7.02 BOOL  ; #1测试NG推料气缸缩回位
7.03 BOOL  ; #1测试NG推料气缸伸出位
7.04 BOOL  ; #2测试NG推料气缸缩回位
7.05 BOOL  ; #2测试NG推料气缸伸出位
7.06 BOOL  ; 出料拉带有料感应
7.07 BOOL  ; 备用
7.08 BOOL  ; 扫码位有料感应
7.09 BOOL  ; 氦检启动OK
7.10 BOOL  ; #1氦检阀原位
7.11 BOOL  ; #2氦检原位
7.12 BOOL  ; #3氦检原位
7.13 BOOL  ; #4氦检原位
7.14 BOOL  ; 备用
7.15 BOOL  ; 可放料信号
8.00 BOOL  ; 进料伺服Serv_On
8.01 BOOL  ; 进料伺服Alarm_Clr
8.02 BOOL  ; 出料伺服Serv_On
8.03 BOOL  ; 出料伺服Alarm_Clr
8.04 BOOL  ; 前腔体进料伺服Serv_On
8.05 BOOL  ; 前腔体进料伺服Alarm_Clr
8.06 BOOL  ; 后腔体进料伺服Serv_On
8.07 BOOL  ; 后腔体进料伺服Alarm_Clr
8.08 BOOL  ; 前腔体出料伺服Serv_On
8.09 BOOL  ; 进料伺服Alarm_Clr
8.10 BOOL  ; 后腔体出料伺服Serv_On
8.11 BOOL  ; 后腔体出料伺服Alarm_Clr
8.12 BOOL  ; 启动指示灯
8.13 BOOL  ; 停止指示灯
8.14 BOOL  ; 复位指示灯
8.15 BOOL  ; 三色绿灯
9.00 BOOL  ; 三色红灯
9.01 BOOL  ; 三色黄灯
9.02 BOOL  ; 蜂鸣器
9.03 BOOL  ; #1真空泵启动
9.04 BOOL  ; 氦检电源打开
9.05 BOOL  ; 氦检仪启动
9.06 BOOL  ; 扫码阻挡
9.07 BOOL  ; 隔离夹紧气缸
9.08 BOOL  ; 上料夹爪气缸
9.09 BOOL  ; 进料升降伺服Serv_On
9.10 BOOL  ; 出料伺服Alarm_Clr
9.11 BOOL  ; 上料横移气缸缩回
9.12 BOOL  ; 上料横移气缸伸出
9.13 BOOL  ; 下料夹爪气缸
9.14 BOOL  ; 出料升降伺服Serv_On
9.15 BOOL  ; 下料#2级升降气缸
A202.00 BOOL  ; 通信端口0允许标志
A202.01 BOOL  ; 通信端口1允许标志
A202.02 BOOL  ; 通信端口2允许标志
A202.03 BOOL  ; 通信端口3允许标志
A202.04 BOOL  ; 通信端口4允许标志
A202.05 BOOL  ; 通信端口5允许标志
A202.06 BOOL  ; 通信端口6允许标志
A202.07 BOOL  ; 通信端口7允许标志
A250.04 BOOL  ; 单元4重启
A276 CHANNEL  ; 脉冲输出0 PV
A278 CHANNEL  ; 脉冲输出1 PV
A280.00 BOOL  ; 脉冲输出 0脉冲输出状态(0：恒速中,1：加减速中)
A280.01 BOOL  ; 脉冲输出 0当前值上溢/下溢
A280.02 BOOL  ; 脉冲输出0脉冲输出量设定
A280.03 BOOL  ; 脉冲输出 0脉冲输出完成
A280.04 BOOL  ; 脉冲输出 0脉冲输出中
A280.05 BOOL  ; 前上料伺服无原点标志(0：原点确定,1：原点未确定)
A280.06 BOOL  ; 脉冲输出 0原点停止标志(0：未停于原点,1：原点停止中)
A280.07 BOOL  ; 脉冲输出 0 原点搜索异常停止标志
A281.00 BOOL  ; 脉冲输出 1脉冲输出状态(0：恒速中,1：加减速中)
A281.01 BOOL  ; 脉冲输出 1当前值上溢/下溢
A281.02 BOOL  ; 脉冲输出1脉冲输出量设定
A281.03 BOOL  ; 脉冲输出 1脉冲输出完成
A281.04 BOOL  ; 脉冲输出 1脉冲输出中
A281.05 BOOL  ; 脉冲输出 1无原点标志(0：原点确定,1：原点未确定)
A281.06 BOOL  ; 脉冲输出 1原点停止标志(0：未停于原点,1：原点停止中)
A281.07 BOOL  ; 脉冲输出 1 原点搜索异常停止标志
A322 CHANNEL  ; 脉冲输出2 PV
A324 CHANNEL  ; 脉冲输出3 PV
A326.04 BOOL  ; 后上料伺服脉冲输出中
A326.05 BOOL  ; 后上料伺服无原点标志
A327.04 BOOL  ; 脉冲输出3脉冲输出中
A327.05 BOOL  ; 脉冲输出3无原点标志
A351 CHANNEL  ; 系统时间
A501.04 BOOL  ; 单元4模块重启
A623.01 BOOL  ; 3单元#1串口重启
A623.02 BOOL  ; 3单元#2串口重启
C0000 BOOL  ; 进料到后放料位次数
C0001 BOOL  ; MES离线模式下进料次数
C0010 BOOL  ; 1#腔清氦次数到达
C0020 BOOL  ; 2#腔清氦次数到达
C0030 BOOL  ; 3#腔清氦次数到达
C0040 BOOL  ; 4#腔清氦次数到达
C0060 BOOL  ; 自动重扫次数
C0090 BOOL  ; 出料到后取料位次数
D0 CHANNEL  ; PLC控制HMI切换的窗口编号
D1 CHANNEL  ; 当前窗口编号
D10 CHANNEL  ; 当前报警代码
D100 CHANNEL  ; #4腔体进入自保前时间
D1000 CHANNEL  ; 扫码自动运行步编号
D1001 CHANNEL  ; 前上料机构自动运行步编号
D1002 CHANNEL  ; 前下料机构自动运行步编号
D1003 CHANNEL  ; 后上料机构自动运行步编号
D1004 CHANNEL  ; 后下料机构自动运行步编号
D1005 CHANNEL  ; 1#腔体机构自动运行步编号
D1006 CHANNEL  ; 2#腔体机构自动运行步编号
D1007 CHANNEL  ; 3#腔体机构自动运行步编号
D1008 CHANNEL  ; 4#腔体机构自动运行步编号
D1009 CHANNEL  ; 出料机构自动运行步编号
D101 CHANNEL  ; #4腔体自保时间
D1010 CHANNEL  ; 扫码机构自动运行步编号
D10102 CHANNEL  ; 安东启动限制（0启动 1禁止）
D10103 CHANNEL  ; 启停故障原因
D10104 CHANNEL  ; PPM
D10105 CHANNEL  ; 启动限制断开（系统赋值1 PLC赋值0）
D10106 CHANNEL  ; 实时PPM
D10108 CHANNEL  ; 绿灯状态
D10109 CHANNEL  ; 红灯
D10110 CHANNEL  ; 黄灯
D10122 CHANNEL  ; 总投入
D10124 CHANNEL  ; .
D10126 CHANNEL  ; 总产出
D1015 CHANNEL  ; 1#腔体自动清氦步编号
D1016 CHANNEL  ; 2#腔体自动清氦步编号
D1017 CHANNEL  ; 3#腔体自动清氦步编号
D1018 CHANNEL  ; 4#腔体自动清氦步编号
D11 CHANNEL  ; 当前报警数量
D1142 CHANNEL  ; #1腔体测试结果
D1144 CHANNEL  ; #2腔体测试结果
D1146 CHANNEL  ; #3测试结果
D1148 CHANNEL  ; #4腔体测试结果
D1152 CHANNEL  ; 放OK品次数
D1154 CHANNEL  ; 放NG品次数
D116 CHANNEL  ; 前上料往腔体1放料安全位置
D1160 CHANNEL  ; 生产总数
D1162 CHANNEL  ; 生产OK品总数
D1164 CHANNEL  ; 生产NG品总数
D1166 CHANNEL  ; 良品率(%)
D118 CHANNEL  ; 前下料腔体1取料安全位
D1200 CHANNEL  ; 腔体真空阀值
D1202 CHANNEL  ; 腔体抽真空时间
D1204 CHANNEL  ; 检漏口压力设定值
D1206 CHANNEL  ; 漏率设定值
D1208 CHANNEL  ; 电池破真空阀值
D1210 CHANNEL  ; 氦检仪稳定设定时间
D1212 CHANNEL  ; 腔体破真空阀值
D1214 CHANNEL  ; 腔体抽氦后压力
D1216 CHANNEL  ; 自检真空阀值
D1218 CHANNEL  ; 自检抽真空时间
D1220 CHANNEL  ; 自检泄漏量
D1222 CHANNEL  ; 自检保压前延时-HMI
D1224 CHANNEL  ; 自检保压时间-HMI
D1226 CHANNEL  ; 氦检时间
D1228 CHANNEL  ; 抽残气时间
D1229 CHANNEL  ; 抽残气压力达到延时
D1230 CHANNEL  ; 电池抽真空阀值
D1232 CHANNEL  ; 电池抽真空时间
D1234 CHANNEL  ; 注氦后压力
D1236 CHANNEL  ; 电池抽氦后压力
D1238 CHANNEL  ; 注氦气时间
D1240 CHANNEL  ; 氦检时的真空阀值
D1242 CHANNEL  ; 充氦压力下限值Pa(F)
D1246 CHANNEL  ; 充氦压力上限值Pa(F)
D1250 CHANNEL  ; 检漏口压力设定值小数部分
D1252 CHANNEL  ; 检漏口压力设定值指数
D1254 CHANNEL  ; 漏率设定值小数部分
D1256 CHANNEL  ; 漏率设定值指数
D1260 CHANNEL  ; 检漏口压力设定值指数部分
D1264 CHANNEL  ; 漏率设定值指数部分
D1266 CHANNEL  ; 漏率设定值(浮点数Pa.m3)
D1270 CHANNEL  ; 注氦嘴气密性设定值小数部分
D1272 CHANNEL  ; 注氦嘴气密性设定值指数
D1274 CHANNEL  ; 注氦嘴气密性设定值指数部分
D1276 CHANNEL  ; 注氦嘴气密性设定值(Float)
D1278 CHANNEL  ; 清氦次数设定值
D1280 CHANNEL  ; 1#腔体抽气阀关闭延时
D1282 CHANNEL  ; 2#腔体抽气阀关闭延时
D1284 CHANNEL  ; 3#腔体抽气阀关闭延时
D1286 CHANNEL  ; 4#腔体抽气阀关闭延时
D1290 CHANNEL  ; 1#腔体抽残气时间
D1292 CHANNEL  ; 2#腔体抽残气时间
D1294 CHANNEL  ; 3#腔体抽残气时间
D1296 CHANNEL  ; 4#腔体抽残气时间
D130 CHANNEL  ; 前腔体电池NG状态
D130.00 BOOL  ; 1#腔电池NG
D130.01 BOOL  ; 2#腔电池NG
D131 CHANNEL  ; 后腔体电池NG状态
D1310 CHANNEL  ; 氦检仪稳定漏率设定值小数
D1312 CHANNEL  ; 氦检仪稳定漏率设定值指数
D1316 CHANNEL  ; 氦检仪稳定漏率设定值(Float)
D131.00 BOOL  ; 3#腔电池NG
D131.01 BOOL  ; 4#腔电池NG
D1330 CHANNEL  ; #1腔体注氦压力阀值
D1332 CHANNEL  ; #2腔体注氦压力阀值
D1334 CHANNEL  ; #3腔体注氦压力阀值
D1336 CHANNEL  ; #4腔体注氦压力阀值
D1342 CHANNEL  ; 充氦压力下限值kPa(F)
D1346 CHANNEL  ; 充氦压力上限值kPa(F)
D135 CHANNEL  ; 清氦失败腔体号
D1350 CHANNEL  ; 1#腔体充氦时电池实际压力（浮点）
D1352 CHANNEL  ; 1#腔体氦检时腔体实际压力（浮点）
D1354 CHANNEL  ; 2#腔体充氦时电池实际压力（浮点）
D1356 CHANNEL  ; 2#腔体氦检时腔体实际压力（浮点）
D1358 CHANNEL  ; 3#腔体充氦时电池实际压力（浮点）
D1360 CHANNEL  ; 3#腔体氦检时腔体实际压力（浮点）
D1362 CHANNEL  ; 4#腔体充氦时电池实际压力（浮点）
D1364 CHANNEL  ; 4#腔体氦检时腔体实际压力（浮点）
D1366 CHANNEL  ; 前下料爪 充氦时电池实际压力（浮点）
D1368 CHANNEL  ; 前下料爪 氦检时腔体实际压力（浮点）
D1370 CHANNEL  ; 后下料爪 充氦时电池实际压力（浮点）
D1372 CHANNEL  ; 后下料爪 氦检时腔体实际压力（浮点）
D14 CHANNEL  ; 感应器ON延时时间
D1400 CHANNEL  ; #1连续NG次数
D1401 CHANNEL  ; #2腔体连续NG次数
D1402 CHANNEL  ; #3腔体连续NG次数
D1403 CHANNEL  ; #4腔体连续NG次数
D1410 CHANNEL  ; 连续NG报警设定
D1411 CHANNEL  ; 自动离线次数
D1412 CHANNEL  ; NG报警状态
D1415 CHANNEL  ; 写数据超时时间
D1416 CHANNEL  ; 氦检仪压力异常延时
D1500 CHANNEL  ; 来料隔离气缸缩回位
D1501 CHANNEL  ; 来料隔离气缸伸出位屏蔽延时时间
D1502 CHANNEL  ; 扫码阻挡气缸缩回位屏蔽延时时间
D1503 CHANNEL  ; 扫码阻挡气缸伸出屏蔽延时时间
D1504 CHANNEL  ; 上料夹爪张开位屏蔽延时时间
D1505 CHANNEL  ; 上料夹爪夹紧位屏蔽延时时间
D1506 CHANNEL  ; 上料#1气缸缩回位蔽延时时间
D1507 CHANNEL  ; 上料#1气缸伸出位屏蔽延时时间
D1508 CHANNEL  ; 上料#2气缸缩回位屏蔽延时
D1509 CHANNEL  ; 上料#2气缸伸出位屏蔽延时
D1510 CHANNEL  ; 上料横移气缸缩回位屏蔽延时
D1511 CHANNEL  ; 上料横移气缸伸出位屏蔽延时
D1512 CHANNEL  ; 下料夹爪张开位蔽延时时间
D1513 CHANNEL  ; 下料夹爪夹紧位屏蔽延时时间
D1514 CHANNEL  ; 下料#1升降气缸缩回位屏蔽延时
D1515 CHANNEL  ; 下料#1级升降气缸伸出位屏蔽延时
D1516 CHANNEL  ; 下料#2级升降气缸缩回位蔽延时时间
D1517 CHANNEL  ; 下料#2级升降气缸伸出位屏蔽延时时间
D1518 CHANNEL  ; 下料横移气缸缩回位蔽延时时间
D1519 CHANNEL  ; 下料横移气缸伸出位屏蔽延时
D1520 CHANNEL  ; 拉带进料夹爪有料感应延时时间
D1521 CHANNEL  ; 拉带出料夹爪有料感应延时时间
D1522 CHANNEL  ; 前腔体进料夹爪有料感应屏蔽延时
D1523 CHANNEL  ; 前腔体出料夹爪有料感应屏蔽延时
D1524 CHANNEL  ; 后腔体进料夹爪有料感应
D1525 CHANNEL  ; 后腔体出料夹爪有料感应
D1526 CHANNEL  ; 精密调压阀过低报警
D1527 CHANNEL  ; 后腔体出料位顶升气缸伸出位屏蔽延时
D1528 CHANNEL  ; 前腔体进料机械手夹爪张开位屏蔽延时时间
D1529 CHANNEL  ; 前腔体进料机械手夹爪夹紧位屏蔽延时
D1530 CHANNEL  ; 前腔体进料机械手升降气缸缩回位屏蔽延时
D1531 CHANNEL  ; 前腔体进料机械手升降气缸伸出位屏蔽延时
D1532 CHANNEL  ; 后腔体进料机械手张开位屏蔽延时
D1533 CHANNEL  ; 后腔体进料机械手夹爪夹紧位屏蔽延时
D1534 CHANNEL  ; 后腔体进料机械手升降气缸缩回位屏蔽延时
D1535 CHANNEL  ; 后腔体进料机械手升降气缸伸出位屏蔽延时
D1536 CHANNEL  ; 前腔体上料机械手夹爪张开位屏蔽延时
D1537 CHANNEL  ; 前腔体出料机械手夹爪夹紧位屏蔽延时
D1538 CHANNEL  ; 前腔体出料机械手升降气缸缩回位屏蔽延时
D1539 CHANNEL  ; 前腔体出料机械手升降气缸伸出位屏蔽延时
D1540 CHANNEL  ; 后腔体出料机械手夹爪张开位屏蔽延时
D1541 CHANNEL  ; 后腔体出料机械手夹爪夹紧位屏蔽延时
D1542 CHANNEL  ; 后腔体出料机械手升降气缸缩回位屏蔽延时
D1543 CHANNEL  ; 后腔体出料机械手升降气缸伸出位屏蔽延时
D1544 CHANNEL  ; #1腔体移栽气缸缩回位屏蔽延时
D1545 CHANNEL  ; #1腔体移栽气缸伸出位屏蔽延时
D1546 CHANNEL  ; #1腔体顶升气缸缩回位屏蔽延时
D1547 CHANNEL  ; #1腔体顶升气缸伸出位屏蔽延时
D1548 CHANNEL  ; #2腔体移栽气缸缩回位屏蔽延时
D1549 CHANNEL  ; #2腔体移栽气缸伸出位屏蔽延时
D1550 CHANNEL  ; #2腔体顶升气缸缩回位屏蔽延时
D1551 CHANNEL  ; #2腔体顶升气缸伸出位屏蔽延时
D1552 CHANNEL  ; #3腔体移栽气缸缩回位屏蔽延时
D1553 CHANNEL  ; #3腔体移栽气缸伸出位屏蔽延时
D1554 CHANNEL  ; #3腔体顶升气缸缩回位屏蔽延时
D1555 CHANNEL  ; #3腔体顶升气缸伸出位屏蔽延时
D1556 CHANNEL  ; #4腔体移栽气缸缩回位屏蔽延时
D1557 CHANNEL  ; #4腔体移栽气缸伸出位屏蔽延时
D1558 CHANNEL  ; #4腔体顶升气缸缩回位屏蔽延时
D1559 CHANNEL  ; #4腔体顶升气缸伸出位屏蔽延时
D1560 CHANNEL  ; #1扫码NG推料气缸缩回位屏蔽延时
D1561 CHANNEL  ; #1扫码NG推料气缸伸出位屏蔽延时
D1562 CHANNEL  ; #2扫码NG推料气缸缩回位屏蔽延时
D1563 CHANNEL  ; #2扫码NG推料气缸伸出位屏蔽延时
D1564 CHANNEL  ; #1测试NG推料气缸缩回位屏蔽延时
D1565 CHANNEL  ; #1测试NG推料气缸伸出屏蔽延时
D1566 CHANNEL  ; #2测试NG推料气缸缩回位屏蔽延时
D1567 CHANNEL  ; #2测试NG推料气缸伸出位屏蔽延时
D1568 CHANNEL  ; 前进料旋转气缸初始位屏蔽延时时间
D1569 CHANNEL  ; 前进料旋转气缸旋转位屏蔽延时时间
D1570 CHANNEL  ; 前出料旋转气缸初始位屏蔽延时时间
D1571 CHANNEL  ; 前出料旋转气缸旋转位屏蔽延时时间
D1572 CHANNEL  ; 后进料旋转气缸初始位屏蔽延时时间
D1573 CHANNEL  ; 后进料旋转气缸旋转位屏蔽延时时间
D1574 CHANNEL  ; 后出料旋转气缸初始位屏蔽延时时间
D1575 CHANNEL  ; 后出料旋转气缸旋转位屏蔽延时时间
D1580 CHANNEL  ; 腔体1左电池密封气缸上位屏蔽延时时间
D1581 CHANNEL  ; 腔体1左电池密封气缸下位屏蔽延时时间
D1582 CHANNEL  ; 腔体1右电池密封气缸上位屏蔽延时时间
D1583 CHANNEL  ; 腔体1右电池密封气缸下位屏蔽延时时间
D1584 CHANNEL  ; 腔体2左电池密封气缸上位屏蔽延时时间
D1585 CHANNEL  ; 腔体2左电池密封气缸下位屏蔽延时时间
D1586 CHANNEL  ; 腔体2右电池密封气缸上位屏蔽延时时间
D1587 CHANNEL  ; 腔体2右电池密封气缸下位屏蔽延时时间
D1588 CHANNEL  ; 腔体3左电池密封气缸上位屏蔽延时时间
D1589 CHANNEL  ; 腔体3左电池密封气缸下位屏蔽延时时间
D1590 CHANNEL  ; 腔体3右电池密封气缸上位屏蔽延时时间
D1591 CHANNEL  ; 腔体3右电池密封气缸下位屏蔽延时时间
D1592 CHANNEL  ; 腔体4左电池密封气缸上位屏蔽延时时间
D1593 CHANNEL  ; 腔体4左电池密封气缸下位屏蔽延时时间
D1594 CHANNEL  ; 腔体4右电池密封气缸上位屏蔽延时时间
D1595 CHANNEL  ; 腔体4右电池密封气缸下位屏蔽延时时间
D1596 CHANNEL  ; 腔体1平移气缸后退位屏蔽延时时间
D1597 CHANNEL  ; 腔体1平移气缸前进位屏蔽延时时间
D1598 CHANNEL  ; 腔体1顶升气缸下位屏蔽延时时间
D1599 CHANNEL  ; 腔体1顶升气缸上位屏蔽延时时间
D16 CHANNEL  ; 感应器Off延时时间
D1600 CHANNEL  ; 腔体2平移气缸后退位屏蔽延时时间
D1601 CHANNEL  ; 腔体2平移气缸前进位屏蔽延时时间
D1602 CHANNEL  ; 腔体2顶升气缸下位屏蔽延时时间
D1603 CHANNEL  ; 腔体2顶升气缸上位屏蔽延时时间
D1604 CHANNEL  ; 腔体3平移气缸后退位屏蔽延时时间
D1605 CHANNEL  ; 腔体3平移气缸前进位屏蔽延时时间
D1606 CHANNEL  ; 腔体3顶升气缸下位屏蔽延时时间
D1607 CHANNEL  ; 腔体3顶升气缸上位屏蔽延时时间
D1608 CHANNEL  ; 腔体4平移气缸后退位屏蔽延时时间
D1609 CHANNEL  ; 腔体4平移气缸前进位屏蔽延时时间
D1610 CHANNEL  ; 腔体4顶升气缸下位屏蔽延时时间
D1611 CHANNEL  ; 腔体4顶升气缸上位屏蔽延时时间
D1700 CHANNEL  ; 左进料阻挡气缸放行位屏蔽设定时间
D1701 CHANNEL  ; 左进料阻挡气缸阻挡位屏蔽设定时间
D1702 CHANNEL  ; 右进料阻挡气缸放行位屏蔽设定时间
D1703 CHANNEL  ; 右进料阻挡气缸阻挡位屏蔽设定时间
D1704 CHANNEL  ; 左扫码阻挡气缸放行位屏蔽设定时间
D1705 CHANNEL  ; 左扫码阻挡气缸阻挡位屏蔽设定时间
D1706 CHANNEL  ; 右扫码阻挡气缸放行位屏蔽设定时间
D1707 CHANNEL  ; 右扫码阻挡气缸阻挡位屏蔽设定时间
D1708 CHANNEL  ; 扫码NG缓存避位气缸接料位屏蔽设定时间
D1709 CHANNEL  ; 扫码NG缓存避位气缸避位位屏蔽设定时间
D1710 CHANNEL  ; 扫码NG缓存接料气缸后退位屏蔽设定时间
D1711 CHANNEL  ; 扫码NG缓存接料气缸前进位屏蔽设定时间
D1712 CHANNEL  ; 扫码NG缓存间隔气缸上位屏蔽设定时间
D1713 CHANNEL  ; 扫码NG缓存间隔气缸下位屏蔽设定时间
D1716 CHANNEL  ; 进料机械手升降气缸上位屏蔽设定时间
D1717 CHANNEL  ; 进料机械手升降气缸下位屏蔽设定时间
D1718 CHANNEL  ; 进料机械手平移气缸开位屏蔽设定时间
D1719 CHANNEL  ; 进料机械手平移气缸合位屏蔽设定时间
D1720 CHANNEL  ; 进料机械手左夹爪气缸张开位屏蔽设定时间
D1721 CHANNEL  ; 进料机械手左夹爪气缸夹紧位屏蔽设定时间
D1722 CHANNEL  ; 进料机械手右夹爪气缸张开位屏蔽设定时间
D1723 CHANNEL  ; 进料机械手右夹爪气缸夹紧位屏蔽设定时间
D1724 CHANNEL  ; 出料机械手升降气缸上位屏蔽设定时间
D1725 CHANNEL  ; 出料机械手升降气缸下位屏蔽设定时间
D1726 CHANNEL  ; 出料机械手平移气缸开位屏蔽设定时间
D1727 CHANNEL  ; 出料机械手平移气缸合位屏蔽设定时间
D1728 CHANNEL  ; 出料机械手左夹爪气缸张开位屏蔽设定时间
D1729 CHANNEL  ; 出料机械手左夹爪气缸夹紧位屏蔽设定时间
D1730 CHANNEL  ; 出料机械手右夹爪气缸张开位屏蔽设定时间
D1731 CHANNEL  ; 出料机械手右夹爪气缸夹紧位屏蔽设定时间
D1732 CHANNEL  ; 前上料机械手1级升降气缸上位屏蔽设定时间
D1733 CHANNEL  ; 前上料机械手1级升降气缸下位屏蔽设定时间
D1734 CHANNEL  ; 前上料机械手2级升降气缸上位屏蔽设定时间
D1735 CHANNEL  ; 前上料机械手2级升降气缸下位屏蔽设定时间
D1736 CHANNEL  ; 前上料机械手左夹爪气缸张开位屏蔽设定时间
D1737 CHANNEL  ; 前上料机械手左夹爪气缸夹紧位屏蔽设定时间
D1738 CHANNEL  ; 前上料机械手右夹爪气缸张开位屏蔽设定时间
D1739 CHANNEL  ; 前上料机械手右夹爪气缸夹紧位屏蔽设定时间
D1740 CHANNEL  ; 前取料机械手1级升降气缸上位屏蔽设定时间
D1741 CHANNEL  ; 前取料机械手1级升降气缸下位屏蔽设定时间
D1742 CHANNEL  ; 前取料机械手2级升降气缸上位屏蔽设定时间
D1743 CHANNEL  ; 前取料机械手2级升降气缸下位屏蔽设定时间
D1744 CHANNEL  ; 前取料机械手左夹爪气缸张开位屏蔽设定时间
D1745 CHANNEL  ; 前取料机械手左夹爪气缸夹紧位屏蔽设定时间
D1746 CHANNEL  ; 前取料机械手右夹爪气缸张开位屏蔽设定时间
D1747 CHANNEL  ; 前取料机械手右夹爪气缸夹紧位屏蔽设定时间
D1748 CHANNEL  ; 后上料机械手1级升降气缸上位屏蔽设定时间
D1749 CHANNEL  ; 后上料机械手1级升降气缸下位屏蔽设定时间
D1750 CHANNEL  ; 后上料机械手2级升降气缸上位屏蔽设定时间
D1751 CHANNEL  ; 后上料机械手2级升降气缸下位屏蔽设定时间
D1752 CHANNEL  ; 后上料机械手左夹爪气缸张开位屏蔽设定时间
D1753 CHANNEL  ; 后上料机械手左夹爪气缸夹紧位屏蔽设定时间
D1754 CHANNEL  ; 后上料机械手右夹爪气缸张开位屏蔽设定时间
D1755 CHANNEL  ; 后上料机械手右夹爪气缸夹紧位屏蔽设定时间
D1756 CHANNEL  ; 后取料机械手1级升降气缸上位屏蔽设定时间
D1757 CHANNEL  ; 后取料机械手1级升降气缸下位屏蔽设定时间
D1758 CHANNEL  ; 后取料机械手2级升降气缸上位屏蔽设定时间
D1759 CHANNEL  ; 后取料机械手2级升降气缸下位屏蔽设定时间
D1760 CHANNEL  ; 后取料机械手左夹爪气缸张开位屏蔽设定时间
D1761 CHANNEL  ; 后取料机械手左夹爪气缸夹紧位屏蔽设定时间
D1762 CHANNEL  ; 后取料机械手右夹爪气缸张开位屏蔽设定时间
D1763 CHANNEL  ; 后取料机械手右夹爪气缸夹紧位屏蔽设定时间
D1764 CHANNEL  ; 前NG拨料气缸后位屏蔽设定时间
D1765 CHANNEL  ; 前NG拨料气缸前位屏蔽设定时间
D1766 CHANNEL  ; 后NG拨料气缸后位屏蔽设定时间
D1767 CHANNEL  ; 后NG拨料气缸前位屏蔽设定时间
D1768 CHANNEL  ; 前进料旋转气缸初始位屏蔽设定时间
D1769 CHANNEL  ; 前进料旋转气缸旋转位屏蔽设定时间
D1770 CHANNEL  ; 前出料旋转气缸初始位屏蔽设定时间
D1771 CHANNEL  ; 前出料旋转气缸旋转位屏蔽设定时间
D1772 CHANNEL  ; 后进料旋转气缸初始位屏蔽设定时间
D1773 CHANNEL  ; 后进料旋转气缸旋转位屏蔽设定时间
D1774 CHANNEL  ; 后出料旋转气缸初始位屏蔽设定时间
D1775 CHANNEL  ; 后出料旋转气缸旋转位屏蔽设定时间
D1780 CHANNEL  ; 腔体1左电池密封气缸上位屏蔽设定时间
D1781 CHANNEL  ; 腔体1左电池密封气缸下位屏蔽设定时间
D1782 CHANNEL  ; 腔体1右电池密封气缸上位屏蔽设定时间
D1783 CHANNEL  ; 腔体1右电池密封气缸下位屏蔽设定时间
D1784 CHANNEL  ; 腔体2左电池密封气缸上位屏蔽设定时间
D1785 CHANNEL  ; 腔体2左电池密封气缸下位屏蔽设定时间
D1786 CHANNEL  ; 腔体2右电池密封气缸上位屏蔽设定时间
D1787 CHANNEL  ; 腔体2右电池密封气缸下位屏蔽设定时间
D1788 CHANNEL  ; 腔体3左电池密封气缸上位屏蔽设定时间
D1789 CHANNEL  ; 腔体3左电池密封气缸下位屏蔽设定时间
D1790 CHANNEL  ; 腔体3右电池密封气缸上位屏蔽设定时间
D1791 CHANNEL  ; 腔体3右电池密封气缸下位屏蔽设定时间
D1792 CHANNEL  ; 腔体4左电池密封气缸上位屏蔽设定时间
D1793 CHANNEL  ; 腔体4左电池密封气缸下位屏蔽设定时间
D1794 CHANNEL  ; 腔体4右电池密封气缸上位屏蔽设定时间
D1795 CHANNEL  ; 腔体4右电池密封气缸下位屏蔽设定时间
D1796 CHANNEL  ; 腔体1平移气缸后退位屏蔽设定时间
D1797 CHANNEL  ; 腔体1平移气缸前进位屏蔽设定时间
D1798 CHANNEL  ; 腔体1顶升气缸下位屏蔽设定时间
D1799 CHANNEL  ; 腔体1顶升气缸上位屏蔽设定时间
D18 CHANNEL  ; 自动运行条件延时时间
D1800 CHANNEL  ; 腔体2平移气缸后退位屏蔽设定时间
D1801 CHANNEL  ; 腔体2平移气缸前进位屏蔽设定时间
D1802 CHANNEL  ; 腔体2顶升气缸下位屏蔽设定时间
D1803 CHANNEL  ; 腔体2顶升气缸上位屏蔽设定时间
D1804 CHANNEL  ; 腔体3平移气缸后退位屏蔽设定时间
D1805 CHANNEL  ; 腔体3平移气缸前进位屏蔽设定时间
D1806 CHANNEL  ; 腔体3顶升气缸下位屏蔽设定时间
D1807 CHANNEL  ; 腔体3顶升气缸上位屏蔽设定时间
D1808 CHANNEL  ; 腔体4平移气缸后退位屏蔽设定时间
D1809 CHANNEL  ; 腔体4平移气缸前进位屏蔽设定时间
D1810 CHANNEL  ; 腔体4顶升气缸下位屏蔽设定时间
D1811 CHANNEL  ; 腔体4顶升气缸上位屏蔽设定时间
D19 CHANNEL  ; 自动运行步间间隔时间
D2 CHANNEL  ; 机台有柔性报警
D20 CHANNEL  ; 轴控位置预置
D2000 CHANNEL  ; 进料水平伺服手动低速加速时间
D2001 CHANNEL  ; 进料伺服手动低速加速时间
D2002 CHANNEL  ; 进料水平移载伺服手动低速减速时间
D2003 CHANNEL  ; 进料伺服手动低速减速时间
D2004 CHANNEL  ; 进料水平移载伺服手动低速速度
D2005 CHANNEL  ; 进料伺服手动低速速度
D2006 CHANNEL  ; 进料伺服手动低速输出脉冲
D20068 CHANNEL  ; 进料伺服定位位置
D20069 CHANNEL  ; 进料伺服定位位置
D2007 CHANNEL  ; 进料伺服手动低速输出脉冲
D20070 CHANNEL  ; 进料伺服定位速度
D20071 CHANNEL  ; 进料伺服定位速度
D20072 CHANNEL  ; 进料伺服加速时间
D20073 CHANNEL  ; 进料伺服加速时间
D20074 CHANNEL  ; 进料伺服减速时间
D20075 CHANNEL  ; 进料伺服减速时间
D2008 CHANNEL  ; 进料水平移载伺服手动当前速度
D20080 CHANNEL  ; 出料伺服定位位置
D20081 CHANNEL  ; 出料伺服定位位置
D20082 CHANNEL  ; 出料伺服定位速度
D20083 CHANNEL  ; 出料伺服定位速度
D20084 CHANNEL  ; 出料伺服加速时间
D20085 CHANNEL  ; 出料伺服加速时间
D20086 CHANNEL  ; 出料伺服减速时间
D20087 CHANNEL  ; 出料伺服减速时间
D2009 CHANNEL  ; 进料伺服手动当前速度
D20092 CHANNEL  ; 进料伺服当前位置
D20093 CHANNEL  ; 进料伺服当前位置
D20096 CHANNEL  ; 出料伺服当前位置
D20097 CHANNEL  ; 出料伺服当前位置
D2010 CHANNEL  ; 进料移载伺服手动高速加速时间
D2011 CHANNEL  ; 进料伺服手动高速加速时间
D2012 CHANNEL  ; 进料移载伺服手动高速减速时间
D20124 CHANNEL  ; 进料伺服定位位置
D20126 CHANNEL  ; 进料水平移载伺服定位速度
D20128 CHANNEL  ; 进料水平伺服加速时间
D2013 CHANNEL  ; 进料伺服手动高速减速时间
D20130 CHANNEL  ; 进料水平伺服减速度
D20136 CHANNEL  ; 出料伺服定位位置
D20138 CHANNEL  ; 出料移载伺服定位速度
D2014 CHANNEL  ; 进料伺服手动高速速度
D20140 CHANNEL  ; 出料移载伺服加速时间
D20142 CHANNEL  ; 出料移载伺服减速时间
D20148 CHANNEL  ; 进料升降伺服定位位置
D2015 CHANNEL  ; 进料伺服手动高速速度
D20150 CHANNEL  ; 进料升降伺服定位速度
D20152 CHANNEL  ; 进料升降伺服加速时间
D20154 CHANNEL  ; 进料升降伺服减速度
D2016 CHANNEL  ; 进料伺服手动高速输出脉冲
D20160 CHANNEL  ; 出料升降伺服定位位置
D20162 CHANNEL  ; 出料升降伺服定位速度
D20164 CHANNEL  ; 出料升降伺服加速时间
D20166 CHANNEL  ; 出料升降伺服减速时间
D2017 CHANNEL  ; 进料伺服手动高速输出脉冲
D20172 CHANNEL  ; 进料移载伺服当前位置
D20176 CHANNEL  ; 出料移载伺服当前位置
D2018 CHANNEL  ; 进料伺服寸动距离
D20180 CHANNEL  ; 进料升降伺服当前位置
D20184 CHANNEL  ; 出料升降伺服当前位置
D2019 CHANNEL  ; 进料伺服寸动距离
D2020 CHANNEL  ; 进料水平移载伺服自动加速时间
D2021 CHANNEL  ; 进料伺服自动加速时间
D2022 CHANNEL  ; 进料水平移载伺服自动减速时间
D2023 CHANNEL  ; 进料伺服自动减速时间
D2024 CHANNEL  ; 进料移载伺服自动速度
D2025 CHANNEL  ; 进料伺服自动速度
D2026 CHANNEL  ; 进料伺服自动输出脉冲
D2027 CHANNEL  ; 进料伺服自动输出脉冲
D2028 CHANNEL  ; 进料伺服自动速度2(低速)
D2030 CHANNEL  ; #4扫码NG位
D2031 CHANNEL  ; 进料伺服待机位置
D2032 CHANNEL  ; 进料水平伺服上料位置
D2033 CHANNEL  ; 进料伺服上料位置
D2034 CHANNEL  ; 进料水平伺服前放料位
D2035 CHANNEL  ; 进料伺服前放料位
D2036 CHANNEL  ; 进料水平伺服后放料位
D2037 CHANNEL  ; 进料伺服后放料位
D2040 CHANNEL  ; #1扫码NG位
D2041 CHANNEL  ; 外部拉带安全运行进料伺服位置
D2042 CHANNEL  ; #2扫码NG位
D2044 CHANNEL  ; #3扫码NG位
D2046 CHANNEL  ; #4扫码NG位
D2050 CHANNEL  ; 进出料转盘直径
D2080 CHANNEL  ; #2扫码NG位
D2082 CHANNEL  ; 前进料转盘后直径边缘位置
D2084 CHANNEL  ; 后进料转盘前直径边缘位置
D2086 CHANNEL  ; 后进料转盘后直径边缘位置
D2100 CHANNEL  ; 前上料伺服手动低速加速比率
D2101 CHANNEL  ; 前上料伺服手动低速减速比率
D2102 CHANNEL  ; 前上料伺服手动低速速度
D2103 CHANNEL  ; 前上料伺服手动低速速度
D2104 CHANNEL  ; 前上料伺服手动低速输出脉冲
D2105 CHANNEL  ; 前上料伺服手动输出脉冲
D2106 CHANNEL  ; 前上料伺服手动启动速度
D2107 CHANNEL  ; 前上料伺服手动启动速度
D2108 CHANNEL  ; 前上料伺服手动当前速度
D2109 CHANNEL  ; 前上料伺服手动当前速度
D2110 CHANNEL  ; 前上料伺服手动高速加速比率
D2111 CHANNEL  ; 前上料伺服手动高速减速比率
D2112 CHANNEL  ; 前上料伺服手动高速速度
D2113 CHANNEL  ; 前上料伺服手动高速速度
D2114 CHANNEL  ; 前上料伺服手动高速输出脉冲
D2115 CHANNEL  ; 前上料伺服手动高速输出脉冲
D2116 CHANNEL  ; 前上料伺服手动高速启动速度
D2117 CHANNEL  ; 前上料伺服手动高速启动速度
D2118 CHANNEL  ; 前上料伺服寸动距离
D2119 CHANNEL  ; 前上料伺服寸动距离
D2120 CHANNEL  ; 前上料伺服自动加速比率
D2121 CHANNEL  ; 前上料伺服自动减速比率
D2122 CHANNEL  ; 前上料伺服自动速度
D2123 CHANNEL  ; 前上料伺服自动速度
D2124 CHANNEL  ; 前上料伺服自动输出脉冲
D2125 CHANNEL  ; 前上料伺服自动输出脉冲
D2126 CHANNEL  ; 前上料伺服自动启动速度
D2127 CHANNEL  ; 前上料伺服自动启动速度
D2130 CHANNEL  ; 前上料伺服待机位置
D2131 CHANNEL  ; 前上料伺服待机位置
D2132 CHANNEL  ; 前上料伺服上料位置
D2133 CHANNEL  ; 前上料伺服上料位置
D2134 CHANNEL  ; 前上料伺服仓1放料位
D2135 CHANNEL  ; 前上料伺服仓1放料位
D2136 CHANNEL  ; 前上料伺服仓2放料位
D2137 CHANNEL  ; 前上料伺服仓2放料位
D2140 CHANNEL  ; 安全位置
D2141 CHANNEL  ; 安全位置
D2150 CHANNEL  ; 前上料伺服上料位置
D2154 CHANNEL  ; 前上料伺服仓1放料位
D2160 CHANNEL  ; 前上料伺服仓2放料位
D220 CHANNEL  ; 接收检漏仪状态的起始字
D2200 CHANNEL  ; 前下料伺服手动低速加速比率
D2201 CHANNEL  ; 前下料伺服手动低速减速比率
D2202 CHANNEL  ; 前下料伺服手动低速速度
D2203 CHANNEL  ; 前下料伺服手动低速速度
D2204 CHANNEL  ; 前下料伺服手动输出脉冲
D2205 CHANNEL  ; 前下料伺服手动输出脉冲
D2206 CHANNEL  ; 前下料伺服手动启动速度
D2207 CHANNEL  ; 前下料伺服手动启动速度
D2208 CHANNEL  ; 前下料伺服手动当前速度
D2209 CHANNEL  ; 前下料伺服手动当前速度
D221 CHANNEL  ; 接收的检漏仪状态
D2210 CHANNEL  ; 前下料伺服手动高速加速比率
D2211 CHANNEL  ; 前下料伺服手动高速减速比率
D2212 CHANNEL  ; 前下料伺服手动高速速度
D2213 CHANNEL  ; 前下料伺服手动高速速度
D2214 CHANNEL  ; 前下料伺服手动高速输出脉冲
D2215 CHANNEL  ; 前下料伺服手动高速输出脉冲
D2216 CHANNEL  ; 前下料伺服手动高速启动速度
D2217 CHANNEL  ; 前下料伺服手动高速启动速度
D2218 CHANNEL  ; 前下料伺服寸动距离
D2219 CHANNEL  ; 前下料伺服寸动距离
D2220 CHANNEL  ; 前下料伺服自动加速比率
D2221 CHANNEL  ; 前下料伺服自动减速比率
D2222 CHANNEL  ; 前下料伺服自动速度与上料相同
D2223 CHANNEL  ; 前下料伺服自动速度
D2224 CHANNEL  ; 前下料伺服自动输出脉冲
D2225 CHANNEL  ; 前下料伺服自动输出脉冲
D2226 CHANNEL  ; 前下料伺服自动启动速度
D2227 CHANNEL  ; 前下料伺服自动启动速度
D2230 CHANNEL  ; 前下料伺服待机位置
D2231 CHANNEL  ; 前下料伺服待机位置
D2232 CHANNEL  ; 前下料伺服仓1取料位
D2233 CHANNEL  ; 前下料伺服仓1取料位
D2234 CHANNEL  ; 前下料伺服仓2取料位
D2235 CHANNEL  ; 前下料伺服仓2取料位
D2236 CHANNEL  ; 前下料伺服放料位
D2237 CHANNEL  ; 前下料伺服OK放料位
D2238 CHANNEL  ; 前下料伺服NG放料位
D2239 CHANNEL  ; 前下料伺服NG放料位
D2300 CHANNEL  ; 后上料伺服手动低速加速比率
D2301 CHANNEL  ; 后上料伺服手动低速减速比率
D2302 CHANNEL  ; 后上料伺服手动低速速度
D2303 CHANNEL  ; 后上料伺服手动低速速度
D2304 CHANNEL  ; 后上料伺服手动输出脉冲
D2305 CHANNEL  ; 后上料伺服手动输出脉冲
D2306 CHANNEL  ; 后上料伺服手动启动速度
D2307 CHANNEL  ; 后上料伺服手动启动速度
D2308 CHANNEL  ; 后上料伺服手动当前速度
D2309 CHANNEL  ; 后上料伺服手动当前速度
D2310 CHANNEL  ; 后上料伺服手动高速加速比率
D2311 CHANNEL  ; 后上料伺服手动高速减速比率
D2312 CHANNEL  ; 后上料伺服手动高速速度
D2313 CHANNEL  ; 后上料伺服手动高速速度
D2314 CHANNEL  ; 后上料伺服手动高速输出脉冲
D2315 CHANNEL  ; 后上料伺服手动高速输出脉冲
D2316 CHANNEL  ; 后上料伺服手动高速启动速度
D2317 CHANNEL  ; 后上料伺服手动高速启动速度
D2318 CHANNEL  ; 后上料伺服寸动距离
D2319 CHANNEL  ; 后上料伺服寸动距离
D2320 CHANNEL  ; 后上料伺服自动加速比率
D2321 CHANNEL  ; 后上料伺服自动减速比率
D2322 CHANNEL  ; 后上料伺服自动速度
D2323 CHANNEL  ; 后上料伺服自动速度
D2324 CHANNEL  ; 后上料伺服自动输出脉冲
D2325 CHANNEL  ; 后上料伺服自动输出脉冲
D2326 CHANNEL  ; 后上料伺服自动启动速度
D2327 CHANNEL  ; 后上料伺服自动启动速度
D2330 CHANNEL  ; 后上料伺服待机位置
D2331 CHANNEL  ; 后上料伺服待机位置
D2332 CHANNEL  ; 后上料伺服上料位置
D2333 CHANNEL  ; 后上料伺服上料位置
D2334 CHANNEL  ; 后上料伺服仓3放料位
D2335 CHANNEL  ; 后上料伺服仓3放料位
D2336 CHANNEL  ; 后上料伺服仓4放料位
D2337 CHANNEL  ; 后上料伺服仓4放料位
D240 CHANNEL  ; 接收检漏仪状态起始字
D2400 CHANNEL  ; 后下料伺服手动低速加速比率
D2401 CHANNEL  ; 后下料伺服手动低速减速比率
D2402 CHANNEL  ; 后下料伺服手动低速速度
D2403 CHANNEL  ; 后下料伺服手动低速速度
D2404 CHANNEL  ; 后下料伺服手动输出脉冲
D2405 CHANNEL  ; 后下料伺服手动输出脉冲
D2406 CHANNEL  ; 后下料伺服手动启动速度
D2407 CHANNEL  ; 后下料伺服手动启动速度
D2408 CHANNEL  ; 后下料伺服手动当前速度
D2409 CHANNEL  ; 后下料伺服手动当前速度
D241 CHANNEL  ; 接收检漏仪状态起始字(ASCII)
D2410 CHANNEL  ; 后下料伺服手动高速加速比率
D2411 CHANNEL  ; 后下料伺服手动高速减速比率
D2412 CHANNEL  ; 后下料伺服手动高速速度
D2413 CHANNEL  ; 后下料伺服手动高速速度
D2414 CHANNEL  ; 后下料伺服手动高速输出脉冲
D2415 CHANNEL  ; 后下料伺服手动高速输出脉冲
D2416 CHANNEL  ; 后下料伺服手动高速启动速度
D2417 CHANNEL  ; 后下料伺服手动高速启动速度
D2418 CHANNEL  ; 后下料伺服寸动距离
D2419 CHANNEL  ; 后下料伺服寸动距离
D2420 CHANNEL  ; 后下料伺服自动加速比率
D2421 CHANNEL  ; 后下料伺服自动减速比率
D2422 CHANNEL  ; 后下料伺服自动速度
D2423 CHANNEL  ; 后下料伺服自动速度
D2424 CHANNEL  ; 后下料伺服自动输出脉冲
D2425 CHANNEL  ; 后下料伺服自动输出脉冲
D2426 CHANNEL  ; 后下料伺服自动启动速度
D2427 CHANNEL  ; 后下料伺服自动启动速度
D2430 CHANNEL  ; 后下料伺服待机位置
D2431 CHANNEL  ; 后下料伺服待机位置
D2432 CHANNEL  ; 后下料伺服仓3取料位
D2433 CHANNEL  ; 后下料伺服仓3取料位
D2434 CHANNEL  ; 后下料伺服仓4取料位
D2435 CHANNEL  ; 后下料伺服仓4取料位
D2436 CHANNEL  ; 后下料伺服OK放料位
D2437 CHANNEL  ; 后下料伺服OK放料位
D2438 CHANNEL  ; 后下料伺服NG放料位
D2439 CHANNEL  ; 后下料伺服NG放料位
D2440 CHANNEL  ; 下料2#NG放料位
D2442 CHANNEL  ; 下料3#NG放料位
D2444 CHANNEL  ; 下料4#NG放料位
D250 CHANNEL  ; 接收检漏口压力的起始字
D2500 CHANNEL  ; 进料升降伺服当前位置
D2504 CHANNEL  ; 进料升降伺服手动低速速度
D2506 CHANNEL  ; 进料升降伺服自动加速时间
D251 CHANNEL  ; 接收检漏口压力(ASCII)
D2510 CHANNEL  ; 进料升降伺服到取料位
D2512 CHANNEL  ; 进料伺服取放料高中
D2514 CHANNEL  ; 进料升降伺服放料位
D2520 CHANNEL  ; 升降伺到取料位
D260 CHANNEL  ; 接收漏率起始字
D2600 CHANNEL  ; 进料升降手动低速加速时间
D2602 CHANNEL  ; 进料升降手动低速减速时间
D261 CHANNEL  ; 接收的漏率(ASCII)
D2620 CHANNEL  ; 进料升降伺服自动加速时间
D2622 CHANNEL  ; 进料升降伺服自动减速时间
D2700 CHANNEL  ; 出料升降伺服当前位置
D2704 CHANNEL  ; 出料升降伺服手动低速速度
D2706 CHANNEL  ; 出料升降自动速度
D2710 CHANNEL  ; 出料升降伺服取料高度
D2712 CHANNEL  ; 出为料升降伺服放料高度
D2720 CHANNEL  ; 出料升降伺服定位位置
D2800 CHANNEL  ; 出料升降伺服手动低速加速时间
D2802 CHANNEL  ; 出料升降伺服手动低速减速时间
D2820 CHANNEL  ; 出料升降伺服自动加速时间
D2822 CHANNEL  ; 出料升降伺服自动减速时间
D2900 CHANNEL  ; 出料伺服手动低速加速时间
D2901 CHANNEL  ; 出料伺服手动低速加速时间
D2902 CHANNEL  ; 出料伺服手动低速减速时间
D2903 CHANNEL  ; 出料伺服手动低速减速时间
D2904 CHANNEL  ; 出料伺服手动低速速度
D2905 CHANNEL  ; 出料伺服手动低速速度
D2906 CHANNEL  ; 出料伺服手动低速输出脉冲
D2907 CHANNEL  ; 出料伺服手动低速输出脉冲
D2908 CHANNEL  ; 出料伺服手动当前速度
D2909 CHANNEL  ; 出料伺服手动当前速度
D2910 CHANNEL  ; 出料伺服手动高速加速时间
D2911 CHANNEL  ; 出料伺服手动高速加速时间
D2912 CHANNEL  ; 出料伺服手动高速减速时间
D2913 CHANNEL  ; 出料伺服手动高速减速时间
D2914 CHANNEL  ; 出料伺服手动高速速度
D2915 CHANNEL  ; 出料伺服手动高速速度
D2916 CHANNEL  ; 出料伺服手动高速输出脉冲
D2917 CHANNEL  ; 出料伺服手动高速输出脉冲
D2918 CHANNEL  ; 出料伺服寸动距离
D2919 CHANNEL  ; 出料伺服寸动距离
D2920 CHANNEL  ; 出料伺服自动加速时间
D2921 CHANNEL  ; 出料伺服自动加速时间
D2922 CHANNEL  ; 出料伺服自动减速时间
D2923 CHANNEL  ; 出料伺服自动减速时间
D2924 CHANNEL  ; 出料伺服自动速度
D2925 CHANNEL  ; 出料伺服自动速度
D2926 CHANNEL  ; 出料伺服自动输出脉冲
D2927 CHANNEL  ; 出料伺服自动输出脉冲
D2928 CHANNEL  ; 出料伺服自动速度2(低速)
D2930 CHANNEL  ; 出料伺服待机位置
D2931 CHANNEL  ; 出料伺服待机位置
D2932 CHANNEL  ; 出料伺服前取料位置
D2933 CHANNEL  ; 出料伺服前取料位置
D2934 CHANNEL  ; 出料伺服后取料位置
D2935 CHANNEL  ; 出料伺服后取料位置
D2936 CHANNEL  ; 出料轴出料位
D2937 CHANNEL  ; 出料伺服放料位
D2938 CHANNEL  ; 出料伺服#1NG测试位置
D2940 CHANNEL  ; 出料伺服#2NG测试位
D2942 CHANNEL  ; 出料伺服#3NG位
D2944 CHANNEL  ; 出料伺服#4NG位
D2980 CHANNEL  ; 前出料转盘前直径边缘位置
D2982 CHANNEL  ; 前出料转盘后直径边缘位置
D2984 CHANNEL  ; 后出料转盘前直径边缘位置
D2986 CHANNEL  ; 后出料转盘后直径边缘位置
D30 CHANNEL  ; #1腔体状态(停用，待料中，测试中，测试完成
D300 CHANNEL  ; #1腔体检漏口压力(浮点)
D3000 CHANNEL  ; 进料水平伺服当前位置
D3010 CHANNEL  ; 间隔气缸下降条件
D302 CHANNEL  ; #1腔体清氦氦检完成时检漏口压力(浮点)
D3030 CHANNEL  ; 进料伺服自动定位位置
D310 CHANNEL  ; #2腔体检漏口压力(浮点)
D3100 CHANNEL  ; 前腔体上料伺服当前位置
D312 CHANNEL  ; #2腔体清氦氦检完成时检漏口压力(浮点)
D3120 CHANNEL  ; 前上料伺服当前定位位置(M)
D3130 CHANNEL  ; 前上料伺服自动定位位置
D3140 CHANNEL  ; 腔体1检测有料开始位置
D3142 CHANNEL  ; 腔体1检测最后位置
D3144 CHANNEL  ; 腔体2检测有料开始位置
D3146 CHANNEL  ; 腔体2检测结束位
D32 CHANNEL  ; #2腔体状态(停用，待料中，测试中，测试完成
D320 CHANNEL  ; #3腔体检漏口压力(浮点)
D3200 CHANNEL  ; 前下料伺服当前位置
D322 CHANNEL  ; #3腔体清氦氦检完成时检漏口压力(浮点)
D3220 CHANNEL  ; 前下料伺服当前定位位置(M)
D3230 CHANNEL  ; 前下料伺服自动定位位置
D330 CHANNEL  ; #4腔体检漏口压力(浮点)
D3300 CHANNEL  ; 后腔体上料伺服当前位置
D332 CHANNEL  ; #4腔体清氦氦检完成时检漏口压力(浮点)
D3320 CHANNEL  ; 后上料伺服当前定位位置(M)
D3330 CHANNEL  ; 后上料伺服自动定位位置
D3340 CHANNEL  ; 腔体3检测有料开始位置
D3342 CHANNEL  ; 腔体3检测最后位置
D3344 CHANNEL  ; 腔体4检测有料开始位置
D3346 CHANNEL  ; 腔体4检测最后位置
D34 CHANNEL  ; #3腔体状态(停用，待料中，测试中，测试完成
D3400 CHANNEL  ; 后下料伺服当前位置
D3420 CHANNEL  ; 后下料伺服当前定位位置(M)
D3430 CHANNEL  ; 后下料伺服自动定位位置
D36 CHANNEL  ; #4腔体状态(停用，待料中，测试中，测试完成
D370 CHANNEL  ; 氦检仪就绪状态
D3900 CHANNEL  ; 出料移载伺服当前位置
D3920 CHANNEL  ; 出料伺服当前定位位置(M)
D3930 CHANNEL  ; 出料伺服自动定位位置
D40 CHANNEL  ; 腔体真空达到阀值
D400 CHANNEL  ; #1腔体漏率(浮点)
D4000 CHANNEL  ; 真空值1转存
D4002 CHANNEL  ; #1真空值运算1
D4004 CHANNEL  ; #1真空值运算2
D4006 CHANNEL  ; #1真空值运算3
D4008 CHANNEL  ; #1真空值运算4
D4010 CHANNEL  ; 腔体1实际真空值(浮点)
D402 CHANNEL  ; #1腔体清氦氦检完成时漏率(浮点)
D4020 CHANNEL  ; 真空值2转存
D4022 CHANNEL  ; #2真空值运算1
D4024 CHANNEL  ; #2真空值运算2
D4026 CHANNEL  ; #2真空值运算3
D4028 CHANNEL  ; #2真空值运算4
D4030 CHANNEL  ; 腔体2实际真空值(浮点)
D4040 CHANNEL  ; 真空值3转存
D4042 CHANNEL  ; #3真空值运算1
D4044 CHANNEL  ; #3真空值运算2
D4046 CHANNEL  ; #3真空值运算3
D4048 CHANNEL  ; #3真空值运算4
D4050 CHANNEL  ; 腔体3实际真空值(浮点)
D4060 CHANNEL  ; 真空3转存
D4062 CHANNEL  ; #4真空值运算1
D4064 CHANNEL  ; #4真空值运算2
D4066 CHANNEL  ; #4真空值运算3
D4068 CHANNEL  ; #4真空值运算4
D4070 CHANNEL  ; 腔体4实际真空值(浮点)
D410 CHANNEL  ; #2腔体漏率(浮点)
D4100 CHANNEL  ; #1电池真空压力表模拟量读数
D4104 CHANNEL  ; #1电池真空压力表读数(浮点)
D4108 CHANNEL  ; #1电池真空压力表计算一
D4110 CHANNEL  ; 氦检开启时腔体实际压力
D4112 CHANNEL  ; #1电池真空压力表计算二
D4116 CHANNEL  ; #1电池真空压力表读数(#1电池真空)
D412 CHANNEL  ; #2腔体清氦氦检完成时漏率(浮点)
D4120 CHANNEL  ; #2电池真空压力表模拟量读数
D4124 CHANNEL  ; #2电池真空压力表读数(浮点)
D4128 CHANNEL  ; #2电池真空压力表计算一
D4132 CHANNEL  ; #2电池真空压力表计算二
D4136 CHANNEL  ; #2电池真空压力表读数
D4140 CHANNEL  ; #3电池真空压力表模拟量读数
D4144 CHANNEL  ; #3电池真空压力表模拟量读数(浮点)
D4148 CHANNEL  ; #3电池真空压力表计算一
D4152 CHANNEL  ; #3电池真空压力表计算二
D4156 CHANNEL  ; #3电池真空压力表读数
D4160 CHANNEL  ; #4电池真空压力表模拟量读数
D4164 CHANNEL  ; #4电池真空压力表模拟量读数(浮点)
D4168 CHANNEL  ; #4电池真空压力表计算一
D4172 CHANNEL  ; #4电池真空压力表计算二
D4176 CHANNEL  ; #4电池真空压力表读数(实际真空值)
D4180 CHANNEL  ; 1#电池真空压力修正系数
D4182 CHANNEL  ; 2#电池真空压力修正系数
D4184 CHANNEL  ; 3#电池真空压力修正系数
D4186 CHANNEL  ; 4#电池真空压力修正系数
D4188 CHANNEL  ; 压力系数5
D42 CHANNEL  ; 腔体抽气时间
D420 CHANNEL  ; #3腔体漏率(浮点)
D4200 CHANNEL  ; #1密封气缸压力表读数(模拟量)
D4204 CHANNEL  ; 1#密封气缸压力表模拟量读数(浮点)
D4216 CHANNEL  ; 1#密封气缸压力表读数(实际压力值)
D422 CHANNEL  ; #3腔体清氦氦检完成时漏率(浮点)
D4220 CHANNEL  ; 2#密封气缸压力表读数(模拟量)
D4224 CHANNEL  ; 2#密封气缸压力表模拟量读数(浮点)
D4236 CHANNEL  ; 2#密封气缸压力表读数(实际压力值)
D4240 CHANNEL  ; 3#密封气缸压力表读数(模拟量)
D4244 CHANNEL  ; 3#密封气缸压力表模拟量读数(浮点)
D4256 CHANNEL  ; 3#密封气缸压力表读数(实际压力值)
D4260 CHANNEL  ; 4#密封气缸压力表读数(模拟量)
D4264 CHANNEL  ; 4#密封气缸压力表模拟量读数(浮点)
D4276 CHANNEL  ; 4#密封气缸压力表读数(实际压力值)
D430 CHANNEL  ; #4腔体漏率(浮点)
D4300 CHANNEL  ; #1腔体保压前真空值
D4304 CHANNEL  ; #1腔体保压后真空值
D4308 CHANNEL  ; #1腔体泄漏量
D432 CHANNEL  ; #4腔体清氦氦检完成时漏率(浮点)
D4320 CHANNEL  ; #2腔体保压前真空
D4324 CHANNEL  ; #2腔体保压后真空
D4328 CHANNEL  ; #2腔体泄漏量
D4340 CHANNEL  ; #3腔体保压前真空
D4344 CHANNEL  ; #3腔体保压后真空
D4348 CHANNEL  ; #3腔体泄漏量
D4360 CHANNEL  ; #4腔体保压前真空
D4364 CHANNEL  ; #4腔体保压后真空
D4368 CHANNEL  ; #4腔体泄漏量
D450 CHANNEL  ; 氦检仪当前实时漏率
D46 CHANNEL  ; 氦检设定时间
D4900 CHANNEL  ; 扫码位暂存码1
D4910 CHANNEL  ; 取料位条码
D50 CHANNEL  ; #1腔体正常抽气时间
D500 CHANNEL  ; 检漏压力
D5000 CHANNEL  ; 扫码1长度
D5001 CHANNEL  ; #1条码
D5020 CHANNEL  ; 条码1在进料爪子
D5060 CHANNEL  ; 条码2在进料爪子
D51 CHANNEL  ; #1电池正常抽气时间
D510 CHANNEL  ; 检漏口压力 浮点
D5100 CHANNEL  ; 在前进料托盘
D5120 CHANNEL  ; 在前上料爪子
D5140 CHANNEL  ; 条码在仓1
D5160 CHANNEL  ; 条码1在仓2
D5180 CHANNEL  ; 条码1在前下料爪子
D52 CHANNEL  ; #2腔体正常抽气时间
D520 CHANNEL  ; 检漏口压力最小值
D5200 CHANNEL  ; 在前进料托盘
D5220 CHANNEL  ; 在前上料爪子
D5240 CHANNEL  ; 条码在仓1
D5260 CHANNEL  ; 条码2在仓2
D5280 CHANNEL  ; 条码2在前下料爪子
D53 CHANNEL  ; #2电池正常抽气时间
D5300 CHANNEL  ; NG位1#条码
D5320 CHANNEL  ; 条码在前出料托盘
D5360 CHANNEL  ; 出料爪上1#条码
D54 CHANNEL  ; #3腔体正常抽气时间
D5400 CHANNEL  ; NG位2#条码
D5420 CHANNEL  ; 条码在前出料托盘
D5460 CHANNEL  ; 出料爪上2#条码
D55 CHANNEL  ; #3电池正常抽气时间
D5510 CHANNEL  ; #1腔检漏口压力
D5512 CHANNEL  ; #1、2腔检漏口压力在前出料托盘
D5516 CHANNEL  ; #1、2腔压力在出料爪子
D5520 CHANNEL  ; #2腔检漏口压力在前下料夹爪
D5530 CHANNEL  ; 腔检漏口压力在NG
D5540 CHANNEL  ; #1/2腔注氦后压力(kPa)(前NG位)
D5550 CHANNEL  ; 前NG位测试结果
D56 CHANNEL  ; #4腔体正常抽气时间
D5610 CHANNEL  ; #1腔体漏率
D5612 CHANNEL  ; 1、2腔体漏率在前出料托盘
D5616 CHANNEL  ; 1、2腔体漏率在出料爪子
D5620 CHANNEL  ; #2腔漏率在前下料夹爪
D5630 CHANNEL  ; 1#腔充氦压力(kPa)在前下料夹爪
D5632 CHANNEL  ; #1、2腔充氦压力在前出料托盘
D5636 CHANNEL  ; #1、2腔充氦压力在出料夹爪
D5640 CHANNEL  ; 腔体漏率
D5650 CHANNEL  ; 1#腔测试结果在前下料夹爪
D5652 CHANNEL  ; #1、2腔测试结果在前出料托盘
D5656 CHANNEL  ; #1、2腔测试结果在出料夹爪
D5660 CHANNEL  ; 2#腔充氦压力(kPa)在前下料夹爪
D5670 CHANNEL  ; 2#腔测试结果在前下料夹爪
D57 CHANNEL  ; #4电池正常抽气时间
D5800 CHANNEL  ; 数据上传位电池的检漏口压力
D5802 CHANNEL  ; 后下料机械手检漏口压力
D5804 CHANNEL  ; 检漏口压在出料托盘
D5900 CHANNEL  ; 数据上传位电池的漏率
D5902 CHANNEL  ; 后下料机械手漏率
D5904 CHANNEL  ; 漏率在出料托盘
D5910 CHANNEL  ; 数据上传位电池充氦压力
D5912 CHANNEL  ; 后下料机械手充氦压力
D5914 CHANNEL  ; 充氦压力在出料托盘
D5920 CHANNEL  ; 数据上传位电池测试结果
D5922 CHANNEL  ; 后下料机械手电池测试结果
D5924 CHANNEL  ; 测试结果在出料托盘
D5930 CHANNEL  ; 前下料机械手电池腔体位置
D5932 CHANNEL  ; 后下料机械手电池腔体位置
D5934 CHANNEL  ; 腔体位置到出料托盘
D60 CHANNEL  ; 接收条码数据字长度
D600 CHANNEL  ; 氦检下限位值
D6000 CHANNEL  ; 设备OEE状态(0-待机,10-正常,70-故障)
D6003.05 BOOL  ; 300A_0_2St TR_Down
D602 CHANNEL  ; 氦检上限位值
D6110 CHANNEL  ; 流入个数
D6204 CHANNEL  ; #1腔体测试完成时的检漏口压力
D6206 CHANNEL  ; #1腔体测试完成时漏率
D6214 CHANNEL  ; #2腔体测试完成时的检漏口压力
D6216 CHANNEL  ; #2腔体测试完成时漏率
D6224 CHANNEL  ; #3腔体测试完成时检漏口压力
D6226 CHANNEL  ; #3腔体测试完成时漏率
D6234 CHANNEL  ; #4腔体测试完成时检漏口压力
D6236 CHANNEL  ; #4腔体测试完成时漏率
D651 CHANNEL  ; 报警时检漏口压力
D66 CHANNEL  ; 设定条码长度
D670 CHANNEL  ; 报警时检漏口压力
D68 CHANNEL  ; 设定条码字长度
D700 CHANNEL  ; 氦检设定时间(储存)
D7000 CHANNEL  ; 扫码2长度
D7001 CHANNEL  ; #2条码
D702 CHANNEL  ; 检漏口压力设定值小数部分(储存)
D704 CHANNEL  ; 检漏口压力设定值指数(储存)
D706 CHANNEL  ; 漏率设定值小数部分(储存)
D708 CHANNEL  ; 漏率设定值指数(储存)
D7100 CHANNEL  ; 在后进料托盘
D7120 CHANNEL  ; 在后上料爪子
D7140 CHANNEL  ; 条码在仓3
D7160 CHANNEL  ; 条码在仓4
D7180 CHANNEL  ; 条码在后下料爪子
D720 CHANNEL  ; 设备状态
D7200 CHANNEL  ; 在后进料托盘
D721 CHANNEL  ; 设备状态(储存)
D722 CHANNEL  ; 设备状态变更
D7220 CHANNEL  ; 在后上料爪子
D7240 CHANNEL  ; 条码在仓3
D7260 CHANNEL  ; 条码在仓4
D7280 CHANNEL  ; 条码在后下料爪子
D730 CHANNEL  ; 早班分、秒
D7300 CHANNEL  ; 条码在NG
D731 CHANNEL  ; 早班日、时
D7320 CHANNEL  ; 条码在后出料托盘
D733 CHANNEL  ; 晚班分、秒
D734 CHANNEL  ; 晚班日、时
D736 CHANNEL  ; 只比较时、分、秒
D7360 CHANNEL  ; 条码在出料爪
D740 CHANNEL  ; 单班生产时间
D7400 CHANNEL  ; 条码在NG
D742 CHANNEL  ; 单班故障时间
D7420 CHANNEL  ; 条码在后出料托盘
D7460 CHANNEL  ; 条码在出料爪
D7510 CHANNEL  ; #3腔检漏口压力在后下料夹爪
D7512 CHANNEL  ; #3、4腔检漏口压力在后托盘
D7516 CHANNEL  ; 出料夹爪上电池的检漏口压力
D7520 CHANNEL  ; #4检漏口压力
D7530 CHANNEL  ; #3、4腔检漏口压力在后NG位
D7540 CHANNEL  ; 后NG位注氦后压力(kPa）
D7550 CHANNEL  ; 后NG位结果类型
D7610 CHANNEL  ; #3腔体漏率在后下料夹爪
D7612 CHANNEL  ; #3、4腔体漏率在后托盘
D7616 CHANNEL  ; 出料夹爪上电池的漏率
D7620 CHANNEL  ; #4腔体漏率
D7630 CHANNEL  ; #3腔体充氦压力在后下料夹爪
D7632 CHANNEL  ; #3/4腔体充氦压力在后出料托盘
D7636 CHANNEL  ; #3/4腔体充氦压力在出料夹爪
D7640 CHANNEL  ; #3、4腔漏率在后NG位
D7650 CHANNEL  ; #3腔体测试结果在后下料夹爪
D7652 CHANNEL  ; #3/4腔体测试结果在后出料托盘
D7656 CHANNEL  ; #3/4腔体测试结果在出料夹爪
D7660 CHANNEL  ; #4腔体充氦压力在后下料夹爪
D7670 CHANNEL  ; #4腔体测试结果在后下料夹爪
D7800 CHANNEL  ; 数据上传位1#条码
D7820 CHANNEL  ; 条码在后下料爪子
D7840 CHANNEL  ; 条码在出料托盘
D7900 CHANNEL  ; 数据上传位2#条码
D800 CHANNEL  ; 扫码步
D8000 CHANNEL  ; 检漏状态第一字节
D8001 CHANNEL  ; 检漏状态第二字节
D8002 CHANNEL  ; 检漏状态结束字节
D8010 CHANNEL  ; 待机状态第一字节
D8011 CHANNEL  ; 待机状态第二字节
D8012 CHANNEL  ; 待机状态结束字节
D802 CHANNEL  ; 进料顺控编号
D8020 CHANNEL  ; 定标状态第一字节
D8021 CHANNEL  ; 定标状态第二字节
D8022 CHANNEL  ; 定标状态结束字节
D8030 CHANNEL  ; 启动状态第一字节
D8031 CHANNEL  ; 启动状态第二字节
D8032 CHANNEL  ; 启动状态结束字节
D804 CHANNEL  ; 检漏口压力底数(储存)
D8040 CHANNEL  ; 错误状态第一字节
D8041 CHANNEL  ; 错误状态第二字节
D8042 CHANNEL  ; 错误状态结束字节
D8050 CHANNEL  ; 暂停状态第一字节
D8051 CHANNEL  ; 暂停状态第二字节
D8052 CHANNEL  ; 暂停状态结束字节
D806 CHANNEL  ; 漏率指数
D808 CHANNEL  ; 漏率底数
D8100 CHANNEL  ; 氦检仪状态(1-检漏,2-待机,3-启动,4-定标,5-错误,6-暂停)
D82 CHANNEL  ; #1冲氦压力
D820 CHANNEL  ; 设备状态
D821 CHANNEL  ; 设备状态(储存)
D822 CHANNEL  ; 设备状态变更
D830 CHANNEL  ; 早班分、秒
D8300 CHANNEL  ; #1条码状态 0-EMS已读取 <>0 触发扫码
D8302 CHANNEL  ; 校验结果（1-OK，2-NG）
D831 CHANNEL  ; 早班日、时
D833 CHANNEL  ; 晚班分、秒
D834 CHANNEL  ; 晚班日、时
D836 CHANNEL  ; 只比较时、分、秒
D838 CHANNEL  ; 晚班传输信号
D84 CHANNEL  ; #2冲氦压力
D840 CHANNEL  ; 单班生产时间
D8400 CHANNEL  ; 读氦检仪报警
D842 CHANNEL  ; 单班故障时间
D8500 CHANNEL  ; 读氦检仪内部校准状态
D86 CHANNEL  ; #3冲氦压力
D8600 CHANNEL  ; 氦检校准暂存状态1-完成
D8601 CHANNEL  ; 氦检校准暂存状态1-完成
D8610 CHANNEL  ; 氦检校准暂存状态2-通过
D8611 CHANNEL  ; 氦检校准暂存状态2-通过
D8612 CHANNEL  ; 氦检校准暂存状态3
D8620 CHANNEL  ; 氦检校准暂存状态3-进行
D8621 CHANNEL  ; 氦检校准暂存状态3-进行
D8622 CHANNEL  ; 氦检校准暂存状态3-进行
D870 CHANNEL  ; 早班分、秒
D88 CHANNEL  ; #4冲氦压力
D90 CHANNEL  ; #1腔体手动抽气时间
D9000 CHANNEL  ; PC通信标志
D9003 CHANNEL  ; PC交互
D91 CHANNEL  ; #1腔体保压前时间
D910 CHANNEL  ; 连续NG次数
D9100 CHANNEL  ; PC返回MES校验结果 1-0K 2-NG
D9101 CHANNEL  ; #1腔体数据处理完成
D9102 CHANNEL  ; #2腔体数据处理完成
D9103 CHANNEL  ; #3腔体数据处理完成
D9104 CHANNEL  ; #4腔体数据处理完成
D9105 CHANNEL  ; #1腔体NG数据处理完成
D9106 CHANNEL  ; #2腔体NG数据处理完成
D9107 CHANNEL  ; #3腔体NG数据处理完成
D9108 CHANNEL  ; #4腔体NG数据处理完成
D9110 CHANNEL  ; PC已接收到更新后参数标志
D912 CHANNEL  ; 测试连续NG三个
D92 CHANNEL  ; #1腔体保压时间
D9200 CHANNEL  ; 错误码
D93 CHANNEL  ; #2腔体自检抽气时间
D9300 CHANNEL  ; 前下料机械手放料
D9302 CHANNEL  ; 后下料机械手放料
D94 CHANNEL  ; #2腔体进入保压前时间
D95 CHANNEL  ; #2腔体保压时间
D9590 CHANNEL  ; 前下料机械手条码
D96 CHANNEL  ; #3腔体自检抽气时间
D9600 CHANNEL  ; 条码在前下料爪子
D9612 CHANNEL  ; 前下料机械手漏率
D9614 CHANNEL  ; 检漏口压力在前下料爪
D9616 CHANNEL  ; 前下料爪电池腔体位置
D9618 CHANNEL  ; 前下料爪电池充氦压力
D9620 CHANNEL  ; 前下料爪电池测试结果
D9622 CHANNEL  ; 前下料爪氦检打开时腔体真空实际值（浮点PC）
D9624 CHANNEL  ; 前下料爪充氦时电池真空实际值（浮点PC）
D9630 CHANNEL  ; 漏率设定值(浮点数Pa.m3)
D9632 CHANNEL  ; 检漏口压力设定值
D9634 CHANNEL  ; 氦检时间（浮点）
D9636 CHANNEL  ; 注氦后压力
D9638 CHANNEL  ; 腔体真空阀值(浮点pc)
D9640 CHANNEL  ; 电池抽真空阀值(浮点pc)
D9690 CHANNEL  ; 条码在后下料爪子
D97 CHANNEL  ; #3腔体自保前时间
D9712 CHANNEL  ; 后下料机械手漏率
D9714 CHANNEL  ; 检漏口压力在后下料爪
D9716 CHANNEL  ; 后下料爪电池腔体位置
D9718 CHANNEL  ; 后下料爪电池充氦压力
D9720 CHANNEL  ; 后下料爪电池测试结果
D9722 CHANNEL  ; 后下料爪氦检打开时腔体真空实际值（浮点PC）
D9724 CHANNEL  ; 后下料爪充氦时电池真空实际值（浮点PC）
D98 CHANNEL  ; #3腔体自保时间
D99 CHANNEL  ; #4腔体自检抽气时间
H0.00 BOOL  ; 手动模式
H0.01 BOOL  ; 自动模式
H100.02 BOOL  ; 错误模拟
H10.06 BOOL  ; 上料托盘有料
H11.00 BOOL  ; 进料夹爪夹紧
H11.01 BOOL  ; 前上料夹爪夹紧
H11.02 BOOL  ; 前下料夹爪夹紧
H11.03 BOOL  ; 后上料夹爪夹紧
H11.04 BOOL  ; 后下料夹爪夹紧
H11.05 BOOL  ; 出料爪子夹紧
H11.09 BOOL  ; 出料夹爪夹紧
H12.00 BOOL  ; 进料伺服归零完成
H12.01 BOOL  ; 前上料伺服归零完成
H12.02 BOOL  ; 前下料伺服归零完成
H12.03 BOOL  ; 后上料伺服归零完成
H12.04 BOOL  ; 后下料伺服归零完成
H12.09 BOOL  ; 出料移栽伺服归零完成
H13.01 BOOL  ; 1腔料
H13.02 BOOL  ; 2腔料
H13.03 BOOL  ; 1腔OK在前托盘
H13.04 BOOL  ; 2腔OK在前托盘
H13.05 BOOL  ; 1腔OK在出料爪子
H13.06 BOOL  ; 2腔OK在出料爪子
H13.11 BOOL  ; 读1腔数据
H13.12 BOOL  ; 读2腔数据
H13.13 BOOL  ; 1腔NG
H13.14 BOOL  ; 2腔NG
H14.01 BOOL  ; 3腔料
H14.02 BOOL  ; 4腔料
H14.03 BOOL  ; 3腔OK在后托盘
H14.04 BOOL  ; 4腔OK在后托盘
H14.05 BOOL  ; 3腔OK在出料爪子
H14.06 BOOL  ; 4腔OK在出料爪子
H14.11 BOOL  ; 读3腔数据
H14.12 BOOL  ; 读4腔数据
H14.13 BOOL  ; 3腔NG
H14.14 BOOL  ; 4腔NG
H16.00 BOOL  ; 氦检启动
H17.00 BOOL  ; 白班传送完标志
H17.01 BOOL  ; 晚班传送完标志
H1.00 BOOL  ; 进料移载伺服手动高速
H1.01 BOOL  ; 前上料伺服手动高速
H1.02 BOOL  ; 前下料伺服手动高速
H1.03 BOOL  ; 后上料伺服手动高速
H1.04 BOOL  ; 后下料伺服手动高速
H1.09 BOOL  ; 出料伺服手动高速
H1.10 BOOL  ; 自动重扫码
H20.00 BOOL  ; 检测NG
H21.00 BOOL  ; #1模组放料完成
H21.01 BOOL  ; #1模组测试中
H21.02 BOOL  ; #1模组测试完成
H21.03 BOOL  ; #1模组取料完成
H21.04 BOOL  ; #1模组测试NG
H21.06 BOOL  ; #1模组有料
H21.07 BOOL  ; #1模组电池MES NG记忆
H21.08 BOOL  ; 腔体1有料
H21.09 BOOL  ; #1模组需要清氦
H21.10 BOOL  ; #1模组清氦中
H21.11 BOOL  ; #1模组清氦完成
H21.12 BOOL  ; #1模组清氦OK
H21.14 BOOL  ; #1模组自动运行中
H21.15 BOOL  ; #1模组工作完成记忆
H22.00 BOOL  ; #2模组放料完成
H22.01 BOOL  ; #2模组测试中
H22.02 BOOL  ; #2模组测试完成
H22.03 BOOL  ; #2模组取料完成
H22.04 BOOL  ; #2模组测试NG
H22.06 BOOL  ; #2模组有料
H22.07 BOOL  ; #2模组电池MES NG记忆
H22.08 BOOL  ; 腔体2有料
H22.09 BOOL  ; #2模组需要清氦
H22.10 BOOL  ; #2模组清氦中
H22.11 BOOL  ; #2模组清氦完成
H22.12 BOOL  ; #2模组清氦OK
H22.14 BOOL  ; #2模组自动运行中
H22.15 BOOL  ; #2模组工作完成记忆
H23.00 BOOL  ; #3模组放料完成
H23.01 BOOL  ; #3模组测试中
H23.02 BOOL  ; #3模组测试完成
H23.03 BOOL  ; #3模组取料完成
H23.04 BOOL  ; #3模组测试NG
H23.06 BOOL  ; #3模组有电池
H23.07 BOOL  ; #3模组电池MES NG记忆
H23.08 BOOL  ; 腔体3有料
H23.09 BOOL  ; #3模组需要清氦
H23.10 BOOL  ; #3模组清氦中
H23.11 BOOL  ; #3模组清氦完成
H23.12 BOOL  ; #3模组清氦OK
H23.14 BOOL  ; #3模组自动运行中
H23.15 BOOL  ; #3模组工作完成记忆
H24.00 BOOL  ; #4模组放料完成
H24.01 BOOL  ; #4模组测试中
H24.02 BOOL  ; #4模组测试完成
H24.03 BOOL  ; #4模组取料完成
H24.04 BOOL  ; #4模组测试NG
H24.06 BOOL  ; #4模组电池条码NG记忆
H24.07 BOOL  ; #4模组电池MES NG记忆
H24.08 BOOL  ; 腔体4有料
H24.09 BOOL  ; #4模组需要清氦
H24.10 BOOL  ; #4模组清氦中
H24.11 BOOL  ; #4模组清氦完成
H24.12 BOOL  ; #4模组清氦OK
H24.14 BOOL  ; #4模组自动运行中
H24.15 BOOL  ; #4模组工作完成记忆
H25.00 BOOL  ; 出料升降伺服归零完成
H2.01 BOOL  ; 开氦检阀前真空不达标做电池泄漏处理
H2.15 BOOL  ; 连续NG报警 1-启用
H31.00 BOOL  ; 1#电池抽真空完成(A)
H31.01 BOOL  ; 1#电池注氦完成(A)
H31.05 BOOL  ; 1#腔氦检后抽残气完成标志
H31.07 BOOL  ; 1#模组测试已启动
H31.08 BOOL  ; 1#模组抽真空
H32.00 BOOL  ; 2#电池抽真空完成(A)
H32.01 BOOL  ; 2#电池注氦完成(A)
H32.05 BOOL  ; 2#腔氦检后抽残气完成标志
H32.07 BOOL  ; 2#模组测试已启动
H32.08 BOOL  ; 2#模组抽真空
H33.00 BOOL  ; 3#电池抽真空完成(A)
H33.01 BOOL  ; 3#电池注氦完成(A)
H33.05 BOOL  ; 3#腔氦检后抽残气完成标志
H33.07 BOOL  ; 3#模组测试已启动
H33.08 BOOL  ; 3#模组抽真空
H34.00 BOOL  ; 4#电池抽真空完成(A)
H34.01 BOOL  ; 4#电池注氦完成(A)
H34.05 BOOL  ; 4#腔氦检后抽残气完成标志
H34.07 BOOL  ; 4#模组测试已启动
H34.08 BOOL  ; 4#模组抽真空
H35.00 BOOL  ; 进料升降伺服归零完成
H3.00 BOOL  ; #1腔体屏蔽
H3.01 BOOL  ; #2腔体屏蔽
H3.02 BOOL  ; #3腔体屏蔽
H3.03 BOOL  ; #4腔体屏蔽
H3.04 BOOL  ; 扫码屏蔽
H3.05 BOOL  ; 重新扫码模式屏蔽-HMI
H3.06 BOOL  ; 门磁屏蔽-HMI
H3.07 BOOL  ; 电脑屏蔽-HMI
H3.08 BOOL  ; 空跑程序
H3.09 BOOL  ; MES模式屏蔽
H3.10 BOOL  ; 屏蔽腔体电池感应器
H3.11 BOOL  ; 氦检仪屏蔽
H3.12 BOOL  ; 气源压力低报警屏蔽
H3.13 BOOL  ; 扫码NG缓存机构屏蔽
H3.14 BOOL  ; 压力表断线检测功能屏蔽
H3.15 BOOL  ; 拉带对接信号屏蔽
H48.00 BOOL  ; 扫码位扫码OK
H48.01 BOOL  ; 扫码位扫码NG
H48.02 BOOL  ; 上料位条码OK
H48.03 BOOL  ; 上料位条码NG
H48.04 BOOL  ; 条码OK在进料夹爪
H48.05 BOOL  ; 条码NG在进料夹爪
H48.06 BOOL  ; 扫码位有电池扫码已完成
H4.00 BOOL  ; 进料伺服激磁关
H4.01 BOOL  ; 前上料伺服激磁关
H4.02 BOOL  ; 前下料伺服激磁关
H4.03 BOOL  ; 后上料伺服激磁关
H4.04 BOOL  ; 后下料伺服激磁关
H4.05 BOOL  ; 柔性报警屏蔽
H4.06 BOOL  ; GRR测试模式开
H4.07 BOOL  ; 位置修正功能使用(1-使用)
H4.08 BOOL  ; 氦气源压力检测屏蔽
H4.09 BOOL  ; 出料伺服激磁关
H4.10 BOOL  ; 氦检仪屏蔽
H4.11 BOOL  ; 在前后放料位都进行位置修正
H4.12 BOOL  ; 并行注氦模式 关
H4.13 BOOL  ; 空气净化器禁用(1-禁用)
H4.14 BOOL  ; 进站接口屏蔽
H500.01 BOOL  ; 安东通信使用屏蔽
H50.00 BOOL  ; 进料夹爪有料
H50.01 BOOL  ; 进料托盘有料
H50.02 BOOL  ; 后进料旋转位有料记忆
H50.03 BOOL  ; 扫码NG缓存位有料记忆
H50.05 BOOL  ; 上料位有料标志
H50.06 BOOL  ; 电池流出扫码位
H50.07 BOOL  ; 后进料托盘电池MES NG记忆
H50.08 BOOL  ; 扫码完成记忆
H50.09 BOOL  ; 扫码位电池条码NG记忆
H50.10 BOOL  ; 扫码位电池MES NG记忆
H50.11 BOOL  ; 进料夹爪上电池条码NG记忆
H50.12 BOOL  ; 进料夹爪上电池MES NG记忆
H50.13 BOOL  ; 前进料托盘电池条码NG记忆
H50.14 BOOL  ; 前进料托盘电池MES NG记忆
H51.00 BOOL  ; 前上料夹爪有料
H51.06 BOOL  ; 前上料夹爪电池条码NG记忆
H51.07 BOOL  ; 前上料夹爪电池MES NG记忆
H52.00 BOOL  ; 前下料夹爪有电池
H52.01 BOOL  ; 前下料夹爪上电池NG
H52.06 BOOL  ; 前下料夹爪电池条码NG记忆
H52.07 BOOL  ; 前下料夹爪电池MES NG记忆
H53.00 BOOL  ; 后上料夹爪有料
H53.06 BOOL  ; 后上料夹爪电池条码NG记忆
H53.07 BOOL  ; 后上料夹爪电池MES NG记忆
H54.00 BOOL  ; 后下料夹爪有电池
H54.01 BOOL  ; 后下料夹爪上电池NG
H54.06 BOOL  ; 后下料夹爪电池条码NG记忆
H54.07 BOOL  ; 后下料夹爪电池MES NG记忆
H59.00 BOOL  ; 出料夹爪有电池
H59.01 BOOL  ; 前NG拨料位有料
H59.02 BOOL  ; 后NG拨料位有料
H59.03 BOOL  ; 前下料托盘有料
H59.04 BOOL  ; 后下料托盘有料
H59.06 BOOL  ; 前NG槽电池条码NG记忆
H59.07 BOOL  ; 前NG槽电池MES NG记忆
H59.08 BOOL  ; 后NG槽电池条码NG记忆
H59.09 BOOL  ; 后NG槽电池MES NG记忆
H5.00 BOOL  ; 清氦功能使用
H5.01 BOOL  ; 开氦检阀前检查氦检仪数值稳定
H5.02 BOOL  ; 扫码NG料放到前后NG槽
H5.03 BOOL  ; 进料可直接放料时跳过待机位
H5.04 BOOL  ; 充氦压力超规格作NG处理
H5.05 BOOL  ; 四楼LFP设备选择
H5.06 BOOL  ; 氦检阀打开前先开腔体抽气阀
H5.07 BOOL  ; 注氦嘴泄漏NG类型使用
H5.08 BOOL  ; 单工站记忆清除功能使用
H5.09 BOOL  ; MES采集漏率单位为mPa.m3/s(仪器显示值1000倍)
H5.12 BOOL  ; 扫码气缸提前伸出模式使用
H5.13 BOOL  ; 出料放料后直接取料
H5.14 BOOL  ; 出料可放料时直接到放料位
H5.15 BOOL  ; 清氦后进行氦检确认
H60.00 BOOL  ; 扫码OK
H60.01 BOOL  ; 扫码NG料
H60.02 BOOL  ; .
H60.03 BOOL  ; 出料托盘有料
H60.04 BOOL  ; OK料在托盘
H60.05 BOOL  ; NG料在托盘
H60.06 BOOL  ; 托盘有测试NG料
H60.07 BOOL  ; NG处理完成
H60.08 BOOL  ; 扫码NG料处理完成
H60.09 BOOL  ; 2#测试NG有料
H60.10 BOOL  ; 1#扫码NG有料
H60.11 BOOL  ; 2#扫码NG有料
H60.12 BOOL  ; 3#扫码NG有料
H60.13 BOOL  ; 4#扫码NG有料
H60.14 BOOL  ; 3#测试NG有料
H60.15 BOOL  ; 4#测试NG有料
H61.00 BOOL  ; 1#测试NG有料
H61.01 BOOL  ; 1腔OK料
H61.02 BOOL  ; 1腔OK料
H61.03 BOOL  ; 1腔OK在出料爪子
H62.02 BOOL  ; 2腔OK料
H62.03 BOOL  ; 2腔OK在出料爪子
H63.01 BOOL  ; 3腔OK料
H63.02 BOOL  ; 3腔OK料
H63.03 BOOL  ; 3腔OK在出料爪子
H64.01 BOOL  ; 4腔OK料
H64.02 BOOL  ; 4腔OK料
H64.03 BOOL  ; 4腔OK在出料爪子
H6.00 BOOL  ; 左扫码位扫码OK记忆
H6.01 BOOL  ; 左进料上料位条码OK记忆
H6.02 BOOL  ; 左进料夹爪上条码OK记忆
H70.00 BOOL  ; 来料隔离气缸缩回位屏蔽
H70.01 BOOL  ; 来料隔离气缸伸出位屏蔽
H70.02 BOOL  ; 扫码阻挡气缸缩回位屏蔽
H70.03 BOOL  ; 扫码阻挡气缸伸出屏蔽
H70.04 BOOL  ; 上料夹爪气缸张开位屏蔽
H70.05 BOOL  ; 上料夹爪气缸夹紧位屏蔽
H70.06 BOOL  ; 上料#1级升降气缸缩回位屏蔽
H70.07 BOOL  ; 上料#1级升降气缸伸出位屏蔽
H70.08 BOOL  ; 上料#2级升降气缸缩回位屏蔽
H70.09 BOOL  ; 上料#2级升降气缸伸出位屏蔽
H70.10 BOOL  ; 上料横移气缸缩回位屏蔽
H70.11 BOOL  ; 上料横移气缸伸出位屏蔽
H70.12 BOOL  ; 下料夹爪气缸缩回位屏蔽
H70.13 BOOL  ; 下料夹爪气缸伸出位屏蔽
H70.14 BOOL  ; 下料#1级升降气缸缩回位屏蔽
H70.15 BOOL  ; 下料#1级升降气缸伸出位屏蔽
H71.00 BOOL  ; 下料#2级升降气缸缩回位屏蔽
H71.01 BOOL  ; 下料#2级升降气缸伸出位屏蔽
H71.02 BOOL  ; 下料横移气缸缩回位屏蔽
H71.03 BOOL  ; 下料横移气缸伸出位屏蔽
H71.04 BOOL  ; 前腔体入料位顶升气缸缩回屏蔽
H71.05 BOOL  ; 拉带出料夹爪有料感应屏蔽
H71.06 BOOL  ; 前腔体进料夹爪有料感应屏蔽
H71.07 BOOL  ; 前腔体出料夹爪有料感应屏蔽
H71.08 BOOL  ; 后腔体进料夹爪有料感应屏蔽
H71.09 BOOL  ; 后腔体出料夹爪有料感应
H71.10 BOOL  ; 精密调压阀过低报警屏蔽
H71.11 BOOL  ; 后腔体出料位顶升气缸伸出位屏蔽
H71.12 BOOL  ; 前腔体进料夹爪张开位屏蔽
H71.13 BOOL  ; 前腔体进料夹爪夹紧位屏蔽
H71.14 BOOL  ; 前腔体进料升降气缸缩回位屏蔽
H71.15 BOOL  ; 前腔体进料升降气缸伸出位屏蔽
H72.00 BOOL  ; 后腔体进料夹爪张开位屏蔽
H72.01 BOOL  ; 后腔体进料夹爪夹紧位屏蔽
H72.02 BOOL  ; 后腔体进料升降气缸缩回位屏蔽
H72.03 BOOL  ; 后腔体进料升降气缸伸出位屏蔽
H72.04 BOOL  ; 前腔体出料夹爪张开位屏蔽
H72.05 BOOL  ; 前腔体出料夹爪夹紧位屏蔽
H72.06 BOOL  ; 前腔体出料升降气缸缩回位屏蔽
H72.07 BOOL  ; 前腔体出料升降气缸伸出位屏蔽
H72.08 BOOL  ; 后腔体出料夹爪张开位屏蔽
H72.09 BOOL  ; 后腔体出料夹爪伸出位屏蔽
H72.10 BOOL  ; 后腔体出料升降气缸缩回位屏蔽
H72.11 BOOL  ; 后腔体出料升降气缸伸出位屏蔽
H72.12 BOOL  ; #1腔体移栽气缸缩回位屏蔽
H72.13 BOOL  ; #1腔体移栽气缸伸出位屏蔽
H72.14 BOOL  ; #1腔体顶升气缸缩回位屏蔽
H72.15 BOOL  ; #1腔体顶升气缸伸出位屏蔽
H73.00 BOOL  ; #2腔体移栽气缸缩回位屏蔽
H73.01 BOOL  ; #2腔体移栽气缸伸出位屏蔽
H73.02 BOOL  ; #2腔体顶升气缸缩回位屏蔽
H73.03 BOOL  ; #2腔体顶升气缸伸出位屏蔽
H73.04 BOOL  ; #3腔体移栽气缸缩回位屏蔽
H73.05 BOOL  ; #3腔体移栽气缸伸出位屏蔽
H73.06 BOOL  ; #3腔体顶升气缸缩回位屏蔽
H73.07 BOOL  ; #3腔体顶升气缸伸出位屏蔽
H73.08 BOOL  ; #4腔体移栽气缸缩回位屏蔽
H73.09 BOOL  ; #4腔体移栽气缸伸出位屏蔽
H73.10 BOOL  ; #4腔体顶升气缸缩回位屏蔽
H73.11 BOOL  ; #4腔体顶升气缸伸出位屏蔽
H73.12 BOOL  ; #1扫码NG推料气缸缩回位屏蔽
H73.13 BOOL  ; #1扫码NG推料气缸伸出位屏蔽
H73.14 BOOL  ; #2扫码NG推料气缸缩回位屏蔽
H73.15 BOOL  ; #2扫码NG推料气缸伸出位屏蔽
H74.00 BOOL  ; #1测试NG推料气缸缩回位屏蔽
H74.01 BOOL  ; #1测试NG推料气缸伸出位屏蔽
H74.02 BOOL  ; #2测试NG推料气缸缩回位屏蔽
H74.03 BOOL  ; #2测试NG推料气缸伸出位屏蔽
H74.04 BOOL  ; #1扫码NG位缓存屏蔽
H74.05 BOOL  ; #2扫码NG位缓存屏蔽
H74.06 BOOL  ; #3扫码NG位缓存屏蔽
H74.07 BOOL  ; #4扫码NG位缓存屏蔽
H74.08 BOOL  ; #1测试NG位缓存屏蔽
H74.09 BOOL  ; #2测试NG位缓存屏蔽
H74.10 BOOL  ; #3测试NG位缓存屏蔽
H74.11 BOOL  ; #4测试NG位缓存屏蔽
H74.12 BOOL  ; 下料拉带位有料屏蔽
H74.13 BOOL  ; 入料托盘上料处有料屏蔽
H74.14 BOOL  ; 前出料托盘处有料屏蔽
H74.15 BOOL  ; 后出料托盘处有料屏蔽
H75.00 BOOL  ; 前腔体有料感应屏蔽
H75.01 BOOL  ; 后腔体有料感应屏蔽
H75.02 BOOL  ; 上料夹爪柔性报警屏蔽
H75.03 BOOL  ; 下料夹爪柔性报警屏蔽
H75.04 BOOL  ; 前进料机械手柔性报警屏蔽
H75.05 BOOL  ; 后进料机械手柔性报警屏蔽
H75.06 BOOL  ; 前出料机械手柔性报警屏蔽
H75.07 BOOL  ; 后出料机械手柔性报警屏蔽
H7.00 BOOL  ; 右扫码位扫码OK记忆
H7.01 BOOL  ; 右进料上料位扫码OK记忆
H7.02 BOOL  ; 右进料夹爪上条码OK记忆
H80.00 BOOL  ; 调机模式
H81.00 BOOL  ; 老氦检仪选择
H81.01 BOOL  ; 氦检仪电源打开—HMI
H81.02 BOOL  ; 提速度
H81.03 BOOL  ; 吹气关（ON不使用OFF使用）
H83.00 BOOL  ; 扫码NG模拟
H83.01 BOOL  ; 测试NG模拟
H8.00 BOOL  ; 扫码NG
T0000 BOOL  ; PLC上电
T0001 BOOL  ; PLC上电延时1s
T0002 BOOL  ; PLC上电延时10s
T0003 BOOL  ; 手动模式延时
T0004 BOOL  ; 自动模式延时
T0005 BOOL  ; 蜂鸣器鸣叫时间
T0006 BOOL  ; 复位按钮2秒延时
T0007 BOOL  ; 自动停止完成延时
T0008 BOOL  ; 启动按钮按下1s延时
T0009 BOOL  ; 停止按钮按下延时
T0010 BOOL  ; 进料机构复位完成延时
T0011 BOOL  ; 前上料机构复位完成延时
T0012 BOOL  ; 前下料机构复位完成延时
T0013 BOOL  ; 后上料机构复位完成延时
T0014 BOOL  ; 后下料机构复位完成延时
T0015 BOOL  ; 1#腔体机构复位完成延时
T0016 BOOL  ; 2#腔体机构复位完成延时
T0017 BOOL  ; 3#腔体机构复位完成延时
T0018 BOOL  ; 4#腔体机构复位完成延时
T0019 BOOL  ; 清料停止完成延时
T0020 BOOL  ; 出料机构复位完成延时
T0021 BOOL  ; 整机在初始位延时
T0022 BOOL  ; 氦检仪稳定延时
T0023 BOOL  ; 氦检仪使用开始延时1s读取状态
T0025 BOOL  ; 柔性报警解除按钮按下延时
T0026 BOOL  ; 氦检仪漏率稳定延时
T0028 BOOL  ; 氦检仪漏率低于设定值延时
T0030 BOOL  ; 真空泵1启动后延时
T0031 BOOL  ; 无腔体正在氦检(A)
T0032 BOOL  ; 真空泵2启动后延时
T0033 BOOL  ; 1#真空泵启动后延时2s
T0034 BOOL  ; 复位延时关停止
T0035 BOOL  ; 1#真空泵启动后延时2s
T0037 BOOL  ; 1#真空泵停机1分钟内禁止启动保护延时
T0038 BOOL  ; 2#真空泵停机1分钟内禁止启动保护延时
T0050 BOOL  ; PC运行标志断开时间
T0051 BOOL  ; PC通信正常持续时间
T0052 BOOL  ; 数据请求延时
T0053 BOOL  ; 前下料数据请求延时
T0054 BOOL  ; 后下料数据请求延时
T0055 BOOL  ; 延时扫码
T0057 BOOL  ; 3单元#2串口占用持续时间
T0058 BOOL  ; 扫码延时
T0059 BOOL  ; 右扫码延时
T0060 BOOL  ; 延时关校准
T0080 BOOL  ; 腔体抽真空时间
T0081 BOOL  ; 电池抽真空时间
T0083 BOOL  ; 注氦气时间
T0090 BOOL  ; 扫码NG料检测辅助1
T0091 BOOL  ; 扫码NG料检测辅助2
T0092 BOOL  ; 扫码NG料检测辅助3
T0093 BOOL  ; 扫码NG料检测辅助4
T0094 BOOL  ; 测试NG缓存1延时
T0095 BOOL  ; 测试NG缓存2延时
T0096 BOOL  ; 测试NG缓存3延时
T0097 BOOL  ; 测试NG缓存4延时
T0100 BOOL  ; 扫码位有料感应
T0101 BOOL  ; 扫码位无料感应
T0102 BOOL  ; 出料拉带可放料信号
T0103 BOOL  ; 出料拉带不可放料信号
T0104 BOOL  ; 上料位有料感应延时
T0105 BOOL  ; 抓料位有料感应无料感应
T0106 BOOL  ; 下料拉带无料感应
T0107 BOOL  ; 后进料旋转位无料感应
T0108 BOOL  ; 前出料旋转位有料感应
T0109 BOOL  ; 进料位托盘无料感应
T0110 BOOL  ; 前下料位有料感应
T0111 BOOL  ; 前下料位无料感应
T0112 BOOL  ; 后下料位有料感应
T0113 BOOL  ; 后下料位无料感应
T0114 BOOL  ; 腔体1右电池有料感应
T0115 BOOL  ; 腔体1右电池无料感应
T0116 BOOL  ; 腔体2左电池有料感应
T0117 BOOL  ; 腔体2左电池无料感应
T0118 BOOL  ; 腔体2右电池有料感应
T0119 BOOL  ; 腔体2右电池无料感应
T0120 BOOL  ; 腔体3左电池有料感应
T0121 BOOL  ; 腔体3左电池无料感应
T0122 BOOL  ; 隔离处感应
T0123 BOOL  ; 隔离处无料感应
T0124 BOOL  ; 腔体4左电池有料感应
T0125 BOOL  ; 腔体4左电池无料感应
T0126 BOOL  ; 腔体4右电池有料感应
T0127 BOOL  ; 腔体4右电池无料感应
T0128 BOOL  ; #1扫码NG缓存料满感应
T0129 BOOL  ; #1扫码NG缓存料未满感应
T0130 BOOL  ; #2扫码NG缓存料满感应
T0131 BOOL  ; #2扫码NG缓存料未满感应
T0132 BOOL  ; #3扫码NG缓存料满感应
T0133 BOOL  ; #3扫码NG缓存料未满感应
T0134 BOOL  ; #4扫码NG缓存料满感应
T0135 BOOL  ; #4扫码NG缓存料未满感应
T0136 BOOL  ; 前上料机械手柔性报警
T0137 BOOL  ; 前上料机械手柔性未报警
T0138 BOOL  ; 前下料机械手柔性报警
T0139 BOOL  ; 前下料机械手柔性未报警
T0140 BOOL  ; 后上料机械手柔性报警
T0141 BOOL  ; 后上料机械手柔性未报警
T0142 BOOL  ; 后下料机械手柔性报警
T0143 BOOL  ; 后下料机械手柔性未报警
T0144 BOOL  ; #1测试NG缓存放料位有料感应
T0145 BOOL  ; #2测试NG缓存位有料感应
T0146 BOOL  ; #3测试NG缓存放料位有料感应
T0147 BOOL  ; #4测试NG缓存位有料感应
T0148 BOOL  ; #1测试NG缓存放料位无料感应
T0149 BOOL  ; #2测试NG缓存放料位无料感应
T0150 BOOL  ; #3测试NG缓存储料位无料感应延时
T0151 BOOL  ; #4测试NG缓存储料位无料感应延时
T0152 BOOL  ; 漏率判断延时
T0153 BOOL  ; 拉带进料夹爪无料感应延时
T0154 BOOL  ; 拉带出料夹爪无料感应延时
T0155 BOOL  ; 前腔体进料夹爪无料感应延时
T0156 BOOL  ; 前腔体出料夹爪无料感应
T0157 BOOL  ; 后腔体进料夹爪有料感应延时
T0158 BOOL  ; 后腔体出料夹爪有料感应延时
T0160 BOOL  ; 左扫码通信异常
T0161 BOOL  ; 右扫码通信异常
T0163 BOOL  ; 氦检仪通信异常
T0165 BOOL  ; #1真空计断线时间
T0166 BOOL  ; #2真空计断线时间
T0167 BOOL  ; #3真空计断线时间
T0168 BOOL  ; #4真空计断线时间
T0169 BOOL  ; #1电池真空压力表断线时间
T0170 BOOL  ; #2电池真空压力断表线时间
T0171 BOOL  ; #3电池真空压力断表线时间
T0172 BOOL  ; #4电池真空压力断表线时间
T0173 BOOL  ; #1密封气缸压力断表线时间
T0174 BOOL  ; #2密封气缸压力断表线时间
T0175 BOOL  ; #3密封气缸压力断表线时间
T0176 BOOL  ; #4密封气缸压力断表线时间
T0180 BOOL  ; 上料夹爪柔性报警
T0181 BOOL  ; 上料夹爪柔性未报警
T0182 BOOL  ; 出料夹爪柔性报警
T0183 BOOL  ; 出料夹爪柔性未报警
T0190 BOOL  ; 氦检仪状态判断延时
T0191 BOOL  ; 检漏口压力判断延时
T0192 BOOL  ; 漏率判断延时
T0193 BOOL  ; 单元4串口1占用时间
T0194 BOOL  ; 串口占用持续时间
T0200 BOOL  ; 上料横移气缸缩回位
T0201 BOOL  ; 上料横移气缸伸出位
T0202 BOOL  ; 拉带进料夹爪有料感应延时
T0203 BOOL  ; 拉带出料夹爪有料感应延时
T0204 BOOL  ; 前腔体进料夹爪有料感应
T0205 BOOL  ; 前腔体出料夹爪有料感应
T0206 BOOL  ; 来料隔离气缸缩回位
T0207 BOOL  ; 来料隔离气缸伸出位
T0208 BOOL  ; 扫码阻挡气缸缩回位
T0209 BOOL  ; 扫码阻挡气缸伸出
T0210 BOOL  ; 上料夹爪张开位
T0211 BOOL  ; 上料夹爪夹紧位
T0212 BOOL  ; 上料#1气缸缩回位
T0213 BOOL  ; 上料#1气缸伸出位位
T0214 BOOL  ; 上料#2气缸缩回位
T0215 BOOL  ; 上料#2气缸伸出位
T0216 BOOL  ; 下料夹爪张开位
T0217 BOOL  ; 下料夹爪夹紧位
T0218 BOOL  ; 下料#1级升降气缸缩回位
T0219 BOOL  ; 下料#1级升降气缸伸出位
T0220 BOOL  ; 下料#2级升降气缸缩回位
T0221 BOOL  ; 下料#2级升降气缸伸出位
T0222 BOOL  ; 下料横移气缸缩回位
T0223 BOOL  ; 下料横移气缸伸出位
T0224 BOOL  ; 后腔体进料夹爪有料感应
T0225 BOOL  ; 后腔体出料夹爪有料感应
T0226 BOOL  ; 精密调压阀过低报警
T0227 BOOL  ; 后腔体出料位顶升气缸伸出位
T0228 BOOL  ; 前腔体进料机械手夹爪张开位
T0229 BOOL  ; 前腔体进料机械手夹爪夹紧位
T0230 BOOL  ; 前腔体进料机械手升降气缸缩回位
T0231 BOOL  ; 前腔体进料机械手升降气缸伸出位
T0232 BOOL  ; 前腔体出料机械手夹爪张开位
T0233 BOOL  ; 前腔体出料机械手夹爪夹紧位
T0234 BOOL  ; 前腔体出料机械手升降气缸缩回位
T0235 BOOL  ; 前腔体出料机械手升降气缸伸出位
T0236 BOOL  ; 后腔体进料机械手夹爪张开位
T0237 BOOL  ; 后腔体进料机械手夹爪夹紧位
T0238 BOOL  ; 后腔体进料机械手升降气缸缩回位
T0239 BOOL  ; 后腔体进料机械手升降气缸伸出位
T0240 BOOL  ; 后腔体出料机械手夹爪张开位
T0241 BOOL  ; 后腔体出料机械手夹爪夹紧位
T0242 BOOL  ; 后腔体出料机械手升降气缸缩回位
T0243 BOOL  ; 后腔体出料机械手升降气缸伸出位
T0244 BOOL  ; #1腔体移栽气缸伸出位
T0245 BOOL  ; #1腔体移栽气缸缩回位
T0246 BOOL  ; #1腔体顶升气缸缩回位
T0247 BOOL  ; #1腔体顶升气缸伸出位
T0248 BOOL  ; #2腔体移栽气缸伸出
T0249 BOOL  ; #2腔体移栽气缸缩回
T0250 BOOL  ; #2腔体顶升气缸缩回位
T0251 BOOL  ; #2腔体顶升气缸伸出位
T0252 BOOL  ; #3腔体移栽气缸伸出.
T0253 BOOL  ; #3腔体移栽气缸缩回位.
T0254 BOOL  ; #3腔体顶升气缸缩回位
T0255 BOOL  ; #3腔体顶升气缸伸出位
T0256 BOOL  ; #4腔体移栽气缸伸出位
T0257 BOOL  ; #4腔体移栽气缸缩回位
T0258 BOOL  ; #4腔体顶升气缸缩回位
T0259 BOOL  ; #4腔体顶升气缸伸出位
T0260 BOOL  ; #1扫码NG推料气缸缩回位
T0261 BOOL  ; #1扫码NG推料气缸伸出位
T0262 BOOL  ; #2扫码NG推料气缸缩回位
T0263 BOOL  ; #2扫码NG推料气缸伸出位
T0264 BOOL  ; #1测试NG推料气缸缩回位
T0265 BOOL  ; #1测试NG推料气缸伸出延时
T0266 BOOL  ; #2测试NG推料气缸缩回位
T0267 BOOL  ; #2测试NG推料气缸伸出位
T0268 BOOL  ; 前进料旋转气缸初始位
T0269 BOOL  ; 前进料旋转气缸旋转位
T0270 BOOL  ; 延时关模式
T0271 BOOL  ; 前出料旋转气缸旋转位
T0272 BOOL  ; 后进料旋转气缸初始位
T0273 BOOL  ; 后进料旋转气缸旋转位
T0274 BOOL  ; 后出料旋转气缸初始位
T0275 BOOL  ; 后出料旋转气缸旋转位
T0280 BOOL  ; 腔体1左电池密封气缸上位
T0281 BOOL  ; 腔体1左电池密封气缸下位
T0282 BOOL  ; 腔体1右电池密封气缸上位
T0283 BOOL  ; 腔体1右电池密封气缸下位
T0284 BOOL  ; 腔体2左电池密封气缸上位
T0285 BOOL  ; 腔体2左电池密封气缸下位
T0286 BOOL  ; 腔体2右电池密封气缸上位
T0287 BOOL  ; 腔体2右电池密封气缸下位
T0288 BOOL  ; 腔体3左电池密封气缸上位
T0289 BOOL  ; 腔体3左电池密封气缸下位
T0290 BOOL  ; 腔体3右电池密封气缸上位
T0291 BOOL  ; 腔体3右电池密封气缸下位
T0292 BOOL  ; 腔体4左电池密封气缸上位
T0293 BOOL  ; 腔体4左电池密封气缸下位
T0294 BOOL  ; 腔体4右电池密封气缸上位
T0295 BOOL  ; 腔体4右电池密封气缸下位
T0296 BOOL  ; 腔体1平移气缸后退位
T0297 BOOL  ; 腔体1平移气缸前进位
T0298 BOOL  ; 腔体1顶升气缸下位
T0299 BOOL  ; 腔体1顶升气缸上位
T0300 BOOL  ; 腔体2平移气缸后退位
T0301 BOOL  ; 吹气时间
T0302 BOOL  ; 腔体2顶升气缸下位
T0303 BOOL  ; 腔体2顶升气缸上位
T0304 BOOL  ; 腔体3平移气缸后退位
T0305 BOOL  ; 腔体3平移气缸前进位
T0306 BOOL  ; 腔体3顶升气缸下位
T0307 BOOL  ; 腔体3顶升气缸上位
T0308 BOOL  ; 腔体4平移气缸后退位
T0309 BOOL  ; 腔体4平移气缸前进位
T0310 BOOL  ; 腔体4顶升气缸下位
T0311 BOOL  ; 腔体4顶升气缸上位
T0312 BOOL  ; 进料移栽伺服Ready
T0313 BOOL  ; 进料移栽伺服报警
T0314 BOOL  ; 出料移栽伺服Ready
T0315 BOOL  ; 出料移栽伺服报警
T0316 BOOL  ; 前上料伺服Ready
T0317 BOOL  ; 前上料伺服报警
T0318 BOOL  ; 前下料伺服Ready
T0319 BOOL  ; 前下料伺服报警
T0320 BOOL  ; 后上料伺服Ready
T0321 BOOL  ; 后上料伺服报警
T0322 BOOL  ; 后下料伺服Ready
T0323 BOOL  ; 后下料伺服报警
T0324 BOOL  ; 氦检仪异常信号
T0325 BOOL  ; 前门磁信号
T0326 BOOL  ; 后门磁信号
T0327 BOOL  ; 左门磁信号
T0328 BOOL  ; 右门磁信号
T0329 BOOL  ; 气压开关
T0330 BOOL  ; 真空泵缺相保护
T0332 BOOL  ; 氦气源压力过低延时
T0333 BOOL  ; 扫码NG缓存位有料感应延时
T0334 BOOL  ; 扫码NG缓存位无料感应延时
T0335 BOOL  ; 出料拉带上有料感应延时
T0336 BOOL  ; $?St$Bk?_#[2599] / 出料拉带上无料感应延时 / $?St$Bk?_#[2599]
T0337 BOOL  ; 氦检仪报警延时2s
T0340 BOOL  ; 腔体1电池密封气缸上位
T0341 BOOL  ; 腔体1电池密封气缸下位
T0342 BOOL  ; 腔体2电池密封气缸上位
T0343 BOOL  ; 腔体2电池密封气缸下位
T0344 BOOL  ; 腔体3电池密封气缸上位
T0345 BOOL  ; 腔体3电池密封气缸下位
T0346 BOOL  ; 腔体4电池密封气缸上位
T0347 BOOL  ; 腔体4电池密封气缸下位
T0348 BOOL  ; 进料夹爪气缸张开位
T0349 BOOL  ; 进料夹爪气缸夹紧位
T0350 BOOL  ; 前上料夹爪气缸张开位
T0351 BOOL  ; 前上料夹爪气缸夹紧位
T0352 BOOL  ; 前下料夹爪气缸张开位
T0353 BOOL  ; 前下料夹爪气缸夹紧位
T0354 BOOL  ; 后上料夹爪气缸张开位
T0355 BOOL  ; 后上料夹爪气缸夹紧位
T0356 BOOL  ; 后下料夹爪气缸张开位
T0357 BOOL  ; 后下料夹爪气缸夹紧位
T0358 BOOL  ; 出料夹爪气缸张开位
T0359 BOOL  ; 出料夹爪气缸夹紧位
T0360 BOOL  ; 进料位有料感应延时
T0361 BOOL  ; 进料位无料感应延时
T0362 BOOL  ; 进料位抓料安全检测延时
T0363 BOOL  ; 进料位抓料不安全检测延时
T0364 BOOL  ; 真空泵1热过载报警延时
T0365 BOOL  ; 真空泵2热过载报警延时
T0368 BOOL  ; 氦检仪不在检漏状态延时
T0370 BOOL  ; 进料升降伺服Ready
T0371 BOOL  ; 进料升降伺服报警
T0372 BOOL  ; 出料升降伺服Ready
T0373 BOOL  ; 出料升降伺服报警
T0380 BOOL  ; 进料升降伺服传输数据延时
T0381 BOOL  ; 进料升降伺服手动延时
T0382 BOOL  ; 进料升降伺服手动定位延时(M)
T0385 BOOL  ; 出料升降伺服手动数据传输延时
T0386 BOOL  ; 出料升降手动延时
T0430 BOOL  ; #1氦检原位延时确认
T0431 BOOL  ; #2氦检原位延时确认
T0432 BOOL  ; NG后延迟重启氦检仪
T0433 BOOL  ; #3氦检原位延时确认
T0435 BOOL  ; #4氦检原位
T0500 BOOL  ; 下降夹爪抓料延时
T0501 BOOL  ; 升降缸缩回启动横移缸
T0502 BOOL  ; 夹爪放料位下降
T0503 BOOL  ; 到NG位延时
T0504 BOOL  ; 到前上料位延时
T0505 BOOL  ; 回出料位辅助延时1
T0506 BOOL  ; 回下料位延时
T0507 BOOL  ; 到NG位时间延时
T0508 BOOL  ; .
T0509 BOOL  ; 放料后延时上升2
T0510 BOOL  ; 下降夹爪抓料延时
T0511 BOOL  ; 升降缸缩回启动横移缸
T0512 BOOL  ; 夹爪放料位下降
T0515 BOOL  ; 移载到前上料位延时
T0516 BOOL  ; 到后放料延时
T0520 BOOL  ; 升降伺服下降取料延时1
T0521 BOOL  ; 升降伺服下降取料延时2
T0522 BOOL  ; 升降伺服取料上升延时1
T0523 BOOL  ; 升降伺服取料上升延时2
T0524 BOOL  ; 升降伺服下降放料延时1
T0525 BOOL  ; 升降伺服下降放料延时2
T0526 BOOL  ; 升降伺服放料上升延时1
T0527 BOOL  ; 升降伺服放料后上升延时2
T0530 BOOL  ; 出料升降下取料延时1
T0531 BOOL  ; 出料升降伺服回零延时1
T0532 BOOL  ; 出料升降伺服回零延时2
T0533 BOOL  ; 夹爪放料位下降延时1
T0535 BOOL  ; 放料后延时上升1
T0600 BOOL  ; 到后上料位延时
T0601 BOOL  ; 到上料位延时
T0602 BOOL  ; 出料伺服到等料位#1NG
T0608 BOOL  ; 放料下降延时缓冲
T0700 BOOL  ; 延时触发脉冲
T0701 BOOL  ; 出料伺服延时启动
T0711 BOOL  ; 出料升降柔性辅助时间
T0714 BOOL  ; 出料升降柔性辅助计时
T0802 BOOL  ; 扫码位有料信号
T0803 BOOL  ; 扫码位料停留延时
T0804 BOOL  ; s扫码位料流走检测
T0821 BOOL  ; 氦检阀1关闭检测延时
T0822 BOOL  ; 扫码不良料取走延时
T0823 BOOL  ; 氦检阀2关闭检测延时
T0824 BOOL  ; 扫码位—上料位料流动延时检测
T0825 BOOL  ; 氦检阀3关闭检测延时
T0826 BOOL  ; 氦检阀4关闭延时检测
T0828 BOOL  ; 进料托盘有料检测延时
T0829 BOOL  ; 前下料位有料感应延时
T0830 BOOL  ; 后下料感应延时
T0831 BOOL  ; 后上料最大保持时间
T0832 BOOL  ; 前下最大保持时间
T0833 BOOL  ; 后下最大保持时间
T0835 BOOL  ; 前下料写数据延时报警
T0836 BOOL  ; 前上料最大保持时间
T0837 BOOL  ; 后下料写数据延时报警
T0840 BOOL  ; 报警延迟弹窗
T0850 BOOL  ; 前下料机械手数据移转完成
T0851 BOOL  ; 后下料机械手数据移转完成
T1000 BOOL  ; 进料机构气缸动作异常
T1001 BOOL  ; 进料水平移载伺服报警
T1003 BOOL  ; 进料水平伺服定位目标位置参数错误延时
T1005 BOOL  ; 进料机构自动运行条件延时
T1006 BOOL  ; 扫码机构自动运行条件延时
T1007 BOOL  ; 扫码NG缓存机构自动条件
T1008 BOOL  ; 进料水平伺服停止延时
T1009 BOOL  ; 进料伺服停止延时
T1010 BOOL  ; 进料伺服手动定位延时(M)
T1011 BOOL  ; 进料伺服手动延时
T1012 BOOL  ; 进料伺服传输数据延时
T1016 BOOL  ; 进料伺服自动定位延时(A)
T1021 BOOL  ; 进料升降伺服报警
T1023 BOOL  ; 进料升降伺服定位目标位置参数错误延时
T1028 BOOL  ; 进料升降伺服停止延时
T1034 BOOL  ; 避位气缸接料条件延时(A)
T1035 BOOL  ; 避位气缸避位条件延时(A)
T1039 BOOL  ; 间隔气缸下降条件延时(A)
T1040 BOOL  ; 扫码气缸前进条件延时(A)
T1041 BOOL  ; 扫码气缸后退条件延时(A)
T1100 BOOL  ; 前上料机构气缸动作异常
T1101 BOOL  ; 前上料伺服报警
T1105 BOOL  ; 前上料机构自动条件延时
T1108 BOOL  ; 前上料伺服停止延时
T1110 BOOL  ; 前上料伺服手动定位延时(M)
T1113 BOOL  ; 前上料手动延时延时
T1114 BOOL  ; 前上料手动位置传输延时
T1116 BOOL  ; 前上料伺服自动定位延时(A)
T1118 BOOL  ; 腔体1判断有料延时
T1119 BOOL  ; 腔体2判断有料延时
T1120 BOOL  ; 延时下降
T1121 BOOL  ; 前上料#1升降气缸下降延时
T1122 BOOL  ; 前下料手动位置传输延时
T1130 BOOL  ; 前下料手动运动延时
T1131 BOOL  ; 前下料手动延时延时
T1132 BOOL  ; 前下料手动位置传输延时
T1150 BOOL  ; #1、#2有料延时报警
T1200 BOOL  ; 前下料机构气缸动作异常
T1201 BOOL  ; 前下料伺服报警
T1205 BOOL  ; 前下料机构自动条件延时
T1208 BOOL  ; 前下料伺服停止延时
T1210 BOOL  ; 前下料伺服手动定位延时(M)
T1216 BOOL  ; 前下料伺服自动定位延时(A)
T1221 BOOL  ; 前下料升降气缸下降放料条件延时(A)
T1300 BOOL  ; 后上料机构气缸动作异常
T1301 BOOL  ; 后上料伺服报警
T1305 BOOL  ; 后上料机构自动条件延时
T1308 BOOL  ; 后上料伺服停止延时
T1310 BOOL  ; 后上料伺服手动定位延时(M)
T1314 BOOL  ; 后上料手动延时延时
T1315 BOOL  ; 后上料手动位置传输延时
T1316 BOOL  ; 后上料伺服自动定位延时(A)
T1318 BOOL  ; 腔体3判断有料延时
T1319 BOOL  ; 腔体4判断有料延时
T1320 BOOL  ; nc
T1323 BOOL  ; 延时复位1238.10
T1330 BOOL  ; 后下料伺服手动定位延时(M)
T1331 BOOL  ; 后下料手动延时延时
T1332 BOOL  ; 后下料手动位置传输延时
T1350 BOOL  ; #3、#4有料延时报警
T1380 BOOL  ; 自动扫码延时
T1381 BOOL  ; 扫码延时
T1382 BOOL  ; 扫码阻挡气缸缩回延时
T1383 BOOL  ; 扫码阻挡气缸伸出延时
T1384 BOOL  ; 电池从扫码位到抓料超时
T1390 BOOL  ; 隔离气缸动延时
T1391 BOOL  ; 隔离气缸关延时
T1400 BOOL  ; 后下料机构气缸动作异常
T1401 BOOL  ; 后下料伺服报警
T1405 BOOL  ; 后下料机构自动条件延时
T1408 BOOL  ; 后下料伺服停止延时
T1410 BOOL  ; 后下料伺服手动定位延时(M)
T1416 BOOL  ; 后下料伺服自动定位延时(A)
T1500 BOOL  ; 1#腔体机构气缸动作异常
T1502 BOOL  ; 1#腔清氦失败延时
T1510 BOOL  ; 1#腔体自检抽真空延时
T1511 BOOL  ; 1#腔体抽真空到达延时
T1512 BOOL  ; 1#腔体自检前保压延时
T1513 BOOL  ; 1#腔体自检保压延时
T1514 BOOL  ; 1#腔体自检保压后数据运算延时
T1515 BOOL  ; 1#腔腔体破真空值到达延时
T1516 BOOL  ; 1#腔电池破真空值到达延时
T1525 BOOL  ; #1密封步延时
T1528 BOOL  ; #1腔腔体抽气阀打开条件延时(A)
T1540 BOOL  ; #1腔体抽气阀打开延时
T1550 BOOL  ; 1#腔体真空值到达(A)
T1551 BOOL  ; 1#电池真空值到达(A)
T1552 BOOL  ; 1#电池注氦完成(A)
T1553 BOOL  ; 1#电池抽真空阀关闭延时(A)
T1554 BOOL  ; 1#腔氦检延时(A)
T1555 BOOL  ; 1#腔氦检结果判断完成(A)
T1556 BOOL  ; 1#腔电池抽残气压力到达延时(A)
T1557 BOOL  ; 1#腔腔体抽残气压力到达延时(A)
T1558 BOOL  ; 1#腔氦检后抽残气时间到达(A)
T1559 BOOL  ; 1#腔腔体破真空压力到达(A)
T1560 BOOL  ; 1#腔电池破真空压力到达(A)
T1561 BOOL  ; 1#腔破真空阀关闭延时(A)
T1562 BOOL  ; 1#腔抽真空阀关闭延时(A)
T1563 BOOL  ; 腔体1真空值到达可氦检条件
T1564 BOOL  ; 1#电池抽残气时间到达
T1565 BOOL  ; #1模组清氦计数延时
T1566 BOOL  ; #1模组清氦破真空后延时
T1567 BOOL  ; 1#腔开氦检阀前抽气时间到达(A)
T1568 BOOL  ; #1模组关氦检阀后延时(清氦步)
T1569 BOOL  ; 1#模组氦检延时(清氦步)
T1570 BOOL  ; 1#腔体抽真空NG延时
T1571 BOOL  ; 1#腔电池抽真空NG延时
T1572 BOOL  ; #1电池注氦压力到达延时
T1580 BOOL  ; 1#腔体抽真空时间到达
T1581 BOOL  ; 1#腔电池抽真空时间到达
T1582 BOOL  ; 1#腔注氦时间到达
T1590 BOOL  ; 所有抽气阀关闭延时
T1591 BOOL  ; 除#1其他都关闭延时
T1592 BOOL  ; 除#1之外其都没抽残气
T1600 BOOL  ; 2#腔体机构气缸动作异常
T1602 BOOL  ; 2#腔清氦失败延时
T1610 BOOL  ; 2#腔体自检抽真空延时
T1611 BOOL  ; 2#腔体抽真空到达延时
T1612 BOOL  ; 2#腔体自检前保压延时
T1613 BOOL  ; 2#腔体自检保压延时
T1614 BOOL  ; 2#腔体自检保压后数据运算延时
T1615 BOOL  ; 2#腔腔体破真空值到达延时
T1616 BOOL  ; 2#腔电池破真空值到达延时
T1640 BOOL  ; #2腔体抽气阀打开延时
T1650 BOOL  ; 2#腔体真空值到达(A)
T1651 BOOL  ; 2#电池真空值到达(A)
T1652 BOOL  ; 2#电池注氦完成(A)
T1653 BOOL  ; 2#电池抽真空阀关闭延时(A)
T1654 BOOL  ; 2#腔氦检延时(A)
T1655 BOOL  ; 2#腔氦检结果判断完成(A)
T1656 BOOL  ; 2#腔电池抽残气压力到达延时(A)
T1657 BOOL  ; 2#腔腔体抽残气压力到达延时(A)
T1658 BOOL  ; 2#腔氦检后抽残气时间到达(A)
T1659 BOOL  ; 2#腔腔体破真空压力到达(A)
T1660 BOOL  ; 2#腔电池破真空压力到达(A)
T1661 BOOL  ; 2#腔破真空阀关闭延时(A)
T1662 BOOL  ; 2#腔抽真空阀关闭延时(A)
T1663 BOOL  ; 腔体2真空值到达可氦检条件
T1664 BOOL  ; 2#电池抽残气时间到达
T1665 BOOL  ; #2模组计数延时
T1666 BOOL  ; #2模组清氦破真空后延时
T1667 BOOL  ; 2#腔开氦检阀前抽气时间到达(A)
T1668 BOOL  ; #2模组关氦检阀后延时(清氦步)
T1669 BOOL  ; 2#模组氦检延时(清氦步)
T1670 BOOL  ; 2#腔体抽真空NG延时
T1671 BOOL  ; 2#腔电池抽真空NG延时
T1672 BOOL  ; 2#电池注氦压力到达延时
T1680 BOOL  ; 2#腔体抽真空时间到达
T1681 BOOL  ; 2#腔电池抽真空时间到达
T1682 BOOL  ; 2#腔注氦时间到达
T1691 BOOL  ; 除#2其他都关闭延时
T1692 BOOL  ; 除#2之外其都没抽残气
T1700 BOOL  ; 3#腔体机构气缸动作异常
T1702 BOOL  ; 3#腔清氦失败延时
T1709 BOOL  ; 3#腔体自检启动条件延时
T1710 BOOL  ; 3#腔体自检抽真空延时
T1711 BOOL  ; 3#腔体抽真空到达延时
T1712 BOOL  ; 3#腔体自检前保压延时
T1713 BOOL  ; 3#腔体自检保压延时
T1714 BOOL  ; 3#腔体自检保压后数据运算延时
T1715 BOOL  ; 3#腔腔体破真空值到达延时
T1716 BOOL  ; 3#腔电池破真空值到达延时
T1740 BOOL  ; #3腔体抽气阀打开延时
T1750 BOOL  ; 3#腔体真空值到达(A)
T1751 BOOL  ; 3#电池真空值到达(A)
T1752 BOOL  ; 3#电池注氦完成(A)
T1753 BOOL  ; 3#电池抽真空阀关闭延时(A)
T1754 BOOL  ; 3#腔氦检延时(A)
T1755 BOOL  ; 3#腔氦检结果判断完成(A)
T1756 BOOL  ; 3#腔电池抽残气压力到达延时(A)
T1757 BOOL  ; 3#腔腔体抽残气压力到达延时(A)
T1758 BOOL  ; 3#腔氦检后抽残气时间到达(A)
T1759 BOOL  ; 3#腔腔体破真空压力到达(A)
T1760 BOOL  ; 3#腔电池破真空压力到达(A)
T1761 BOOL  ; 3#腔破真空阀关闭延时(A)
T1762 BOOL  ; 3#腔抽真空阀关闭延时(A)
T1763 BOOL  ; 腔体3真空值到达可氦检条件
T1764 BOOL  ; 3#电池抽残气时间到达
T1765 BOOL  ; #3模组计数延时
T1766 BOOL  ; #3模组清氦破真空后延时
T1767 BOOL  ; 3#腔开氦检阀前抽气时间到达(A)
T1768 BOOL  ; #3模组关氦检阀后延时(清氦步)
T1769 BOOL  ; 3#模组氦检延时(清氦步)
T1770 BOOL  ; 3#腔体抽真空NG延时
T1771 BOOL  ; 3#腔电池抽真空NG延时
T1772 BOOL  ; 3#电池注氦压力到达延时
T1780 BOOL  ; 3#腔体抽真空时间到达
T1781 BOOL  ; 3#腔电池抽真空时间到达
T1782 BOOL  ; 3#腔注氦时间到达
T1791 BOOL  ; 除#3其他都关闭延时
T1792 BOOL  ; 除#3之外其都没抽残气
T1800 BOOL  ; 4#腔体机构气缸动作异常
T1802 BOOL  ; 4#腔清氦失败延时
T1810 BOOL  ; 4#腔体自检抽真空延时
T1811 BOOL  ; 4#腔体抽真空到达延时
T1812 BOOL  ; 4#腔体自检前保压延时
T1813 BOOL  ; 4#腔体自检保压延时
T1814 BOOL  ; 4#腔体自检保压后数据运算延时
T1815 BOOL  ; 4#腔腔体破真空值到达延时
T1816 BOOL  ; 4#腔电池破真空值到达延时
T1840 BOOL  ; #4腔体抽气阀打开延时
T1850 BOOL  ; 4#腔体真空值到达(A)
T1851 BOOL  ; 4#电池真空值到达(A)
T1852 BOOL  ; 4#电池注氦完成(A)
T1853 BOOL  ; 4#电池抽真空阀关闭延时(A)
T1854 BOOL  ; 4#腔氦检延时(A)
T1855 BOOL  ; 4#腔氦检结果判断完成(A)
T1856 BOOL  ; 4#腔电池抽残气压力到达延时(A)
T1857 BOOL  ; 4#腔腔体抽残气压力到达延时(A)
T1858 BOOL  ; 4#腔氦检后抽残气时间到达(A)
T1859 BOOL  ; 4#腔腔体破真空压力到达(A)
T1860 BOOL  ; 4#腔电池破真空压力到达(A)
T1861 BOOL  ; 4#腔破真空阀关闭延时(A)
T1862 BOOL  ; 4#腔抽真空阀关闭延时(A)
T1863 BOOL  ; 腔体4真空值到达可氦检条件
T1864 BOOL  ; 4#电池抽残气时间到达
T1865 BOOL  ; #4模组计数延时
T1866 BOOL  ; #4模组清氦破真空后延时
T1867 BOOL  ; 4#腔开氦检阀前抽气时间到达(A)
T1868 BOOL  ; #4模组关氦检阀后延时(清氦步)
T1869 BOOL  ; 4#模组氦检延时(清氦步)
T1870 BOOL  ; 4#腔体抽真空NG延时
T1871 BOOL  ; 4#腔电池抽真空NG延时
T1872 BOOL  ; 4#电池注氦压力到达延时
T1880 BOOL  ; 4#腔体抽真空时间到达
T1881 BOOL  ; 4#腔电池抽真空时间到达
T1882 BOOL  ; 4#腔注氦时间到达
T1891 BOOL  ; 除#4其他都关闭延时
T1892 BOOL  ; 除#4之外其都没抽残气
T1900 BOOL  ; 出料机构气缸动作异常
T1901 BOOL  ; 出料伺服报警
T1903 BOOL  ; 出料伺服定位目标位置参数错误延时
T1905 BOOL  ; 出料机构自动条件延时
T1908 BOOL  ; 出料伺服停止延时
T1910 BOOL  ; 出料伺服手动定位延时(M)
T1911 BOOL  ; 出料手动延时
T1912 BOOL  ; 出料伺服手动数据传输延时
T1916 BOOL  ; 出料伺服自动定位延时(A)
T1921 BOOL  ; 出料升降伺服报警
T1923 BOOL  ; 出料升降伺服定位目标位置参数错误延时
T1928 BOOL  ; 出料升降伺服停止延时
T1930 BOOL  ; 推NG延时缩回
T1931 BOOL  ; 推NG延时缩回
T1936 BOOL  ; 抽气延时2
T1937 BOOL  ; 抽气延时3
T1938 BOOL  ; 抽气延时4
T3002 BOOL  ; 防呆寄存器断开
T3004 BOOL  ; 防呆寄存器正常
W0.00 BOOL  ; 自动状态-HMI
W0.01 BOOL  ; 扫码感应拉带停止触发扫码
W100.00 BOOL  ; 1#腔体已用
W100.01 BOOL  ; 2#腔体已用
W100.02 BOOL  ; 3#腔体已用
W100.03 BOOL  ; 4#腔体已用
W101.01 BOOL  ; 在后旋转位放料
W102.01 BOOL  ; 到仓1取料
W102.02 BOOL  ; 到仓2取料
W102.03 BOOL  ; 前下料放料互锁
W104.01 BOOL  ; 到仓3取料
W104.02 BOOL  ; 到仓4取料
W109.01 BOOL  ; 到前取料位取位
W109.02 BOOL  ; 到后取料位取位
W109.03 BOOL  ; 出料夹爪为后托盘料
W10.00 BOOL  ; 进料机械手升降气缸下降
W10.01 BOOL  ; 前上料机械手升降气缸下降
W10.02 BOOL  ; 前下料机械手升降气缸下降
W10.03 BOOL  ; 后上料机械手升降气缸下降
W10.04 BOOL  ; 后下料机械手升降气缸下降
W10.09 BOOL  ; 出料机械手升降气缸下降
W135.00 BOOL  ; 启动氦检仪
W13.10 BOOL  ; 夹缸动作
W13.11 BOOL  ; 下料拉带
W13.12 BOOL  ; 下料位放料
W13.14 BOOL  ; 进料拉带动作
W13.15 BOOL  ; 上料位有料
W14.00 BOOL  ; 氦检仪检漏状态
W14.01 BOOL  ; 氦检仪待机状态
W14.02 BOOL  ; 氦检仪启动状态
W14.03 BOOL  ; 氦检仪定标状态
W14.04 BOOL  ; 氦检仪错误状态
W14.05 BOOL  ; 氦检仪暂停状态
W14.10 BOOL  ; 氦检仪不在检漏状态
W14.14 BOOL  ; 氦检电源开-HMI
W14.15 BOOL  ; 氦捡仪稳定中
W15.00 BOOL  ; 校准完成
W15.01 BOOL  ; 校准出错
W15.02 BOOL  ; 校准中
W15.07 BOOL  ; #1腔体自检泄漏
W15.10 BOOL  ; 腔体1自检NG
W16.05 BOOL  ; #2腔体自检泄露
W16.08 BOOL  ; #2腔体自检NG
W17.05 BOOL  ; #3腔体自检泄露
W17.08 BOOL  ; #3腔体自检NG
W188.05 BOOL  ; nc
W188.06 BOOL  ; nc
W18.05 BOOL  ; #4腔体自检泄露
W18.08 BOOL  ; #4腔体自检NG
W19.01 BOOL  ; PC系统条件
W19.02 BOOL  ; 机械手归零条件
W19.03 BOOL  ; 安全门条件
W19.10 BOOL  ; 启动状态
W19.14 BOOL  ; 氦检仪启动条件
W19.15 BOOL  ; 氦检仪启动
W1.00 BOOL  ; 出料已读取数据
W1.01 BOOL  ; PC处理OK数据已完成
W1.03 BOOL  ; PC处理前NG数据已完成
W1.05 BOOL  ; PC处理后NG数据已完成
W1.10 BOOL  ; PC处理MES数据已完成
W200.00 BOOL  ; 状态复位按钮-HMI
W200.02 BOOL  ; 调试
W200.03 BOOL  ; 调试
W200.04 BOOL  ; 调试
W200.05 BOOL  ; 调试
W200.06 BOOL  ; 调试
W200.08 BOOL  ; 调试
W20.00 BOOL  ; 机台清氦中
W20.01 BOOL  ; 扫码信号
W21.04 BOOL  ; 1#腔电池气密性NG
W21.05 BOOL  ; 1#腔注氦嘴泄漏NG
W21.06 BOOL  ; 1#腔腔体泄漏
W21.07 BOOL  ; 1#腔电池泄漏
W21.08 BOOL  ; 1#腔电池注氦压力超下限
W21.09 BOOL  ; 1#腔电池注氦压力超上限
W21.11 BOOL  ; 1#腔电池注氦超时
W21.13 BOOL  ; 1#腔氦检异常
W21.15 BOOL  ; 1#腔测试异常结束
W22.04 BOOL  ; 2#腔电池气密性NG
W22.05 BOOL  ; 2#腔注氦嘴泄漏NG
W22.06 BOOL  ; 2#腔腔体泄漏
W22.07 BOOL  ; 2#腔电池泄漏
W22.08 BOOL  ; 2#腔电池注氦压力超下限
W22.09 BOOL  ; 2#腔电池注氦压力超上限
W22.11 BOOL  ; 2#腔电池注氦超时
W22.13 BOOL  ; 2#腔氦检异常
W22.15 BOOL  ; 2#腔测试异常结束
W23.04 BOOL  ; 3#腔电池气密性NG
W23.05 BOOL  ; 3#腔注氦嘴泄漏NG
W23.06 BOOL  ; 3#腔腔体泄漏
W23.07 BOOL  ; 3#腔电池泄漏
W23.08 BOOL  ; 3#腔电池注氦压力超下限
W23.09 BOOL  ; 3#腔电池注氦压力超上限
W23.11 BOOL  ; 3#腔电池注氦超时
W23.13 BOOL  ; 3#腔氦检异常
W23.15 BOOL  ; 3#腔测试异常结束
W24.04 BOOL  ; 4#腔电池气密性NG
W24.05 BOOL  ; 4#腔注氦嘴泄漏NG
W24.06 BOOL  ; 4#腔腔体泄漏
W24.07 BOOL  ; 4#腔电池泄漏
W24.08 BOOL  ; 4#腔电池注氦压力超下限
W24.09 BOOL  ; 4#腔电池注氦压力超上限
W24.11 BOOL  ; 4#腔电池注氦超时
W24.13 BOOL  ; 4#腔氦检异常
W24.15 BOOL  ; 4#腔测试异常结束
W26.00 BOOL  ; 有两个以上的电池抽气阀打开
W27.00 BOOL  ; #1#2升降气缸缩回
W27.01 BOOL  ; #1#2升降气缸到位
W27.02 BOOL  ; #1升降气缸下降
W27.03 BOOL  ; 夹爪夹料
W27.04 BOOL  ; 横移缸伸出
W27.05 BOOL  ; 横移缸缩回位
W27.08 BOOL  ; 二级气缸下降
W27.10 BOOL  ; 横移气缸伸出条件
W28.00 BOOL  ; 回原点后自动时到自动到上料位
W28.01 BOOL  ; 到前放料位置
W28.02 BOOL  ; 到后放料位置
W28.04 BOOL  ; 到上料位置
W28.05 BOOL  ; 到上料位置2
W28.06 BOOL  ; 到NG位置
W28.07 BOOL  ; 到NG扫码缓存
W28.08 BOOL  ; NG推料辅助1
W28.09 BOOL  ; 回上料位辅助
W28.10 BOOL  ; 到上料位辅助
W28.11 BOOL  ; #1NG扫码缓存
W28.12 BOOL  ; #2NG扫码缓存
W28.13 BOOL  ; #3NG扫码缓存
W28.14 BOOL  ; #4NG扫码缓存
W28.15 BOOL  ; 水平伺服运动
W29.00 BOOL  ; 前轴屏蔽状态
W29.01 BOOL  ; 后轴屏蔽料状态
W29.15 BOOL  ; 升降伺服运动
W2.00 BOOL  ; HMI已打开报警弹出窗口
W300.00 BOOL  ; 设备故障
W303.01 BOOL  ; 设备暂停
W30.00 BOOL  ; 前入料顶升缸伸出
W30.01 BOOL  ; 后入料顶升缸伸出
W30.02 BOOL  ; #1扫码NG推料气缸
W30.03 BOOL  ; #2扫码NG推料气缸
W310.00 BOOL  ; 扫码阻挡伸出辅助1
W311.02 BOOL  ; 扫码阻挡缩回辅助1
W32.00 BOOL  ; 读检漏仪状态
W32.01 BOOL  ; 读氦检仪状态完成
W32.02 BOOL  ; 读检漏口压力
W32.03 BOOL  ; 读检漏口压力完成
W32.05 BOOL  ; 读漏率
W32.06 BOOL  ; 读漏率完成
W32.07 BOOL  ; 读漏率失败
W32.08 BOOL  ; 读氦检仪状态失败
W32.09 BOOL  ; 读检漏口压力失败
W32.10 BOOL  ; .
W37.00 BOOL  ; #1#2升降气缸缩回
W37.01 BOOL  ; #1#2升降气缸到位
W37.02 BOOL  ; #2升降气缸下降
W37.03 BOOL  ; 下料夹爪夹料
W37.04 BOOL  ; 横移缸到位
W37.05 BOOL  ; 横移缸缩回位
W37.08 BOOL  ; #1升降气缸下降
W37.09 BOOL  ; 复位下放料
W38.00 BOOL  ; 出料回原后自动时初始位
W38.01 BOOL  ; 到前取料位置
W38.02 BOOL  ; 到后取料位置
W38.03 BOOL  ; 前取料顶缸
W38.04 BOOL  ; 后取料顶缸
W38.05 BOOL  ; 回下料位
W38.06 BOOL  ; 到NG料槽
W38.07 BOOL  ; 到#1NG位
W38.08 BOOL  ; 到1#NG料
W38.09 BOOL  ; NG缩回辅助
W38.10 BOOL  ; #1NG
W38.11 BOOL  ; #2NG
W38.12 BOOL  ; #3NG
W38.13 BOOL  ; #4NG
W38.14 BOOL  ; 有NG 料处理
W38.15 BOOL  ; 伺服运动
W390.00 BOOL  ; 暂停 继续
W39.00 BOOL  ; 前轴屏蔽状态
W39.01 BOOL  ; 后轴屏蔽状态
W39.05 BOOL  ; 到下料位
W400.00 BOOL  ; (W400.00) 紧急停止！
W400.01 BOOL  ; (W400.01) 前安全门打开！
W400.02 BOOL  ; (W400.02) 后安全门打开！
W400.03 BOOL  ; (W400.03) 左安全门打开！
W400.04 BOOL  ; (W400.04) 右安全门打开！
W400.05 BOOL  ; (W400.05) 手动模式不能启动！
W400.06 BOOL  ; (W400.06) 氦气源压力过低
W400.07 BOOL  ; (W400.07) 气源压力过低！
W400.08 BOOL  ; (W400.08) 真空泵缺相异常！
W400.09 BOOL  ; (W400.09) 电脑软件未启动
W400.10 BOOL  ; (W400.10) 进料伺服未归零
W400.11 BOOL  ; (W400.11) 前上料伺服未归零
W400.12 BOOL  ; (W400.12) 前下料伺服未归零
W400.13 BOOL  ; (W400.13) 后上料料伺服未归零
W400.14 BOOL  ; (W400.14) 后下料伺服未归零
W400.15 BOOL  ; (W400.15) 出料伺服未归零
W401.00 BOOL  ; (W401.00) 氦检仪没启动
W401.01 BOOL  ; (W401.01) 氦检仪通信异常
W401.02 BOOL  ; (W401.02) #1真空计断线
W401.03 BOOL  ; (W401.03) #2真空计断线
W401.04 BOOL  ; (W401.04) #3真空计断线
W401.05 BOOL  ; (W401.05) #4真空计断线
W401.06 BOOL  ; (W401.06) #1电池真空压力表断线
W401.07 BOOL  ; (W401.07) #2电池真空压力表断线
W401.08 BOOL  ; (W401.08) #3电池真空压力表断线
W401.09 BOOL  ; (W401.09) #4电池真空压力表断线
W401.10 BOOL  ; (W401.10) 连续三个扫码NG
W401.11 BOOL  ; (W401.11) 测连续三个NG
W401.12 BOOL  ; (W401.12) #3密封气缸压力表断线
W401.13 BOOL  ; (W401.13) 电池从扫码位到抓料位超时
W401.14 BOOL  ; (W401.14) 左扫码通信异常
W401.15 BOOL  ; (W401.15) 精密调压阀过低报警
W402.00 BOOL  ; (I:3.02) 扫码阻挡气缸缩回位感应异常！
W402.01 BOOL  ; (W402.11) 进料升降伺服上限位报警！
W402.02 BOOL  ; (I:3.04) 抓料阻挡气缸缩回位感应异常
W402.03 BOOL  ; (I:3.05) 抓料阻挡气缸伸出位感应异常
W402.04 BOOL  ; (I:3.06) 上料夹爪张开位感应异常
W402.05 BOOL  ; (I:3.07) 上料夹爪夹紧位感应异常
W402.06 BOOL  ; (I:3.12) 上料横移气缸缩回位感应异常
W402.07 BOOL  ; (I:3.13) 上料横移气缸伸出位感应异常
W402.08 BOOL  ; (I:3.12) 上料横移气缸要在缩回位
W402.09 BOOL  ; (I:3.13) 上料横移气缸要在伸出位
W402.10 BOOL  ; (W402.10) 进料升降伺服下限位报警！
W402.11 BOOL  ; (W402.10) 进料升降伺服上限位报警！
W402.12 BOOL  ; (W402.12) 进料升降伺服马达报警！
W402.13 BOOL  ; (W402.13) 进料升降伺服原点丢失！
W402.14 BOOL  ; (W402.014) 进料升降伺服准备好信号异常！
W402.15 BOOL  ; (W402.15) 进料升降伺服位置参数错误，按复位键重试！
W403.00 BOOL  ; (W403.00) 进料柔性报警
W403.01 BOOL  ; (W421.05) 出料夹爪柔性报警！
W403.02 BOOL  ; (W403.02) 进料平移气缸开位感应异常！
W403.03 BOOL  ; (W403.03) 进料平移气缸合位感应异常！
W403.04 BOOL  ; (W403.04) 进料左夹爪气缸张开位感应异常！
W403.05 BOOL  ; (W403.05) 进料左夹爪气缸夹紧位感应异常！
W403.06 BOOL  ; (W403.06) 进料右夹爪气缸张开位感应异常！
W403.07 BOOL  ; (W403.07) 进料右夹爪气缸夹紧位感应异常！
W403.08 BOOL  ; (W403.08) 前进料旋转气缸初始位感应异常！
W403.09 BOOL  ; (W403.09) 前进料旋转气缸旋转位感应异常！
W403.10 BOOL  ; (W403.10) 后进料旋转气缸初始位感应异常！
W403.11 BOOL  ; (W403.11) 后进料旋转气缸旋转位感应异常！
W403.12 BOOL  ; (W403.12) 进料位有电池跟随或感应异常
W403.13 BOOL  ; 进料升伺超过软件限位，先按复位键再归零
W403.14 BOOL  ; 出料升伺超过软件限位，先按复位键再归零
W403.15 BOOL  ; 进料拉带有电池拉带不能复位
W404.00 BOOL  ; (W404.00) 进料伺服前限位报警！
W404.01 BOOL  ; (W404.01) 进料伺服后限位报警！
W404.02 BOOL  ; (W404.02) 进料伺服马达报警！
W404.03 BOOL  ; (W404.03) 进料伺服原点丢失！
W404.04 BOOL  ; (W404.04) 进料伺服准备好信号异常！
W404.05 BOOL  ; (W404.05) 进料伺服需要归零！
W404.06 BOOL  ; (W404.06) 进料伺服位置参数错误，按复位键重试！
W404.07 BOOL  ; (W404.07)
W404.08 BOOL  ; (W404.08)
W404.09 BOOL  ; (W404.09) 进料机械手柔性报警
W404.10 BOOL  ; (W404.10) 前进料旋转位有电池！
W404.11 BOOL  ; (W404.11) 后进料旋转位有电池！
W404.12 BOOL  ; (W404.12) 进料位电池MES校验NG
W404.13 BOOL  ; (W404.13)
W404.14 BOOL  ; (W404.14)
W404.15 BOOL  ; (W404.15)
W405.00 BOOL  ; (I:4.14) 前腔体进料机械手夹爪松开位感应异常
W405.01 BOOL  ; (I:4.15) 前腔体进料机械手夹爪夹紧位感应异常
W405.02 BOOL  ; (I:5.00) 前腔体进料机械手升降气缸缩回位感应异常
W405.03 BOOL  ; (I:5.01) 前腔体进料机械手升降气缸伸出位感应异常
W405.04 BOOL  ; (I:1.06) 前腔体进料机械手柔性报警
W405.05 BOOL  ; (W405.05) 前上料左夹爪气缸夹紧位感应异常！
W405.06 BOOL  ; (W405.06) 前上料右夹爪气缸张开位感应异常！
W405.07 BOOL  ; (W405.07) 前上料右夹爪气缸夹紧位感应异常！
W405.08 BOOL  ; (W405.08)
W405.09 BOOL  ; (W405.09)
W405.10 BOOL  ; (W405.10)
W405.11 BOOL  ; (W405.11)
W405.12 BOOL  ; (W405.12)
W405.13 BOOL  ; (W405.13) 前上料机械手柔性报警！
W405.14 BOOL  ; 腔体1有料报警
W405.15 BOOL  ; 腔体2有料报警
W406.00 BOOL  ; (W406.00) 前上料伺服前限位报警！
W406.01 BOOL  ; (W406.01) 前上料伺服后限位报警！
W406.02 BOOL  ; (W406.02) 前上料伺服马达报警！
W406.03 BOOL  ; (W406.03) 前上料伺服原点丢失！
W406.04 BOOL  ; (W406.04) 前上料伺服准备好信号异常！
W406.05 BOOL  ; (W406.05) 前上料伺服需要归零！
W406.06 BOOL  ; (W406.06) 拉带进料夹爪有料感应异常！
W406.07 BOOL  ; (W406.07)拉出料夹爪有料感应异常！
W406.08 BOOL  ; (W406.08)前腔体进料夹爪有料感应异常
W406.09 BOOL  ; (W406.09)前腔体出料夹爪有料感应异常！
W406.10 BOOL  ; (W406.10)后腔体进料夹爪有料感应异常
W406.11 BOOL  ; (W406.11)后腔体出料夹爪有料感应异常！
W406.12 BOOL  ; (W406.12)
W406.13 BOOL  ; (W406.13)
W406.14 BOOL  ; (W406.14)
W406.15 BOOL  ; (W406.15)
W407.00 BOOL  ; (I:5.06) 前腔体出料机械手夹爪张开位感应异常
W407.01 BOOL  ; (I:5.07) 前腔体出料机械手夹爪夹紧位感应异常
W407.02 BOOL  ; (I:5.08) 前腔体出料机械手升降气缸缩回位感应异常
W407.03 BOOL  ; (I:5.09) 前腔体出料机械手升降气缸伸出位感应异常
W407.04 BOOL  ; (W407.04) 前下料左夹爪气缸张开位感应异常！
W407.05 BOOL  ; (W407.05) 前下料左夹爪气缸夹紧位感应异常！
W407.06 BOOL  ; (W407.06) 前下料右夹爪气缸张开位感应异常！
W407.07 BOOL  ; (W407.07) 前下料右夹爪气缸夹紧位感应异常！
W407.08 BOOL  ; (W407.08)
W407.09 BOOL  ; (W407.09)
W407.10 BOOL  ; (W407.10)
W407.11 BOOL  ; (W407.11)
W407.12 BOOL  ; (W407.12)
W407.13 BOOL  ; (W407.13) 前下料机械手柔性报警
W407.14 BOOL  ; (W407.14)
W407.15 BOOL  ; (W407.15)
W408.00 BOOL  ; (W408.00) 前下料伺服前限位报警！
W408.01 BOOL  ; (W408.01) 前下料伺服后限位报警！
W408.02 BOOL  ; (W408.02) 前下料伺服马达报警！
W408.03 BOOL  ; (W408.03) 前下料伺服原点丢失！
W408.04 BOOL  ; (W408.04) 前下料伺服准备好信号异常！
W408.05 BOOL  ; (W408.05) 前下料伺服需要归零！
W408.06 BOOL  ; (W408.06) 前下料伺服位置参数错误，按复位键重试！
W408.07 BOOL  ; (W408.07)
W408.08 BOOL  ; (W408.08)
W408.09 BOOL  ; (W408.09)
W408.10 BOOL  ; (W408.10)
W408.11 BOOL  ; (W408.11)
W408.12 BOOL  ; (W408.12)
W408.13 BOOL  ; (W408.13)
W408.14 BOOL  ; (W408.14)
W408.15 BOOL  ; (W408.15)
W409.00 BOOL  ; (I:5.02) 后腔体进料机械手夹爪张开位感应异常
W409.01 BOOL  ; (I:5.03) 后腔体进料机械手夹爪夹紧位感应异常
W409.02 BOOL  ; (I:5.04) 后腔体进料机械手升降气缸缩回位感应异常
W409.03 BOOL  ; (I:5.05) 后腔体进料机械手升降气缸伸出位感应异常
W409.04 BOOL  ; (W409.04) 后上料左夹爪气缸张开位感应异常！
W409.05 BOOL  ; (W409.05) 后上料左夹爪气缸夹紧位感应异常！
W409.06 BOOL  ; (W409.06) 后上料右夹爪气缸张开位感应异常！
W409.07 BOOL  ; (W409.07) 后上料右夹爪气缸夹紧位感应异常！
W409.08 BOOL  ; (W409.08)
W409.09 BOOL  ; (W409.09)
W409.10 BOOL  ; (W409.10)
W409.11 BOOL  ; (W409.11)
W409.12 BOOL  ; (W409.12)
W409.13 BOOL  ; (I:1.07) 后上料机械手柔性报警
W409.14 BOOL  ; (W409.14) 腔体3有料报警
W409.15 BOOL  ; (W409.15) 腔体4有料报警
W40.00 BOOL  ; 顶缸辅助1
W40.02 BOOL  ; #1测试NG推料气缸
W40.03 BOOL  ; #2测试NG推料气缸
W410.00 BOOL  ; (W410.00) 后上料伺服前限位报警！
W410.01 BOOL  ; (W410.01) 后上料伺服后限位报警！
W410.02 BOOL  ; (W410.02) 后上料伺服马达报警！
W410.03 BOOL  ; (W410.03) 后上料伺服原点丢失！
W410.04 BOOL  ; (W410.04) 后上料伺服准备好信号异常！
W410.05 BOOL  ; (W410.05) 后上料伺服需要归零！
W410.06 BOOL  ; (W410.06) 后上料伺服位置参数错误，按复位键重试！
W410.07 BOOL  ; (W410.07)
W410.08 BOOL  ; (W410.08)
W410.09 BOOL  ; (W410.09)
W410.10 BOOL  ; (W410.10)
W410.11 BOOL  ; (W410.11)
W410.12 BOOL  ; (W410.12)
W410.13 BOOL  ; (W410.13)
W410.14 BOOL  ; (W410.14)
W410.15 BOOL  ; (W410.15)
W411.00 BOOL  ; (I:5.10) 后腔体出料机械手夹爪张开感应异常
W411.01 BOOL  ; (I:5.11) 后腔体出料机械手夹爪夹紧位感应异常
W411.02 BOOL  ; (I:5.12) 后出料机械手升降气缸缩回位感应异常
W411.03 BOOL  ; (I:5.13) 后腔体出料机械手升降气缸伸出位感应异常
W411.04 BOOL  ; (W411.04) 后下料左夹爪气缸张开位感应异常！
W411.05 BOOL  ; (W411.05) 后下料左夹爪气缸夹紧位感应异常！
W411.06 BOOL  ; (W411.06) 后下料右夹爪气缸张开位感应异常！
W411.07 BOOL  ; (W411.07) 后下料右夹爪气缸夹紧位感应异常！
W411.08 BOOL  ; (W411.08)
W411.09 BOOL  ; (W411.09)
W411.10 BOOL  ; (W411.10) 前出料旋转位有电池！
W411.11 BOOL  ; (W411.11) 后出料旋转位有电池！
W411.12 BOOL  ; (W411.12)
W411.13 BOOL  ; (I:1.09) 后腔体出料机械手柔性报警
W411.14 BOOL  ; (W411.14)
W411.15 BOOL  ; (W411.15)
W412.00 BOOL  ; (W412.00) 后下料伺服前限位报警！
W412.01 BOOL  ; (W412.01) 后下料伺服后限位报警！
W412.02 BOOL  ; (W412.02) 后下料伺服马达报警！
W412.03 BOOL  ; (W412.03) 后下料伺服原点丢失！
W412.04 BOOL  ; (W412.04) 后下料伺服准备好信号异常！
W412.05 BOOL  ; (W412.05) 后下料伺服需要归零！
W412.06 BOOL  ; (W412.06) 后下料伺服位置参数错误，按复位键重试！
W412.07 BOOL  ; (W412.07)
W412.08 BOOL  ; (W412.08)
W412.09 BOOL  ; (W412.09)
W412.10 BOOL  ; (W412.10)
W412.11 BOOL  ; (W412.11)
W412.12 BOOL  ; (W412.12)
W412.13 BOOL  ; (W412.13)
W412.14 BOOL  ; (W412.14)
W412.15 BOOL  ; (W412.15)
W413.00 BOOL  ; (I:3.14) 下料夹爪张开位感应异常
W413.01 BOOL  ; (I:3.15) 下料夹爪夹紧位感应异常
W413.02 BOOL  ; (I:4.00) 下料#1级升降气缸缩回位感应异常
W413.03 BOOL  ; (I:4.01) 下料#1级升降气缸伸出位感应异常
W413.04 BOOL  ; (I:4.02) 下料#2级升降气缸缩回位感应异常
W413.05 BOOL  ; (I:4.03) 下料#2级升降气缸伸出位感应异常
W413.06 BOOL  ; (I:4.04) 下料横移气缸缩回位感应异常
W413.07 BOOL  ; (I:4.05) 下料横移气缸伸出位感应异常
W413.08 BOOL  ; (I:4.04) 下料横移气缸要在缩回位才能下降取料
W413.09 BOOL  ; (I:4.04) 下料横移气缸要在缩回位才能下降放料
W413.10 BOOL  ; (W413.10) 出料升降伺服下限位报警！
W413.11 BOOL  ; (W413.10) 出料升降伺服上限位报警！
W413.12 BOOL  ; (W413.12) 出料升降伺服马达报警！
W413.13 BOOL  ; (W413.13)出料升降伺服原点丢失！
W413.14 BOOL  ; (W413.14)出料升降伺服准备好信号异常！
W413.15 BOOL  ; (W413.15) 出料升降伺服位置参数错误，按复位键重试！
W414.00 BOOL  ; (W414.00)
W414.01 BOOL  ; (W414.01)
W414.02 BOOL  ; (W414.02)
W414.03 BOOL  ; (W414.03)
W414.04 BOOL  ; (W414.04)
W414.05 BOOL  ; (W414.05)
W414.06 BOOL  ; (W414.06)
W414.07 BOOL  ; (W414.07)
W414.08 BOOL  ; (W414.08)
W414.09 BOOL  ; (W414.09) 出料机械手柔性报警
W414.10 BOOL  ; (W414.10) 扫码NG缓存料已满
W414.11 BOOL  ; (W414.11) 前NG缓存右料已满
W414.12 BOOL  ; (W414.12) 测试NG缓存料已满
W414.13 BOOL  ; (W414.13) 后NG缓存右料已满
W414.14 BOOL  ; (W414.14)
W414.15 BOOL  ; (W414.15)
W415.00 BOOL  ; (W415.00) 出料伺服前限位报警！
W415.01 BOOL  ; (W415.01) 出料伺服后限位报警！
W415.02 BOOL  ; (W415.02) 出料伺服马达报警！
W415.03 BOOL  ; (W415.03) 出料伺服原点丢失！
W415.04 BOOL  ; (W415.04) 出料伺服准备好信号异常！
W415.05 BOOL  ; (W415.05) 出料伺服需要归零！
W415.06 BOOL  ; (W415.06) 出料伺服位置参数错误，按复位键重试！
W415.07 BOOL  ; (W415.07)
W415.08 BOOL  ; (W415.08)
W415.09 BOOL  ; (W415.09)
W415.10 BOOL  ; (W415.10) 出料拉带出电池超时！
W415.11 BOOL  ; (W415.11) 出料拉带感应电池异常
W415.12 BOOL  ; (W415.12)
W415.13 BOOL  ; (W415.13)
W415.14 BOOL  ; (W415.14)
W415.15 BOOL  ; (W415.15)
W416.00 BOOL  ; (I:5.14) #1腔体移栽气缸缩回位感应异常
W416.01 BOOL  ; (I:5.15) #1腔体移栽气缸伸出位感应异常
W416.02 BOOL  ; (I:6.00) #1腔体顶升气缸缩回位感应异常
W416.03 BOOL  ; (I:6.01) #1腔体顶升气缸伸出位感应异常
W416.04 BOOL  ; (W416.04) 腔体1平移气缸后退位感应异常！
W416.05 BOOL  ; (W416.05) 腔体1平移气缸前进位感应异常！
W416.06 BOOL  ; (W416.06) 腔体1顶升气缸下位感应异常！
W416.07 BOOL  ; (W416.07) 腔体1顶升气缸上位感应异常！
W416.08 BOOL  ; (W416.08) 腔体1腔体破真空超时！
W416.09 BOOL  ; (W416.09) 腔体1电池破真空超时！
W416.10 BOOL  ; (W416.10) 1#真空泵热过载！
W416.11 BOOL  ; (W416.11)
W416.12 BOOL  ; (W416.12)
W416.13 BOOL  ; (W416.13) 腔体1清氦不完全！
W416.14 BOOL  ; (W416.14) 腔体1内有电池！
W416.15 BOOL  ; (W416.15) 腔体1机构步序异常，请进行工站复位！
W417.00 BOOL  ; (I:6.02) #2腔体移栽气缸缩回位感应异常
W417.01 BOOL  ; (I:6.03) #2腔体移栽气缸伸出位感应异常
W417.02 BOOL  ; (I:6.04) #2腔体顶升气缸缩回位感应异常
W417.03 BOOL  ; (I:6.05) #2腔体顶升气缸伸出位感应异常
W417.04 BOOL  ; (W417.04) 腔体2平移气缸后退位感应异常！
W417.05 BOOL  ; (W417.05) 腔体2平移气缸前进位感应异常！
W417.06 BOOL  ; (W417.06) 腔体2顶升气缸下位感应异常！
W417.07 BOOL  ; (W417.07) 腔体2顶升气缸上位感应异常！
W417.08 BOOL  ; (W417.08) 腔体2腔体破真空超时！
W417.09 BOOL  ; (W417.09) 腔体2电池破真空超时！
W417.10 BOOL  ; (W417.10) 氦检仪报警！
W417.11 BOOL  ; (W417.11) MES离线进料次数到达！
W417.12 BOOL  ; (W417.12)
W417.13 BOOL  ; (W417.13) 腔体2清氦不完全！
W417.14 BOOL  ; (W417.14) 腔体2内有电池！
W417.15 BOOL  ; (W417.15) 腔体2机构步序异常，请进行工站复位！
W418.00 BOOL  ; (I:6.06) #3腔体移栽气缸缩回位感应异常
W418.01 BOOL  ; (I:6.07) #3腔体移栽气缸伸出位感应异常
W418.02 BOOL  ; (I:6.08) #3腔体顶升气缸缩回位感应异常
W418.03 BOOL  ; (I:6.09) #3腔体顶升气缸伸出位感应异常
W418.04 BOOL  ; (W418.04) 腔体3平移气缸后退位感应异常！
W418.05 BOOL  ; (W418.05) 腔体3平移气缸前进位感应异常！
W418.06 BOOL  ; (W418.06) 腔体3顶升气缸下位感应异常！
W418.07 BOOL  ; (W418.07) 腔体3顶升气缸上位感应异常！
W418.08 BOOL  ; (W418.08) 腔体3腔体破真空超时！
W418.09 BOOL  ; (W418.09) 腔体3电池破真空超时！
W418.10 BOOL  ; (W418.10) 2#真空泵热过载！
W418.11 BOOL  ; (W418.11)
W418.12 BOOL  ; (W418.12)
W418.13 BOOL  ; (W418.13) 腔体3清氦不完全！
W418.14 BOOL  ; (W418.14) 腔体3内有电池！
W418.15 BOOL  ; (W418.15) 腔体3机构步序异常，请进行工站复位！
W419.00 BOOL  ; (I:6.10) #4移栽气缸缩回位感应异常
W419.01 BOOL  ; (I:6.11) #4腔体移栽气缸伸出位感应异常
W419.02 BOOL  ; (I:6.12) #4腔体顶升气缸缩回位感应异常
W419.03 BOOL  ; (I:6.13) #4腔体顶升气缸伸出位感应异常
W419.04 BOOL  ; (W419.04) 腔体4平移气缸后退位感应异常！
W419.05 BOOL  ; (W419.05) 腔体4平移气缸前进位感应异常！
W419.06 BOOL  ; (W419.06) 腔体4顶升气缸下位感应异常！
W419.07 BOOL  ; (W419.07) 腔体4顶升气缸上位感应异常！
W419.08 BOOL  ; (W419.08) 腔体4腔体破真空超时！
W419.09 BOOL  ; (W419.09) 腔体4电池破真空超时！
W419.10 BOOL  ; (W419.10)
W419.11 BOOL  ; (W419.11)
W419.12 BOOL  ; (W419.12)
W419.13 BOOL  ; (W419.13) 腔体4清氦不完全！
W419.14 BOOL  ; (W419.14) 腔体4内有电池！
W419.15 BOOL  ; (W419.15) 腔体4机构步序异常，请进行工站复位！
W420.00 BOOL  ; 扫码NG感应1异常
W420.01 BOOL  ; 扫码NG感应2异常
W420.02 BOOL  ; 扫码NG感应3异常
W420.03 BOOL  ; 扫码N感应4异常
W420.04 BOOL  ; 测试NG感应1异常
W420.05 BOOL  ; 测试NG感应2异常
W420.06 BOOL  ; 测试NG感应3异常
W420.07 BOOL  ; 测试NG感应4异常
W420.08 BOOL  ; 进料托盘有料感应异常
W420.09 BOOL  ; 前下料感应异常
W420.10 BOOL  ; 后下料感应异常
W420.11 BOOL  ; 检漏口压力异常
W420.12 BOOL  ; 氦检阀1关闭异常
W420.13 BOOL  ; 氦检阀2关闭异常
W420.14 BOOL  ; 氦检阀3关闭异常
W420.15 BOOL  ; 氦检阀4关闭异常
W421.00 BOOL  ; 1#测试NG气缸缩回位异常
W421.01 BOOL  ; 1#测试NG气缸伸出位异常
W421.04 BOOL  ; 1#扫码NG气缸缩回位异常
W421.05 BOOL  ; 1#扫码NG推料气缸伸出位异常
W421.06 BOOL  ; 腔体1连续NG
W421.07 BOOL  ; 腔体1自动离线
W421.08 BOOL  ; 腔体2连续NG
W421.09 BOOL  ; 腔体2自动离线
W421.10 BOOL  ; 腔体3连续NG
W421.11 BOOL  ; 腔体3离线报警
W421.12 BOOL  ; 腔体4连续NG
W421.13 BOOL  ; 腔体4自动离线报警
W422.00 BOOL  ; #1 NG清零
W422.01 BOOL  ; #2 NG清零
W422.02 BOOL  ; #3NG清零
W422.03 BOOL  ; #4NG清零
W422.04 BOOL  ; 数据传输超时
W422.07 BOOL  ; 氦检仪检漏口 值长时超低
W423.00 BOOL  ; 前上料夹紧中
W423.01 BOOL  ; 前下料夹紧中
W423.02 BOOL  ; 后上料爪紧中
W423.03 BOOL  ; 后下料夹紧中
W425.00 BOOL  ; 入料升降柔性辅助
W425.01 BOOL  ; 出料升降柔性辅助
W44.00 BOOL  ; 1#真空泵停机1分钟内禁止启动保护
W44.06 BOOL  ; 2#真空泵停机1分钟内禁止启动保护
W44.10 BOOL  ; 扫码NG槽无料
W44.12 BOOL  ; 测试NG槽无料
W450.00 BOOL  ; NG料满警报
W450.01 BOOL  ; 测试NG料满
W480 CHANNEL  ; 校验触发
W480.00 BOOL  ; MES数据发送请求
W480.01 BOOL  ; #1腔体数据发送请求
W480.02 BOOL  ; #2腔体数据发送请求
W480.03 BOOL  ; #3腔体数据发送请求
W480.04 BOOL  ; #4腔体数据发送请求
W480.05 BOOL  ; #1腔体NG数据发送请求
W480.06 BOOL  ; #2腔体NG数据发送请求
W480.07 BOOL  ; #3腔体NG数据发送请求
W480.08 BOOL  ; #4腔体NG数据发送请求
W480.09 BOOL  ; 设备OEE状态有更新标志
W480.10 BOOL  ; 设备参数有更新标志
W480.11 BOOL  ; 进料位无料标志
W480.12 BOOL  ; MES采集漏率单位为mPa.m3/s(仪器显示值1000倍)
W480.15 BOOL  ; 设备在MES模式下运行
W481.00 BOOL  ; 前下料发送请求
W481.01 BOOL  ; 前下料机械手下料处理完成
W481.02 BOOL  ; 后下料发送请求
W481.03 BOOL  ; 后下料机械手下料处理完成
W481.05 BOOL  ; 氦检时间改变
W481.06 BOOL  ; 检口压力改变
W481.07 BOOL  ; 漏率改变
W481.08 BOOL  ; 注氦压力改变
W492.00 BOOL  ; NG位未满
W492.01 BOOL  ; NG传感器信号有空位
W492.03 BOOL  ; 扫码NG缓存有空位
W4.00 BOOL  ; 进料机构气缸感应器异常报警
W4.01 BOOL  ; 前上料机构气缸感应器异常报警
W4.02 BOOL  ; 前下料机构气缸感应器异常报警
W4.03 BOOL  ; 后上料机构气缸感应器异常报警
W4.04 BOOL  ; 后下料机构气缸感应器异常报警
W4.05 BOOL  ; 1#腔体机构气缸感应器异常报警
W4.06 BOOL  ; 2#腔体机构气缸感应器异常报警
W4.07 BOOL  ; 3#腔体机构气缸感应器异常报警
W4.08 BOOL  ; 4#腔体机构气缸感应器异常报警
W4.09 BOOL  ; 出料机构气缸感应器异常报警
W50 CHANNEL  ; PLC交互
W500.03 BOOL  ; ts3
W500.04 BOOL  ; 不允许往下放料标志
W500.05 BOOL  ; 停机
W500.06 BOOL  ; TS6
W500.07 BOOL  ; 输送带自动中
W500.09 BOOL  ; 扫码OK料已流走
W500.10 BOOL  ; 复位判断
W501.02 BOOL  ; 设备禁止启动
W501.03 BOOL  ; 安东系统断开设备停止报警
W501.04 BOOL  ; 弹屏
W501.05 BOOL  ; 设备允许启动
W502.00 BOOL  ; 未知原因按钮
W502.01 BOOL  ; 环境不满足
W502.02 BOOL  ; 样品制件
W502.03 BOOL  ; 盘点
W502.04 BOOL  ; 维护保养
W502.05 BOOL  ; 品种切换
W502.06 BOOL  ; 清洁检点
W502.07 BOOL  ; 培训
W502.08 BOOL  ; 等待物料
W502.09 BOOL  ; 交接班
W502.10 BOOL  ; 首件检查
W502.11 BOOL  ; 无生产计划
W502.12 BOOL  ; 品质异常
W502.13 BOOL  ; 物料更换
W502.14 BOOL  ; 来料异常
W502.15 BOOL  ; 现场岗位处理
W503.00 BOOL  ; 产能不匹配
W503.01 BOOL  ; 设备故障
W50.00 BOOL  ; 扫码完成信号->PC
W50.01 BOOL  ; #1模组放料->PC
W50.02 BOOL  ; #2模组放料->PC
W50.03 BOOL  ; #3模组放料->PC
W50.04 BOOL  ; #4模组放料->PC
W50.05 BOOL  ; 设备参数有更新标志
W510.01 BOOL  ; 开始扫码
W510.11 BOOL  ; TS
W5.14 BOOL  ; 弹出窗口报警中
W61.01 BOOL  ; 1腔OK料
W62.01 BOOL  ; 2腔OK料
W63.01 BOOL  ; 3腔OK料
W64.01 BOOL  ; 4腔OK料
W65.00 BOOL  ; 扫码
W65.01 BOOL  ; 左扫码完成
W65.02 BOOL  ; 扫码失败
W65.03 BOOL  ; 扫码OK
W65.04 BOOL  ; 左扫码开始
W65.10 BOOL  ; 扫码2(右扫码)
W65.11 BOOL  ; 右扫码完成
W65.12 BOOL  ; 右扫码失败
W65.13 BOOL  ; 右扫码-OK
W65.14 BOOL  ; 右扫码开始
W6.10 BOOL  ; 扫码2
W6.11 BOOL  ; 扫码忽略—HMI
W6.12 BOOL  ; 左扫码按钮(T)
W6.14 BOOL  ; 扫码NG清除-hmi
W6.15 BOOL  ; 测试NG清除-hmi
W70.00 BOOL  ; 上料前顶料下降回上料位辅助
W70.01 BOOL  ; 上料后顶料下降辅助
W80.00 BOOL  ; 自动重扫码
W8.00 BOOL  ; 自动状态-HMI
_Battery_Vacuum_01 VacuumPress_Convert
_Battery_Vacuum_02 VacuumPress_Convert
_Battery_Vacuum_03 VacuumPress_Convert
_Battery_Vacuum_04 VacuumPress_Convert
_SMC_ISE30A_Convert_01 SMC_ISE30A_Convert
_SMC_ISE30A_Convert_02 SMC_ISE30A_Convert
_SMC_ISE30A_Convert_03 SMC_ISE30A_Convert
_SMC_ISE30A_Convert_04 SMC_ISE30A_Convert

## Program Main (cyclic task 0)

### Section Main

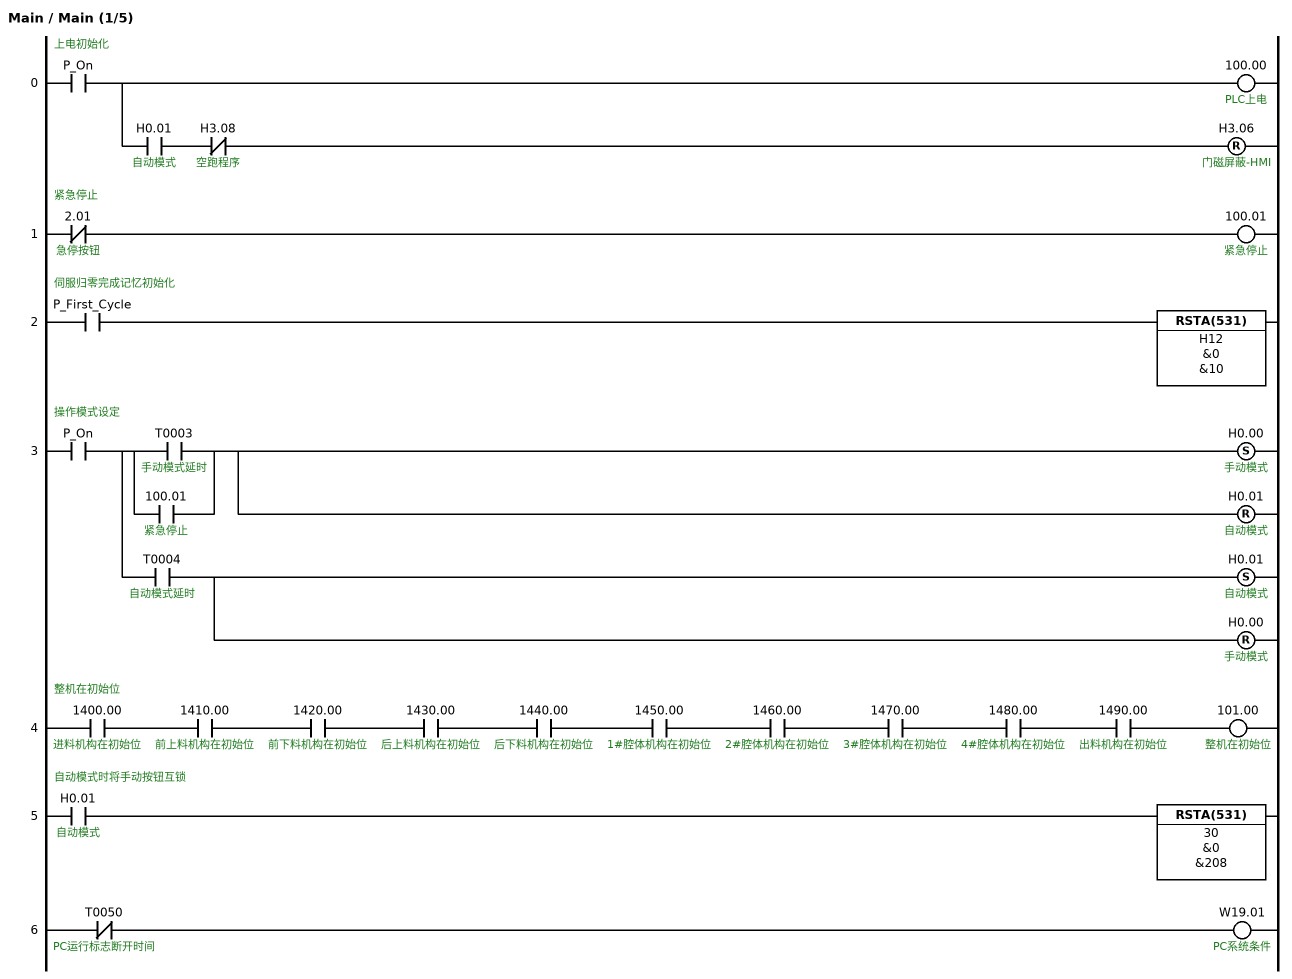
; rung 0: 上电初始化
LD P_On
OUT 100.00  ; PLC上电
AND H0.01  ; 自动模式
ANDNOT H3.08  ; 空跑程序
RSET H3.06  ; 门磁屏蔽-HMI
; rung 1: 紧急停止
LDNOT 2.01  ; 急停按钮
OUT 100.01  ; 紧急停止
; rung 2: 伺服归零完成记忆初始化
LD P_First_Cycle
RSTA(531) H12 &0 &10
; rung 3: 操作模式设定
LD P_On
OUT TR0
LD T0003  ; 手动模式延时
OR 100.01  ; 紧急停止
ANDLD
SET H0.00  ; 手动模式
RSET H0.01  ; 自动模式
LD TR0
AND T0004  ; 自动模式延时
SET H0.01  ; 自动模式
RSET H0.00  ; 手动模式
; rung 4: 整机在初始位
LD 1400.00  ; 进料机构在初始位
AND 1410.00  ; 前上料机构在初始位
AND 1420.00  ; 前下料机构在初始位
AND 1430.00  ; 后上料机构在初始位
AND 1440.00  ; 后下料机构在初始位
AND 1450.00  ; 1#腔体机构在初始位
AND 1460.00  ; 2#腔体机构在初始位
AND 1470.00  ; 3#腔体机构在初始位
AND 1480.00  ; 4#腔体机构在初始位
AND 1490.00  ; 出料机构在初始位
OUT 101.00  ; 整机在初始位
; rung 5: 自动模式时将手动按钮互锁
LD H0.01  ; 自动模式
RSTA(531) 30 &0 &208
; rung 6
LDNOT T0050  ; PC运行标志断开时间
OUT W19.01  ; PC系统条件

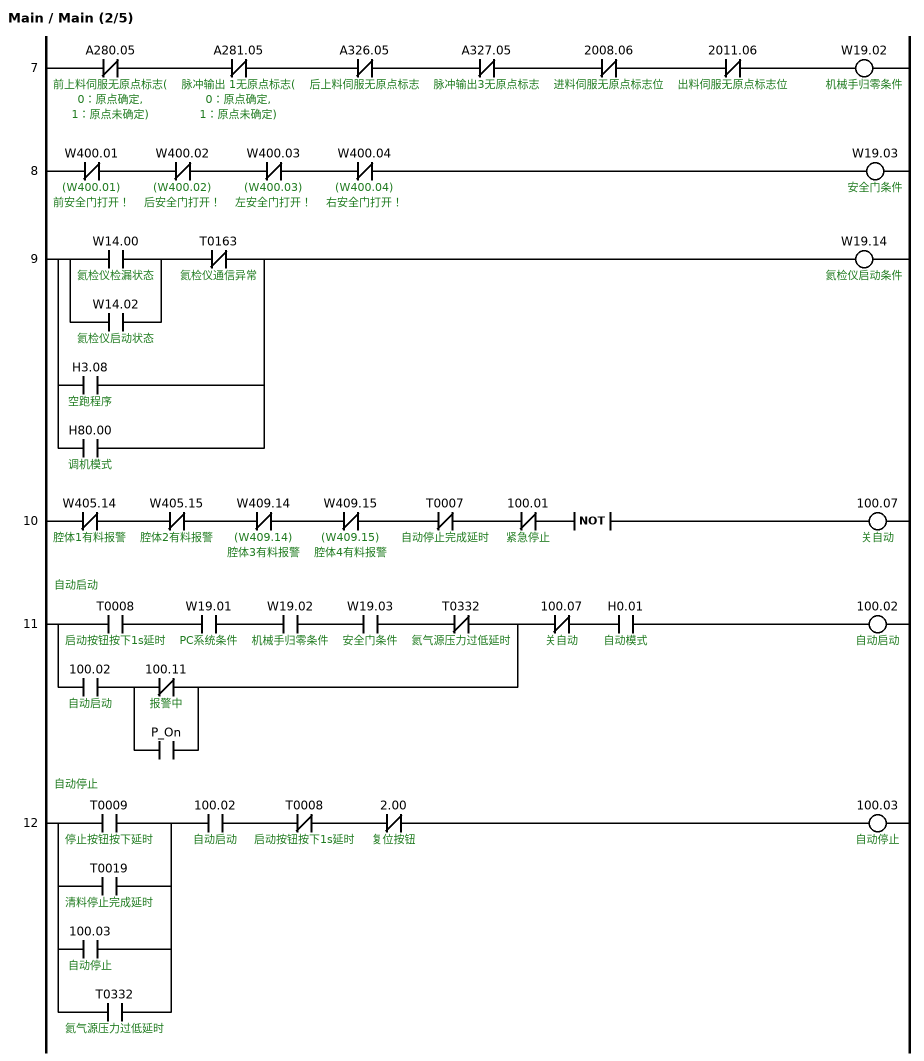
; rung 7
LDNOT A280.05  ; 前上料伺服无原点标志(0：原点确定,1：原点未确定)
ANDNOT A281.05  ; 脉冲输出 1无原点标志(0：原点确定,1：原点未确定)
ANDNOT A326.05  ; 后上料伺服无原点标志
ANDNOT A327.05  ; 脉冲输出3无原点标志
ANDNOT 2008.06  ; 进料伺服无原点标志位
ANDNOT 2011.06  ; 出料伺服无原点标志位
OUT W19.02  ; 机械手归零条件
; rung 8
LDNOT W400.01  ; (W400.01) 前安全门打开！
ANDNOT W400.02  ; (W400.02) 后安全门打开！
ANDNOT W400.03  ; (W400.03) 左安全门打开！
ANDNOT W400.04  ; (W400.04) 右安全门打开！
OUT W19.03  ; 安全门条件
; rung 9
LD W14.00  ; 氦检仪检漏状态
OR W14.02  ; 氦检仪启动状态
ANDNOT T0163  ; 氦检仪通信异常
OR H3.08  ; 空跑程序
OR H80.00  ; 调机模式
OUT W19.14  ; 氦检仪启动条件
; rung 10
LDNOT W405.14  ; 腔体1有料报警
ANDNOT W405.15  ; 腔体2有料报警
ANDNOT W409.14  ; (W409.14) 腔体3有料报警
ANDNOT W409.15  ; (W409.15) 腔体4有料报警
ANDNOT T0007  ; 自动停止完成延时
ANDNOT 100.01  ; 紧急停止
NOT(520)
OUT 100.07  ; 关自动
; rung 11: 自动启动
LD T0008  ; 启动按钮按下1s延时
AND W19.01  ; PC系统条件
AND W19.02  ; 机械手归零条件
AND W19.03  ; 安全门条件
ANDNOT T0332  ; 氦气源压力过低延时
LD 100.02  ; 自动启动
LDNOT 100.11  ; 报警中
OR P_On
ANDLD
ORLD
ANDNOT 100.07  ; 关自动
AND H0.01  ; 自动模式
OUT 100.02  ; 自动启动
; rung 12: 自动停止
LD T0009  ; 停止按钮按下延时
OR T0019  ; 清料停止完成延时
OR 100.03  ; 自动停止
OR T0332  ; 氦气源压力过低延时
AND 100.02  ; 自动启动
ANDNOT T0008  ; 启动按钮按下1s延时
ANDNOT 2.00  ; 复位按钮
OUT 100.03  ; 自动停止

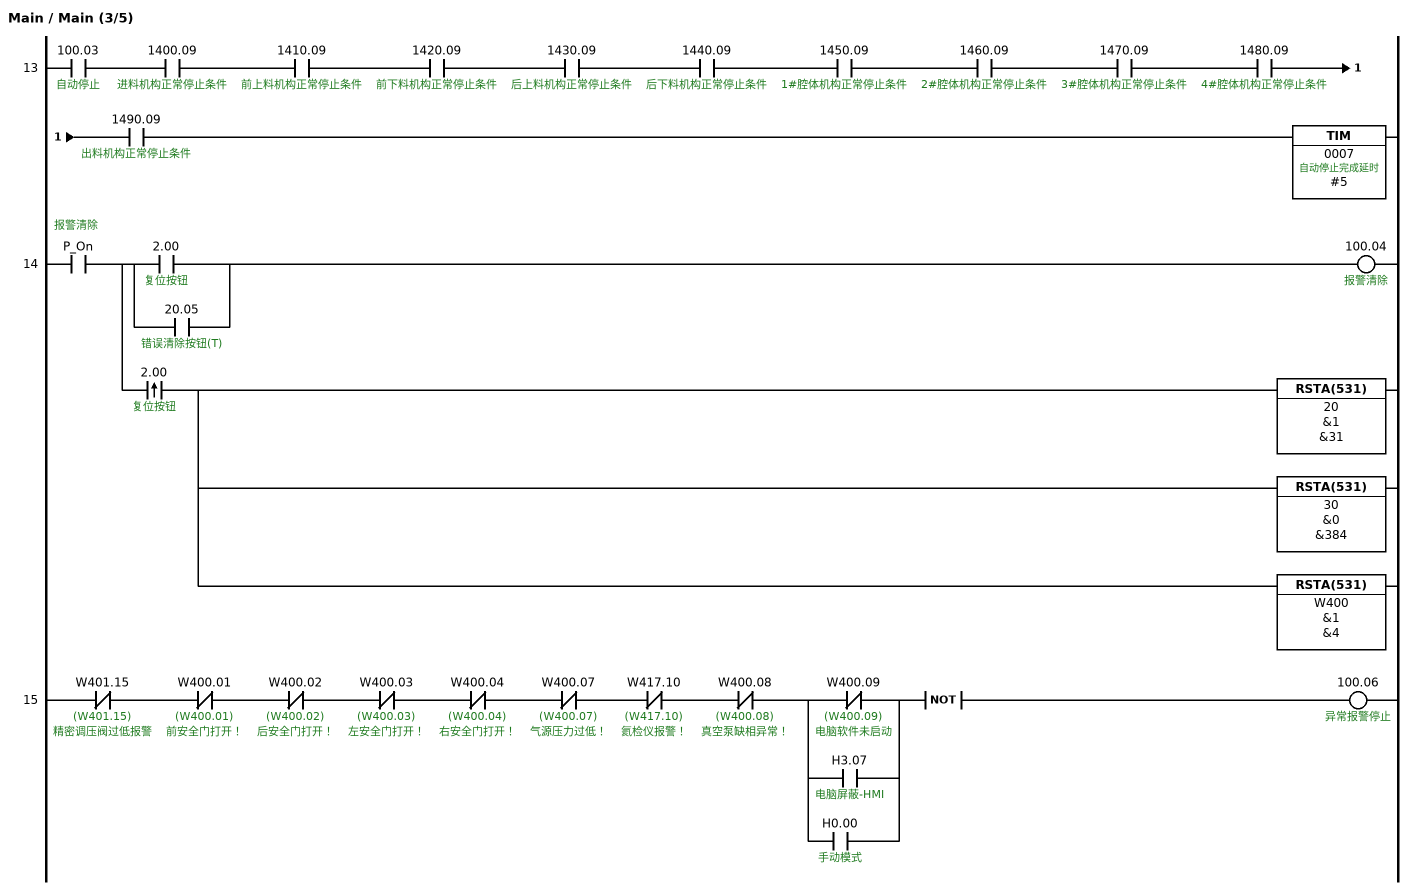
; rung 13
LD 100.03  ; 自动停止
AND 1400.09  ; 进料机构正常停止条件
AND 1410.09  ; 前上料机构正常停止条件
AND 1420.09  ; 前下料机构正常停止条件
AND 1430.09  ; 后上料机构正常停止条件
AND 1440.09  ; 后下料机构正常停止条件
AND 1450.09  ; 1#腔体机构正常停止条件
AND 1460.09  ; 2#腔体机构正常停止条件
AND 1470.09  ; 3#腔体机构正常停止条件
AND 1480.09  ; 4#腔体机构正常停止条件
AND 1490.09  ; 出料机构正常停止条件
TIM 0007 #5  ; 自动停止完成延时
; rung 14: 报警清除
LD P_On
OUT TR0
LD 2.00  ; 复位按钮
OR 20.05  ; 错误清除按钮(T)
ANDLD
OUT 100.04  ; 报警清除
LD TR0
@AND 2.00  ; 复位按钮
RSTA(531) 20 &1 &31
RSTA(531) 30 &0 &384
RSTA(531) W400 &1 &4
; rung 15
LDNOT W401.15  ; (W401.15) 精密调压阀过低报警
ANDNOT W400.01  ; (W400.01) 前安全门打开！
ANDNOT W400.02  ; (W400.02) 后安全门打开！
ANDNOT W400.03  ; (W400.03) 左安全门打开！
ANDNOT W400.04  ; (W400.04) 右安全门打开！
ANDNOT W400.07  ; (W400.07) 气源压力过低！
ANDNOT W417.10  ; (W417.10) 氦检仪报警！
ANDNOT W400.08  ; (W400.08) 真空泵缺相异常！
LDNOT W400.09  ; (W400.09) 电脑软件未启动
OR H3.07  ; 电脑屏蔽-HMI
OR H0.00  ; 手动模式
ANDLD
NOT(520)
OUT 100.06  ; 异常报警停止

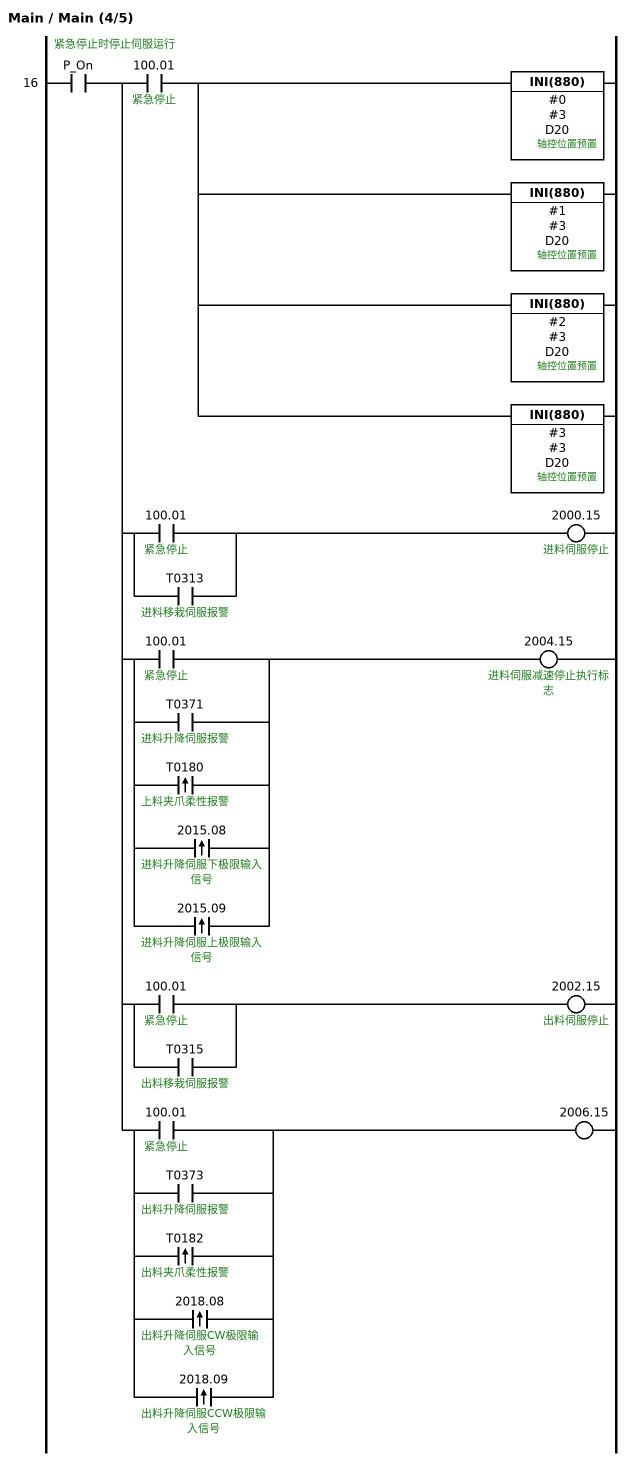
; rung 16: 紧急停止时停止伺服运行
LD P_On
OUT TR0
AND 100.01  ; 紧急停止
INI(880) #0 #3 D20  ; 轴控位置预置
INI(880) #1 #3 D20  ; 轴控位置预置
INI(880) #2 #3 D20  ; 轴控位置预置
INI(880) #3 #3 D20  ; 轴控位置预置
LD TR0
LD 100.01  ; 紧急停止
OR T0313  ; 进料移栽伺服报警
ANDLD
OUT 2000.15  ; 进料伺服停止
LD TR0
LD 100.01  ; 紧急停止
OR T0371  ; 进料升降伺服报警
@OR T0180  ; 上料夹爪柔性报警
@OR 2015.08  ; 进料升降伺服下极限输入信号
@OR 2015.09  ; 进料升降伺服上极限输入信号
ANDLD
OUT 2004.15  ; 进料伺服减速停止执行标志
LD TR0
LD 100.01  ; 紧急停止
OR T0315  ; 出料移栽伺服报警
ANDLD
OUT 2002.15  ; 出料伺服停止
LD TR0
LD 100.01  ; 紧急停止
OR T0373  ; 出料升降伺服报警
@OR T0182  ; 出料夹爪柔性报警
@OR 2018.08  ; 出料升降伺服CW极限输入信号
@OR 2018.09  ; 出料升降伺服CCW极限输入信号
ANDLD
OUT 2006.15

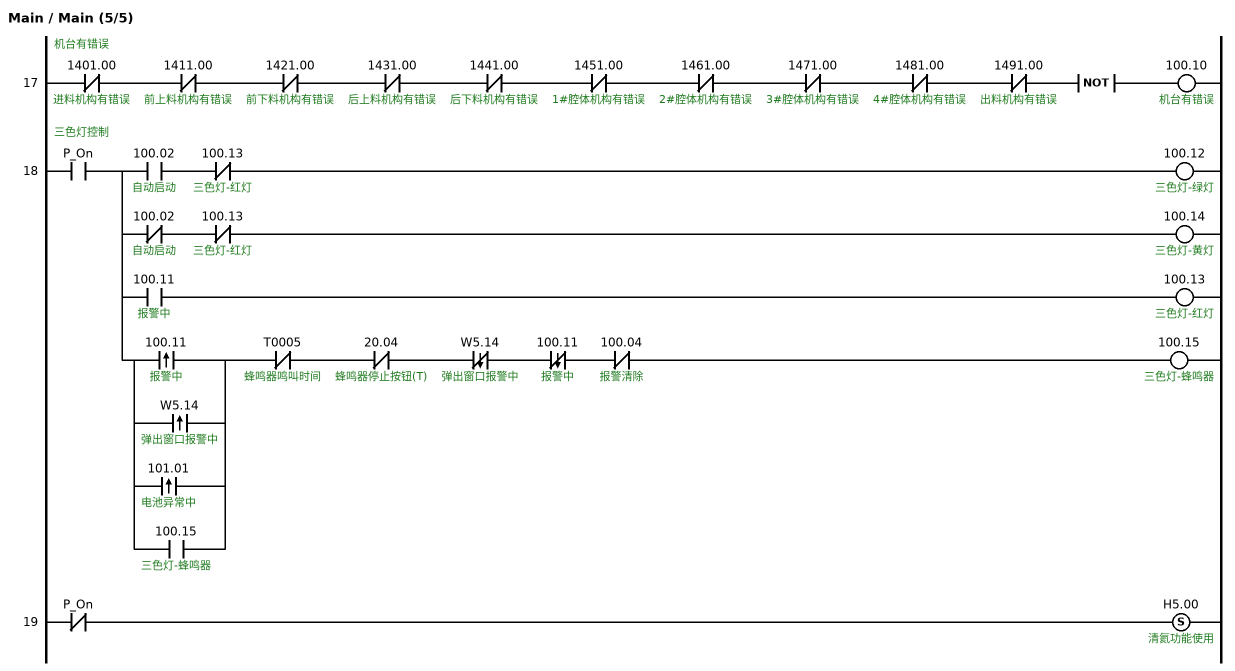
; rung 17: 机台有错误
LDNOT 1401.00  ; 进料机构有错误
ANDNOT 1411.00  ; 前上料机构有错误
ANDNOT 1421.00  ; 前下料机构有错误
ANDNOT 1431.00  ; 后上料机构有错误
ANDNOT 1441.00  ; 后下料机构有错误
ANDNOT 1451.00  ; 1#腔体机构有错误
ANDNOT 1461.00  ; 2#腔体机构有错误
ANDNOT 1471.00  ; 3#腔体机构有错误
ANDNOT 1481.00  ; 4#腔体机构有错误
ANDNOT 1491.00  ; 出料机构有错误
NOT(520)
OUT 100.10  ; 机台有错误
; rung 18: 三色灯控制
LD P_On
OUT TR0
AND 100.02  ; 自动启动
ANDNOT 100.13  ; 三色灯-红灯
OUT 100.12  ; 三色灯-绿灯
LD TR0
ANDNOT 100.02  ; 自动启动
ANDNOT 100.13  ; 三色灯-红灯
OUT 100.14  ; 三色灯-黄灯
LD TR0
AND 100.11  ; 报警中
OUT 100.13  ; 三色灯-红灯
LD TR0
@LD 100.11  ; 报警中
@OR W5.14  ; 弹出窗口报警中
@OR 101.01  ; 电池异常中
OR 100.15  ; 三色灯-蜂鸣器
ANDLD
ANDNOT T0005  ; 蜂鸣器鸣叫时间
ANDNOT 20.04  ; 蜂鸣器停止按钮(T)
%ANDNOT W5.14  ; 弹出窗口报警中
%ANDNOT 100.11  ; 报警中
ANDNOT 100.04  ; 报警清除
OUT 100.15  ; 三色灯-蜂鸣器
; rung 19
LDNOT P_On
SET H5.00  ; 清氦功能使用

### Section SCU21_1584_扫码

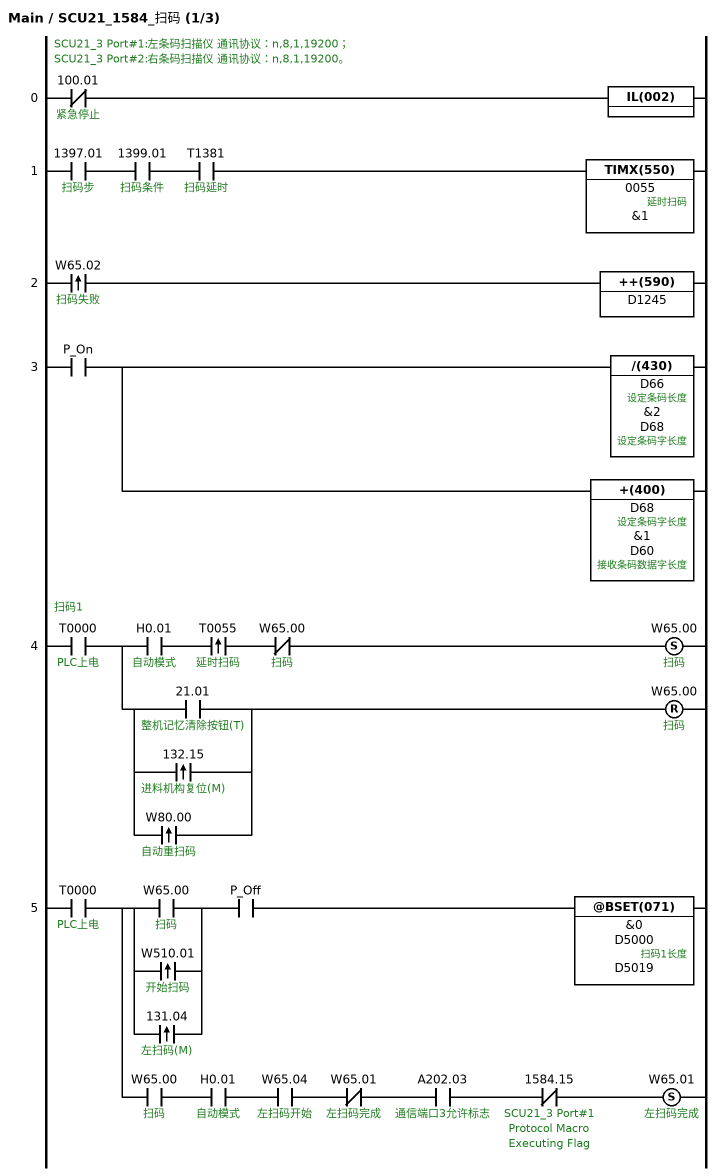
; rung 0: SCU21_3 Port#1:左条码扫描仪 通讯协议：n,8,1,19200； / SCU21_3 Port#2:右条码扫描仪 通讯协议：n,8,1,19200。
LDNOT 100.01  ; 紧急停止
IL(002)
; rung 1
LD 1397.01  ; 扫码步
AND 1399.01  ; 扫码条件
AND T1381  ; 扫码延时
TIMX(550) 0055 &1  ; 延时扫码
; rung 2
@LD W65.02  ; 扫码失败
++(590) D1245
; rung 3
LD P_On
/(430) D66 &2 D68  ; 设定条码长度, 设定条码字长度
+(400) D68 &1 D60  ; 设定条码字长度, 接收条码数据字长度
; rung 4: 扫码1
LD T0000  ; PLC上电
OUT TR0
AND H0.01  ; 自动模式
@AND T0055  ; 延时扫码
ANDNOT W65.00  ; 扫码
SET W65.00  ; 扫码
LD TR0
LD 21.01  ; 整机记忆清除按钮(T)
@OR 132.15  ; 进料机构复位(M)
@OR W80.00  ; 自动重扫码
ANDLD
RSET W65.00  ; 扫码
; rung 5
LD T0000  ; PLC上电
OUT TR0
LD W65.00  ; 扫码
@OR W510.01  ; 开始扫码
@OR 131.04  ; 左扫码(M)
ANDLD
AND P_Off
@BSET(071) &0 D5000 D5019  ; 扫码1长度
LD TR0
AND W65.00  ; 扫码
AND H0.01  ; 自动模式
AND W65.04  ; 左扫码开始
ANDNOT W65.01  ; 左扫码完成
AND A202.03  ; 通信端口3允许标志
ANDNOT 1584.15  ; SCU21_3 Port#1 Protocol Macro Executing Flag
SET W65.01  ; 左扫码完成

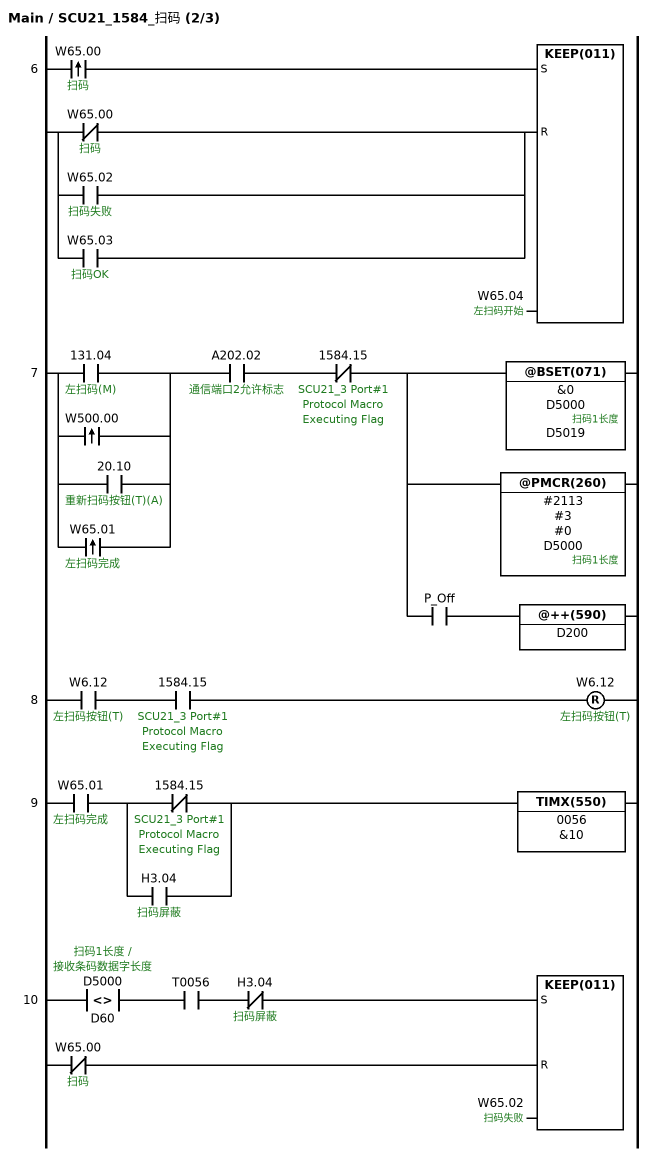
; rung 6
@LD W65.00  ; 扫码
LDNOT W65.00  ; 扫码
OR W65.02  ; 扫码失败
OR W65.03  ; 扫码OK
KEEP(011) W65.04  ; 左扫码开始
; rung 7
LD 131.04  ; 左扫码(M)
@OR W500.00
OR 20.10  ; 重新扫码按钮(T)(A)
@OR W65.01  ; 左扫码完成
AND A202.02  ; 通信端口2允许标志
ANDNOT 1584.15  ; SCU21_3 Port#1 Protocol Macro Executing Flag
@BSET(071) &0 D5000 D5019  ; 扫码1长度
@PMCR(260) #2113 #3 #0 D5000  ; 扫码1长度
AND P_Off
@++(590) D200
; rung 8
LD W6.12  ; 左扫码按钮(T)
AND 1584.15  ; SCU21_3 Port#1 Protocol Macro Executing Flag
RSET W6.12  ; 左扫码按钮(T)
; rung 9
LD W65.01  ; 左扫码完成
LDNOT 1584.15  ; SCU21_3 Port#1 Protocol Macro Executing Flag
OR H3.04  ; 扫码屏蔽
ANDLD
TIMX(550) 0056 &10
; rung 10
LD<>(305) D5000 D60  ; 扫码1长度, 接收条码数据字长度
AND T0056
ANDNOT H3.04  ; 扫码屏蔽
LDNOT W65.00  ; 扫码
KEEP(011) W65.02  ; 扫码失败

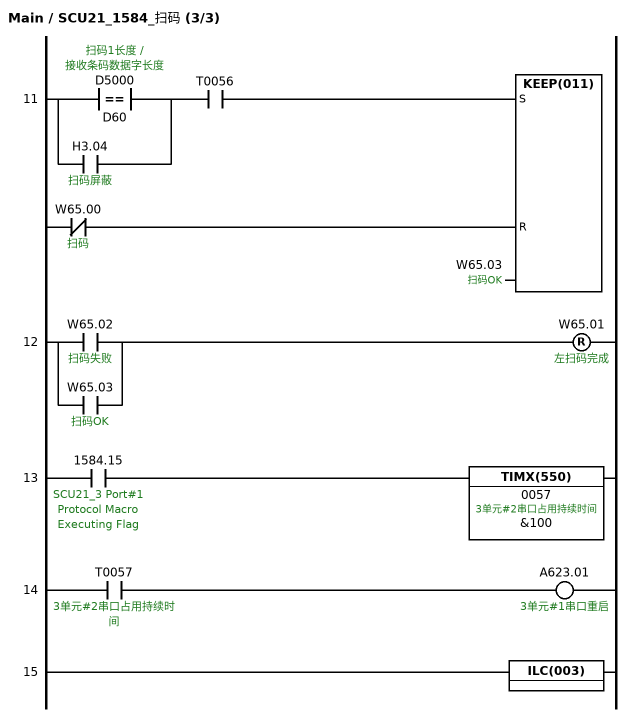
; rung 11
LD=(300) D5000 D60  ; 扫码1长度, 接收条码数据字长度
OR H3.04  ; 扫码屏蔽
AND T0056
LDNOT W65.00  ; 扫码
KEEP(011) W65.03  ; 扫码OK
; rung 12
LD W65.02  ; 扫码失败
OR W65.03  ; 扫码OK
RSET W65.01  ; 左扫码完成
; rung 13
LD 1584.15  ; SCU21_3 Port#1 Protocol Macro Executing Flag
TIMX(550) 0057 &100  ; 3单元#2串口占用持续时间
; rung 14
LD T0057  ; 3单元#2串口占用持续时间
OUT A623.01  ; 3单元#1串口重启
; rung 15
ILC(003)

### Section SCU21_1594_氦检仪

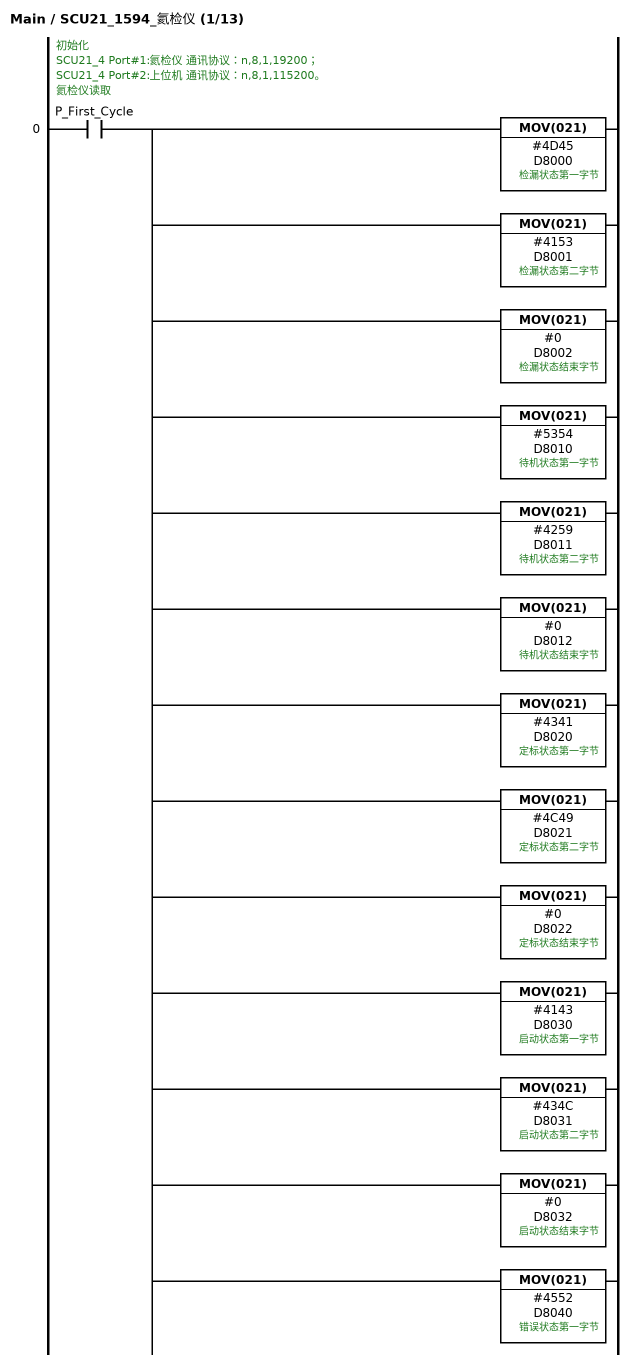

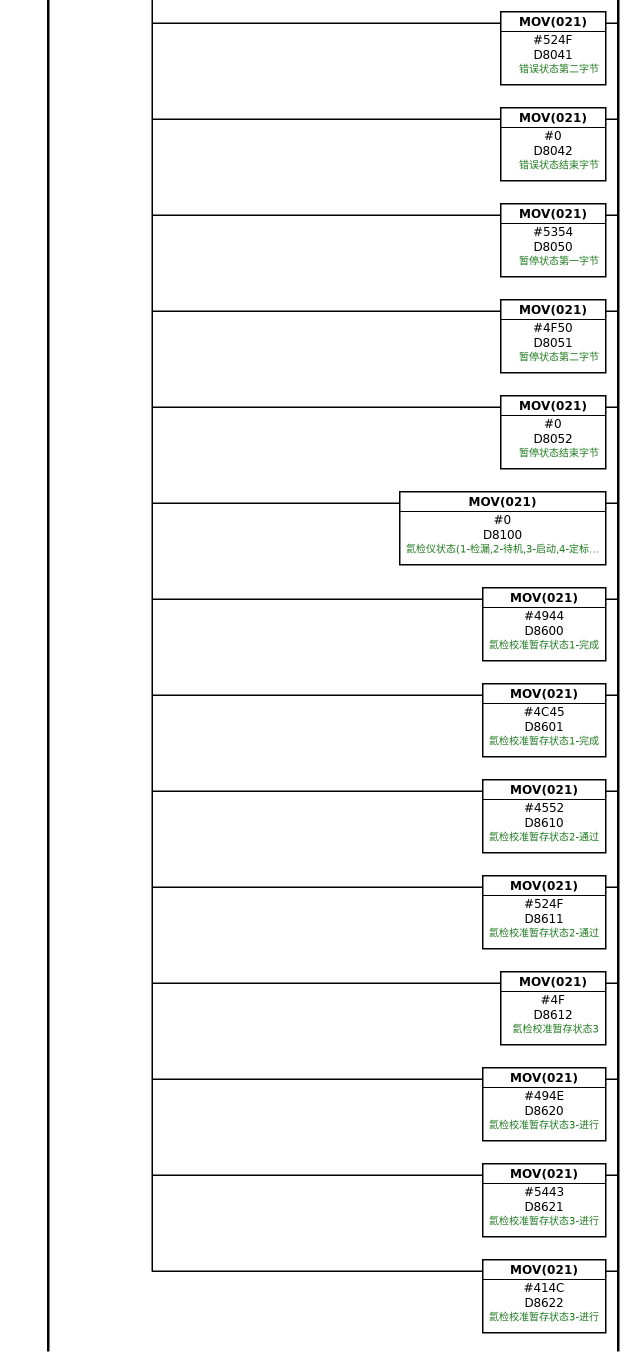
; rung 0: 初始化 / SCU21_4 Port#1:氦检仪 通讯协议：n,8,1,19200； / SCU21_4 Port#2:上位机 通讯协议：n,8,1,115200。 / 氦检仪读取
LD P_First_Cycle
MOV(021) #4D45 D8000  ; 检漏状态第一字节
MOV(021) #4153 D8001  ; 检漏状态第二字节
MOV(021) #0 D8002  ; 检漏状态结束字节
MOV(021) #5354 D8010  ; 待机状态第一字节
MOV(021) #4259 D8011  ; 待机状态第二字节
MOV(021) #0 D8012  ; 待机状态结束字节
MOV(021) #4341 D8020  ; 定标状态第一字节
MOV(021) #4C49 D8021  ; 定标状态第二字节
MOV(021) #0 D8022  ; 定标状态结束字节
MOV(021) #4143 D8030  ; 启动状态第一字节
MOV(021) #434C D8031  ; 启动状态第二字节
MOV(021) #0 D8032  ; 启动状态结束字节
MOV(021) #4552 D8040  ; 错误状态第一字节
MOV(021) #524F D8041  ; 错误状态第二字节
MOV(021) #0 D8042  ; 错误状态结束字节
MOV(021) #5354 D8050  ; 暂停状态第一字节
MOV(021) #4F50 D8051  ; 暂停状态第二字节
MOV(021) #0 D8052  ; 暂停状态结束字节
MOV(021) #0 D8100  ; 氦检仪状态(1-检漏,2-待机,3-启动,4-定标,5-错误,6-暂停)
MOV(021) #4944 D8600  ; 氦检校准暂存状态1-完成
MOV(021) #4C45 D8601  ; 氦检校准暂存状态1-完成
MOV(021) #4552 D8610  ; 氦检校准暂存状态2-通过
MOV(021) #524F D8611  ; 氦检校准暂存状态2-通过
MOV(021) #4F D8612  ; 氦检校准暂存状态3
MOV(021) #494E D8620  ; 氦检校准暂存状态3-进行
MOV(021) #5443 D8621  ; 氦检校准暂存状态3-进行
MOV(021) #414C D8622  ; 氦检校准暂存状态3-进行

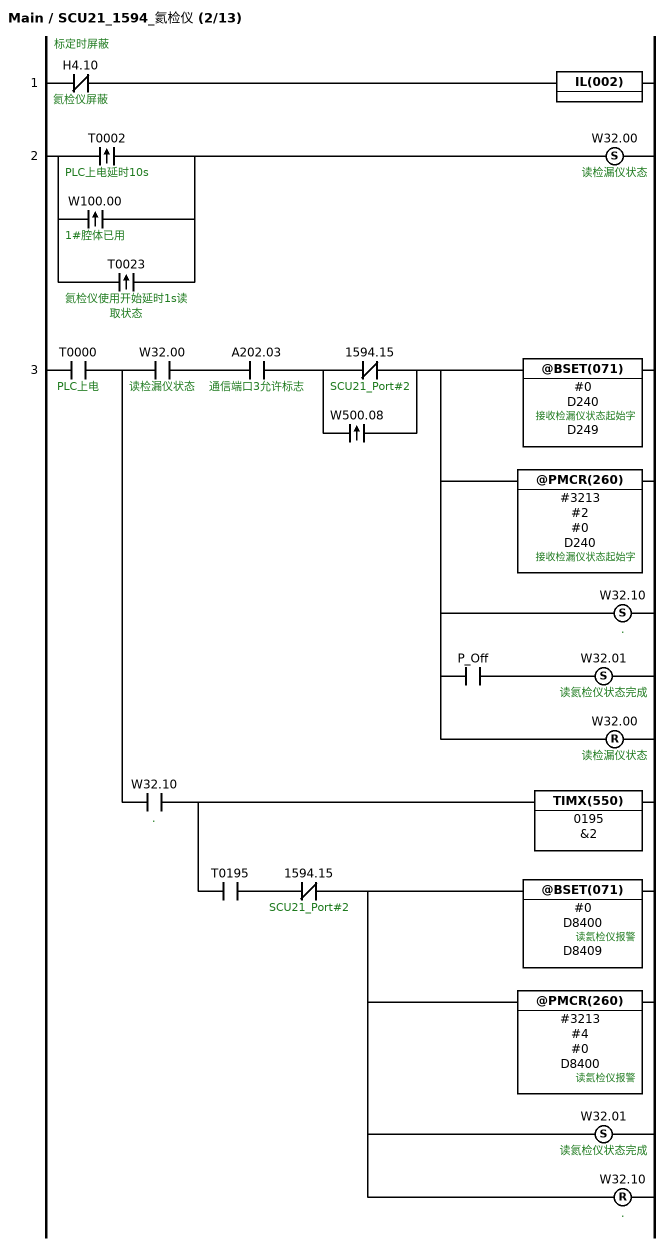
; rung 1: 标定时屏蔽
LDNOT H4.10  ; 氦检仪屏蔽
IL(002)
; rung 2
@LD T0002  ; PLC上电延时10s
@OR W100.00  ; 1#腔体已用
@OR T0023  ; 氦检仪使用开始延时1s读取状态
SET W32.00  ; 读检漏仪状态
; rung 3
LD T0000  ; PLC上电
OUT TR0
AND W32.00  ; 读检漏仪状态
AND A202.03  ; 通信端口3允许标志
LDNOT 1594.15  ; SCU21_Port#2
@OR W500.08
ANDLD
OUT TR1
@BSET(071) #0 D240 D249  ; 接收检漏仪状态起始字
@PMCR(260) #3213 #2 #0 D240  ; 接收检漏仪状态起始字
SET W32.10  ; .
AND P_Off
SET W32.01  ; 读氦检仪状态完成
LD TR1
RSET W32.00  ; 读检漏仪状态
LD TR0
AND W32.10  ; .
TIMX(550) 0195 &2
AND T0195
ANDNOT 1594.15  ; SCU21_Port#2
@BSET(071) #0 D8400 D8409  ; 读氦检仪报警
@PMCR(260) #3213 #4 #0 D8400  ; 读氦检仪报警
SET W32.01  ; 读氦检仪状态完成
RSET W32.10  ; .

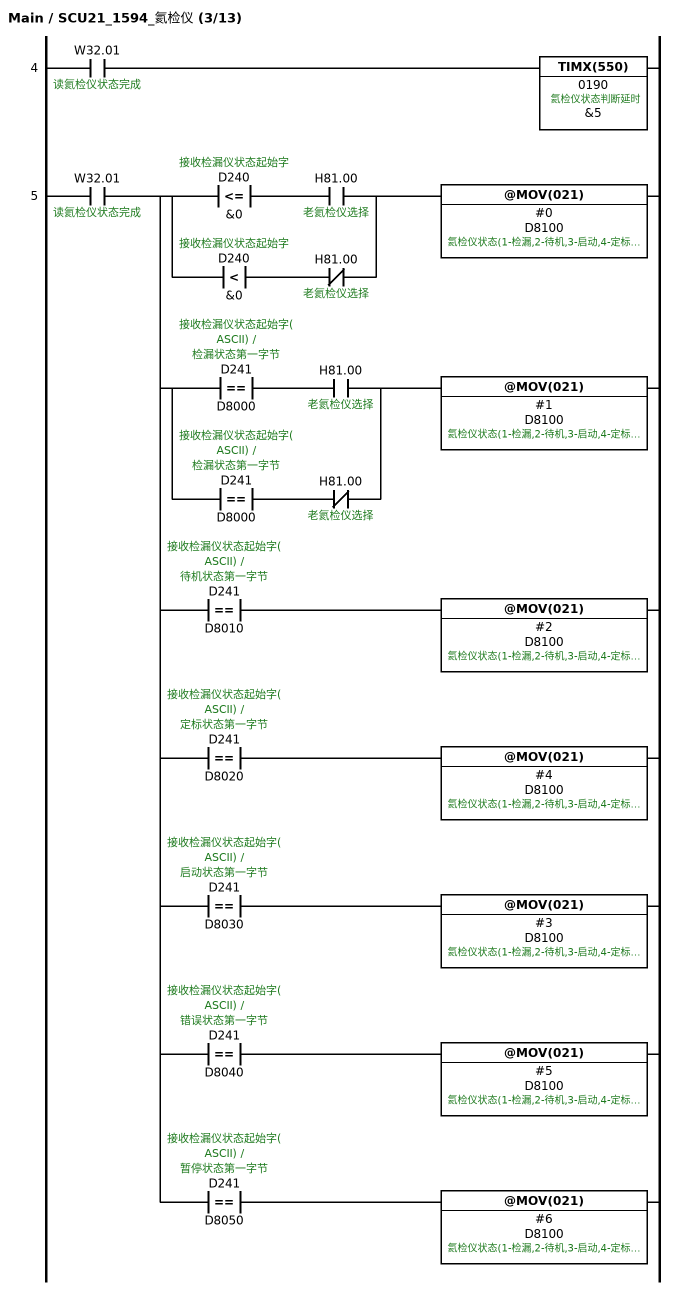
; rung 4
LD W32.01  ; 读氦检仪状态完成
TIMX(550) 0190 &5  ; 氦检仪状态判断延时
; rung 5
LD W32.01  ; 读氦检仪状态完成
OUT TR0
LD<=(315) D240 &0  ; 接收检漏仪状态起始字
AND H81.00  ; 老氦检仪选择
LD<(310) D240 &0  ; 接收检漏仪状态起始字
ANDNOT H81.00  ; 老氦检仪选择
ORLD
ANDLD
@MOV(021) #0 D8100  ; 氦检仪状态(1-检漏,2-待机,3-启动,4-定标,5-错误,6-暂停)
LD TR0
LD=$(670) D241 D8000  ; 接收检漏仪状态起始字(ASCII), 检漏状态第一字节
AND H81.00  ; 老氦检仪选择
LD=(300) D241 D8000  ; 接收检漏仪状态起始字(ASCII), 检漏状态第一字节
ANDNOT H81.00  ; 老氦检仪选择
ORLD
ANDLD
@MOV(021) #1 D8100  ; 氦检仪状态(1-检漏,2-待机,3-启动,4-定标,5-错误,6-暂停)
LD TR0
AND=$(670) D241 D8010  ; 接收检漏仪状态起始字(ASCII), 待机状态第一字节
@MOV(021) #2 D8100  ; 氦检仪状态(1-检漏,2-待机,3-启动,4-定标,5-错误,6-暂停)
LD TR0
AND=$(670) D241 D8020  ; 接收检漏仪状态起始字(ASCII), 定标状态第一字节
@MOV(021) #4 D8100  ; 氦检仪状态(1-检漏,2-待机,3-启动,4-定标,5-错误,6-暂停)
LD TR0
AND=$(670) D241 D8030  ; 接收检漏仪状态起始字(ASCII), 启动状态第一字节
@MOV(021) #3 D8100  ; 氦检仪状态(1-检漏,2-待机,3-启动,4-定标,5-错误,6-暂停)
LD TR0
AND=$(670) D241 D8040  ; 接收检漏仪状态起始字(ASCII), 错误状态第一字节
@MOV(021) #5 D8100  ; 氦检仪状态(1-检漏,2-待机,3-启动,4-定标,5-错误,6-暂停)
LD TR0
AND=$(670) D241 D8050  ; 接收检漏仪状态起始字(ASCII), 暂停状态第一字节
@MOV(021) #6 D8100  ; 氦检仪状态(1-检漏,2-待机,3-启动,4-定标,5-错误,6-暂停)

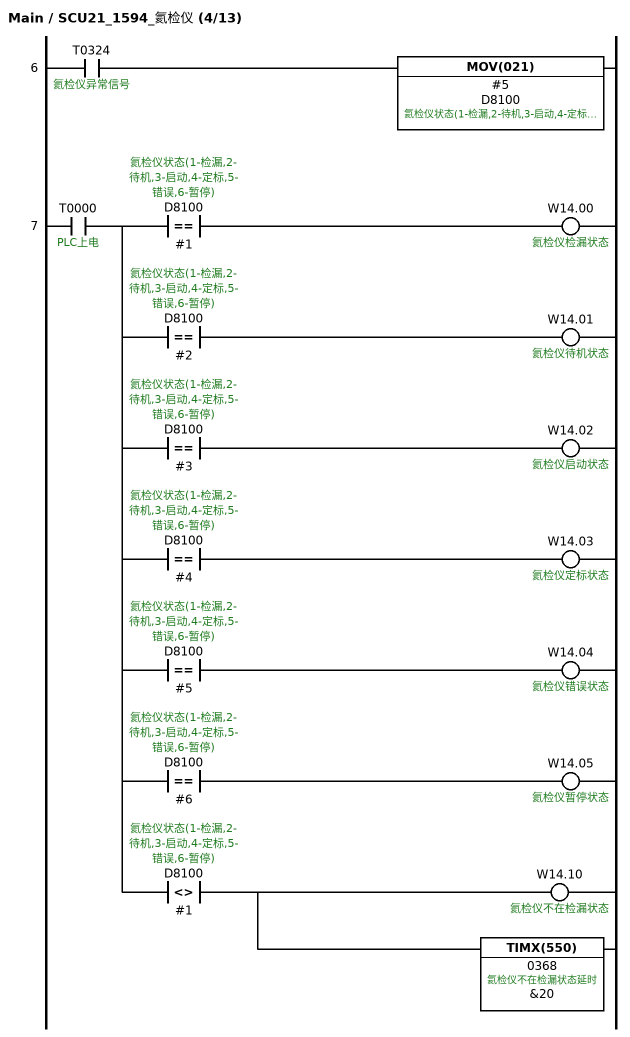
; rung 6
LD T0324  ; 氦检仪异常信号
MOV(021) #5 D8100  ; 氦检仪状态(1-检漏,2-待机,3-启动,4-定标,5-错误,6-暂停)
; rung 7
LD T0000  ; PLC上电
OUT TR0
AND=(300) D8100 #1  ; 氦检仪状态(1-检漏,2-待机,3-启动,4-定标,5-错误,6-暂停)
OUT W14.00  ; 氦检仪检漏状态
LD TR0
AND=(300) D8100 #2  ; 氦检仪状态(1-检漏,2-待机,3-启动,4-定标,5-错误,6-暂停)
OUT W14.01  ; 氦检仪待机状态
LD TR0
AND=(300) D8100 #3  ; 氦检仪状态(1-检漏,2-待机,3-启动,4-定标,5-错误,6-暂停)
OUT W14.02  ; 氦检仪启动状态
LD TR0
AND=(300) D8100 #4  ; 氦检仪状态(1-检漏,2-待机,3-启动,4-定标,5-错误,6-暂停)
OUT W14.03  ; 氦检仪定标状态
LD TR0
AND=(300) D8100 #5  ; 氦检仪状态(1-检漏,2-待机,3-启动,4-定标,5-错误,6-暂停)
OUT W14.04  ; 氦检仪错误状态
LD TR0
AND=(300) D8100 #6  ; 氦检仪状态(1-检漏,2-待机,3-启动,4-定标,5-错误,6-暂停)
OUT W14.05  ; 氦检仪暂停状态
LD TR0
AND<>(305) D8100 #1  ; 氦检仪状态(1-检漏,2-待机,3-启动,4-定标,5-错误,6-暂停)
OUT W14.10  ; 氦检仪不在检漏状态
TIMX(550) 0368 &20  ; 氦检仪不在检漏状态延时

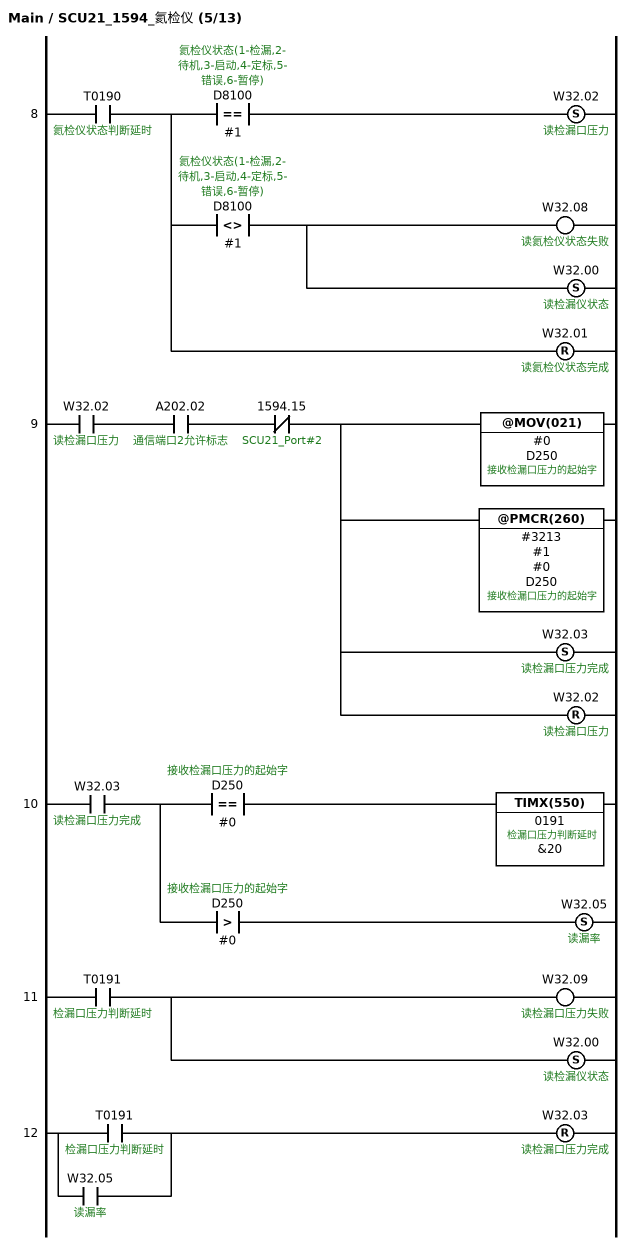
; rung 8
LD T0190  ; 氦检仪状态判断延时
OUT TR0
AND=(300) D8100 #1  ; 氦检仪状态(1-检漏,2-待机,3-启动,4-定标,5-错误,6-暂停)
SET W32.02  ; 读检漏口压力
LD TR0
AND<>(305) D8100 #1  ; 氦检仪状态(1-检漏,2-待机,3-启动,4-定标,5-错误,6-暂停)
OUT W32.08  ; 读氦检仪状态失败
SET W32.00  ; 读检漏仪状态
LD TR0
RSET W32.01  ; 读氦检仪状态完成
; rung 9
LD W32.02  ; 读检漏口压力
AND A202.02  ; 通信端口2允许标志
ANDNOT 1594.15  ; SCU21_Port#2
@MOV(021) #0 D250  ; 接收检漏口压力的起始字
@PMCR(260) #3213 #1 #0 D250  ; 接收检漏口压力的起始字
SET W32.03  ; 读检漏口压力完成
RSET W32.02  ; 读检漏口压力
; rung 10
LD W32.03  ; 读检漏口压力完成
OUT TR0
AND=(300) D250 #0  ; 接收检漏口压力的起始字
TIMX(550) 0191 &20  ; 检漏口压力判断延时
LD TR0
AND>(320) D250 #0  ; 接收检漏口压力的起始字
SET W32.05  ; 读漏率
; rung 11
LD T0191  ; 检漏口压力判断延时
OUT W32.09  ; 读检漏口压力失败
SET W32.00  ; 读检漏仪状态
; rung 12
LD T0191  ; 检漏口压力判断延时
OR W32.05  ; 读漏率
RSET W32.03  ; 读检漏口压力完成

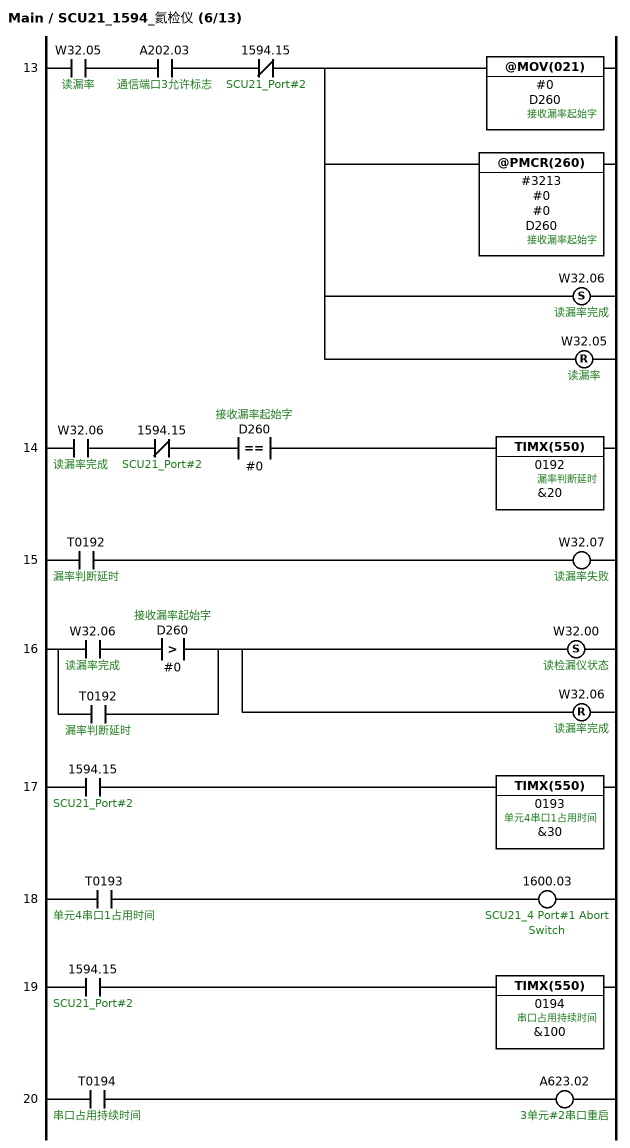
; rung 13
LD W32.05  ; 读漏率
AND A202.03  ; 通信端口3允许标志
ANDNOT 1594.15  ; SCU21_Port#2
@MOV(021) #0 D260  ; 接收漏率起始字
@PMCR(260) #3213 #0 #0 D260  ; 接收漏率起始字
SET W32.06  ; 读漏率完成
RSET W32.05  ; 读漏率
; rung 14
LD W32.06  ; 读漏率完成
ANDNOT 1594.15  ; SCU21_Port#2
AND=(300) D260 #0  ; 接收漏率起始字
TIMX(550) 0192 &20  ; 漏率判断延时
; rung 15
LD T0192  ; 漏率判断延时
OUT W32.07  ; 读漏率失败
; rung 16
LD W32.06  ; 读漏率完成
AND>(320) D260 #0  ; 接收漏率起始字
OR T0192  ; 漏率判断延时
SET W32.00  ; 读检漏仪状态
RSET W32.06  ; 读漏率完成
; rung 17
LD 1594.15  ; SCU21_Port#2
TIMX(550) 0193 &30  ; 单元4串口1占用时间
; rung 18
LD T0193  ; 单元4串口1占用时间
OUT 1600.03  ; SCU21_4 Port#1 Abort Switch
; rung 19
LD 1594.15  ; SCU21_Port#2
TIMX(550) 0194 &100  ; 串口占用持续时间
; rung 20
LD T0194  ; 串口占用持续时间
OUT A623.02  ; 3单元#2串口重启

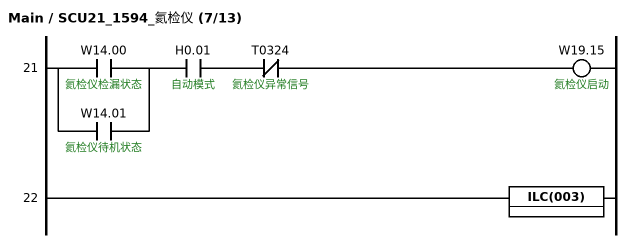
; rung 21
LD W14.00  ; 氦检仪检漏状态
OR W14.01  ; 氦检仪待机状态
AND H0.01  ; 自动模式
ANDNOT T0324  ; 氦检仪异常信号
OUT W19.15  ; 氦检仪启动
; rung 22
ILC(003)

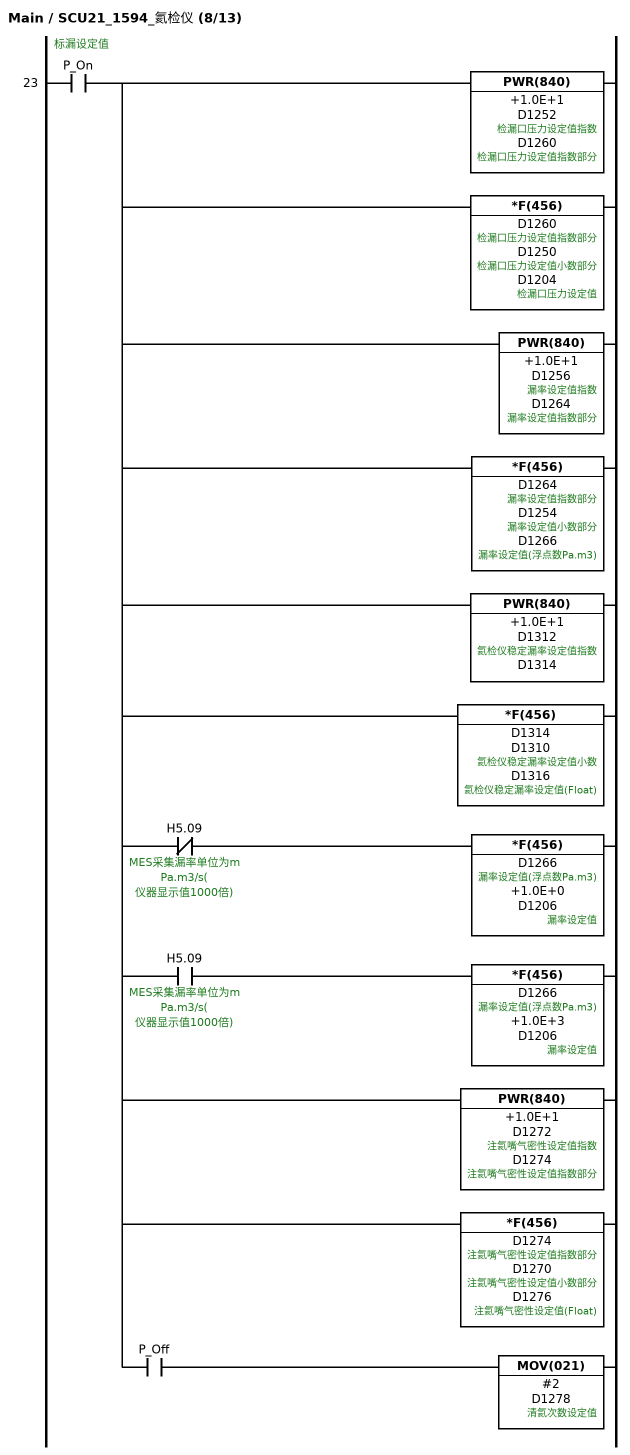
; rung 23: 标漏设定值
LD P_On
OUT TR0
PWR(840) +1.0E+1 D1252 D1260  ; 检漏口压力设定值指数, 检漏口压力设定值指数部分
*F(456) D1260 D1250 D1204  ; 检漏口压力设定值指数部分, 检漏口压力设定值小数部分, 检漏口压力设定值
PWR(840) +1.0E+1 D1256 D1264  ; 漏率设定值指数, 漏率设定值指数部分
*F(456) D1264 D1254 D1266  ; 漏率设定值指数部分, 漏率设定值小数部分, 漏率设定值(浮点数Pa.m3)
PWR(840) +1.0E+1 D1312 D1314  ; 氦检仪稳定漏率设定值指数
*F(456) D1314 D1310 D1316  ; 氦检仪稳定漏率设定值小数, 氦检仪稳定漏率设定值(Float)
ANDNOT H5.09  ; MES采集漏率单位为mPa.m3/s(仪器显示值1000倍)
*F(456) D1266 +1.0E+0 D1206  ; 漏率设定值(浮点数Pa.m3), 漏率设定值
LD TR0
AND H5.09  ; MES采集漏率单位为mPa.m3/s(仪器显示值1000倍)
*F(456) D1266 +1.0E+3 D1206  ; 漏率设定值(浮点数Pa.m3), 漏率设定值
LD TR0
PWR(840) +1.0E+1 D1272 D1274  ; 注氦嘴气密性设定值指数, 注氦嘴气密性设定值指数部分
*F(456) D1274 D1270 D1276  ; 注氦嘴气密性设定值指数部分, 注氦嘴气密性设定值小数部分, 注氦嘴气密性设定值(Float)
AND P_Off
MOV(021) #2 D1278  ; 清氦次数设定值

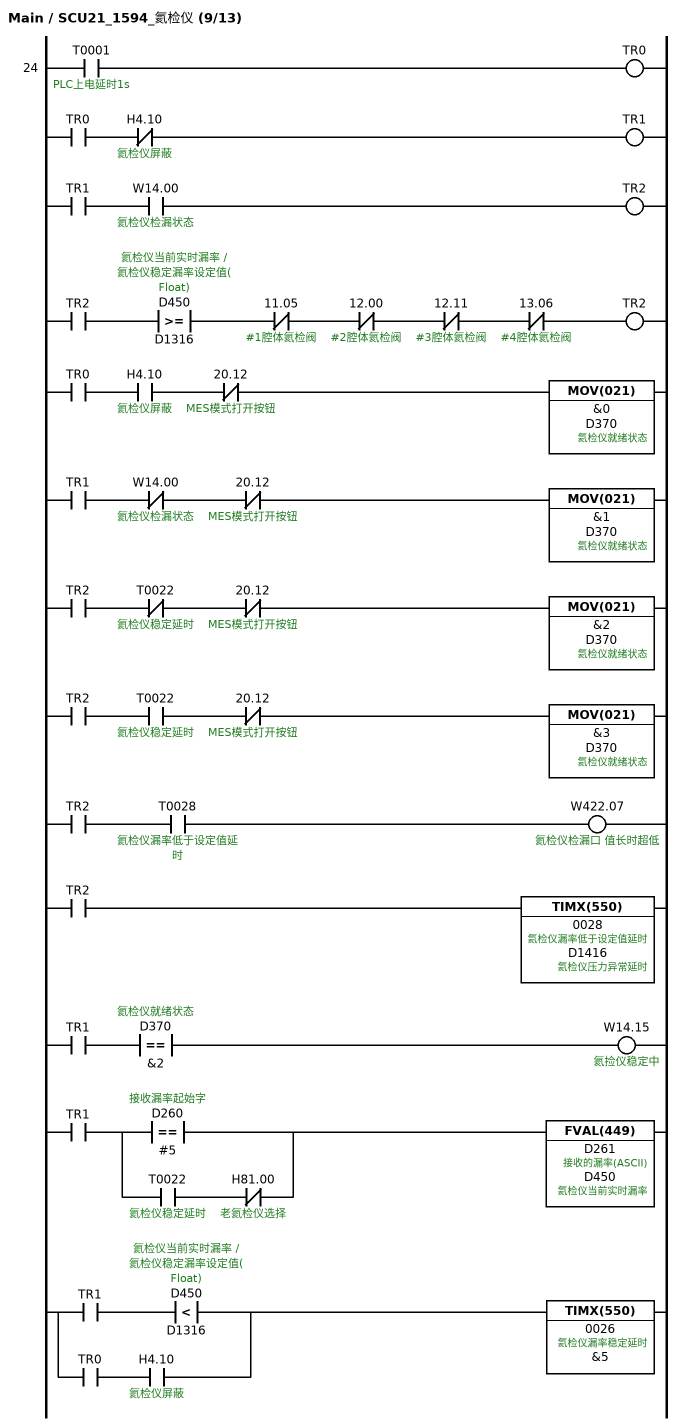
; rung 24
LD T0001  ; PLC上电延时1s
OUT TR0
AND H4.10  ; 氦检仪屏蔽
ANDNOT 20.12  ; MES模式打开按钮
MOV(021) &0 D370  ; 氦检仪就绪状态
LD TR0
ANDNOT H4.10  ; 氦检仪屏蔽
OUT TR1
ANDNOT W14.00  ; 氦检仪检漏状态
ANDNOT 20.12  ; MES模式打开按钮
MOV(021) &1 D370  ; 氦检仪就绪状态
LD TR1
AND W14.00  ; 氦检仪检漏状态
OUT TR2
ANDNOT T0022  ; 氦检仪稳定延时
ANDNOT 20.12  ; MES模式打开按钮
MOV(021) &2 D370  ; 氦检仪就绪状态
LD TR2
AND T0022  ; 氦检仪稳定延时
ANDNOT 20.12  ; MES模式打开按钮
MOV(021) &3 D370  ; 氦检仪就绪状态
LD TR2
AND>=F(334) D450 D1316  ; 氦检仪当前实时漏率, 氦检仪稳定漏率设定值(Float)
ANDNOT 11.05  ; #1腔体氦检阀
ANDNOT 12.00  ; #2腔体氦检阀
ANDNOT 12.11  ; #3腔体氦检阀
ANDNOT 13.06  ; #4腔体氦检阀
OUT TR2
AND T0028  ; 氦检仪漏率低于设定值延时
OUT W422.07  ; 氦检仪检漏口 值长时超低
LD TR2
TIMX(550) 0028 D1416  ; 氦检仪压力异常延时, 氦检仪漏率低于设定值延时
LD TR1
AND=(300) D370 &2  ; 氦检仪就绪状态
OUT W14.15  ; 氦捡仪稳定中
LD TR1
LD=(300) D260 #5  ; 接收漏率起始字
LD T0022  ; 氦检仪稳定延时
ANDNOT H81.00  ; 老氦检仪选择
ORLD
ANDLD
FVAL(449) D261 D450  ; 接收的漏率(ASCII), 氦检仪当前实时漏率
LD TR1
AND<F(331) D450 D1316  ; 氦检仪当前实时漏率, 氦检仪稳定漏率设定值(Float)
LD TR0
AND H4.10  ; 氦检仪屏蔽
ORLD
TIMX(550) 0026 &5  ; 氦检仪漏率稳定延时

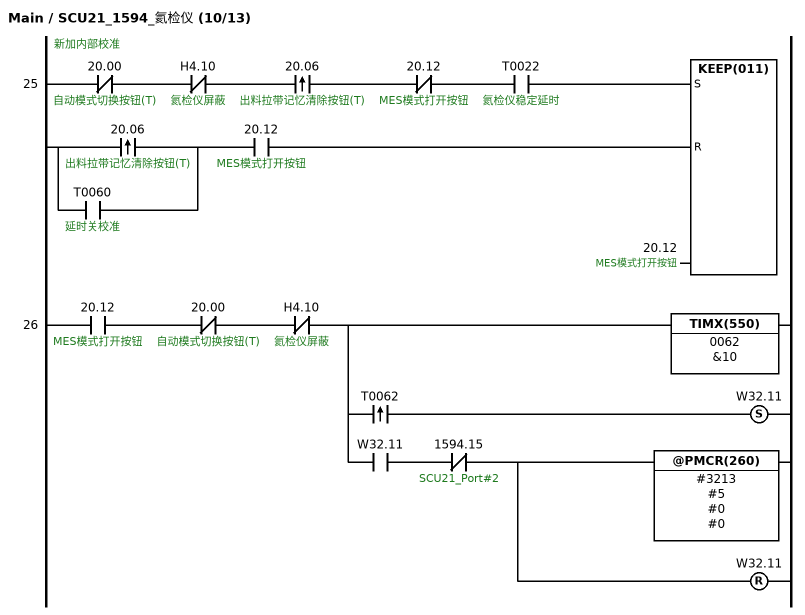
; rung 25: 新加内部校准
LDNOT 20.00  ; 自动模式切换按钮(T)
ANDNOT H4.10  ; 氦检仪屏蔽
@AND 20.06  ; 出料拉带记忆清除按钮(T)
ANDNOT 20.12  ; MES模式打开按钮
AND T0022  ; 氦检仪稳定延时
@LD 20.06  ; 出料拉带记忆清除按钮(T)
OR T0060  ; 延时关校准
AND 20.12  ; MES模式打开按钮
KEEP(011) 20.12  ; MES模式打开按钮
; rung 26
LD 20.12  ; MES模式打开按钮
ANDNOT 20.00  ; 自动模式切换按钮(T)
ANDNOT H4.10  ; 氦检仪屏蔽
OUT TR0
TIMX(550) 0062 &10
@AND T0062
SET W32.11
LD TR0
AND W32.11
ANDNOT 1594.15  ; SCU21_Port#2
@PMCR(260) #3213 #5 #0 #0
RSET W32.11

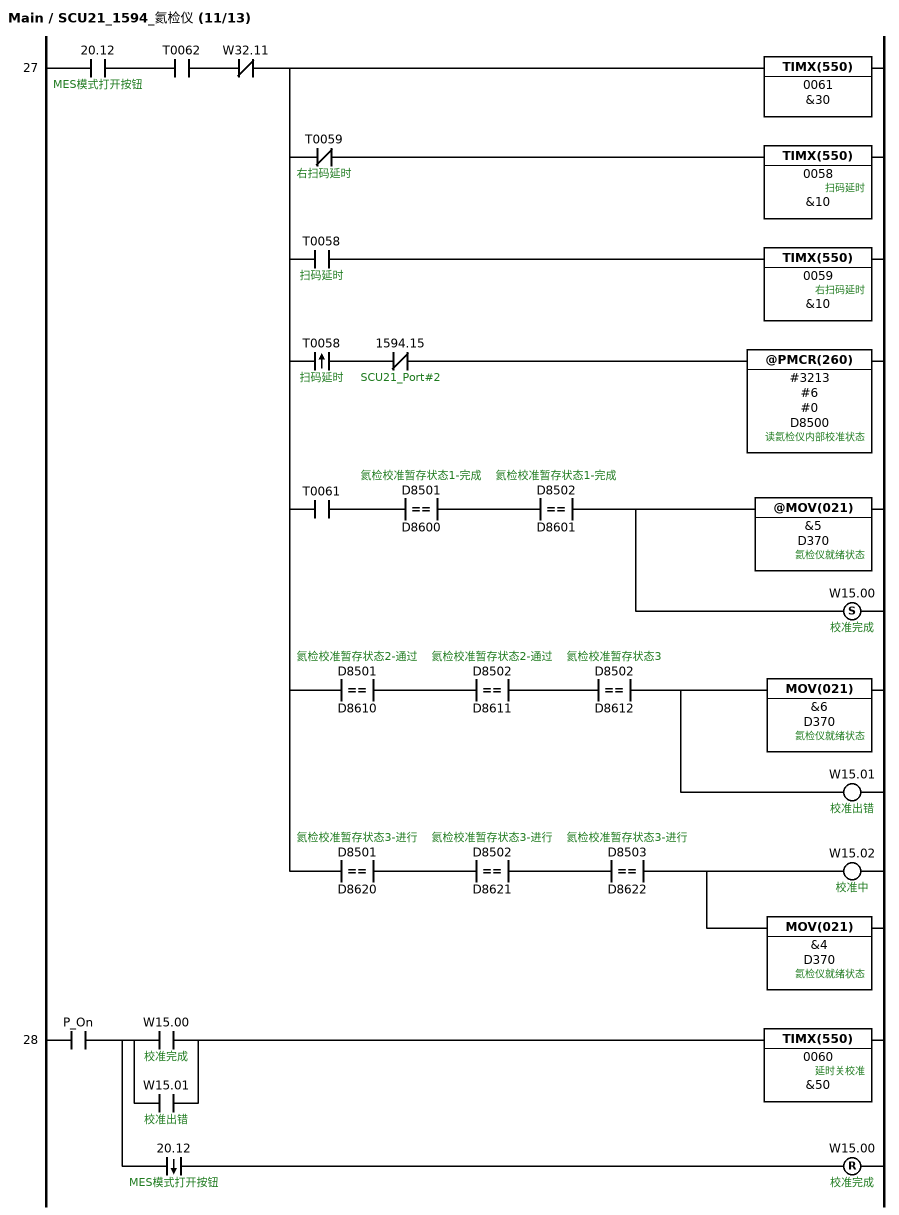
; rung 27
LD 20.12  ; MES模式打开按钮
AND T0062
ANDNOT W32.11
OUT TR0
TIMX(550) 0061 &30
ANDNOT T0059  ; 右扫码延时
TIMX(550) 0058 &10  ; 扫码延时
LD TR0
AND T0058  ; 扫码延时
TIMX(550) 0059 &10  ; 右扫码延时
LD TR0
@AND T0058  ; 扫码延时
ANDNOT 1594.15  ; SCU21_Port#2
@PMCR(260) #3213 #6 #0 D8500  ; 读氦检仪内部校准状态
LD TR0
AND T0061
AND=(300) D8501 D8600  ; 氦检校准暂存状态1-完成
AND=(300) D8502 D8601  ; 氦检校准暂存状态1-完成
@MOV(021) &5 D370  ; 氦检仪就绪状态
SET W15.00  ; 校准完成
LD TR0
AND=(300) D8501 D8610  ; 氦检校准暂存状态2-通过
AND=(300) D8502 D8611  ; 氦检校准暂存状态2-通过
AND=(300) D8502 D8612  ; 氦检校准暂存状态3
MOV(021) &6 D370  ; 氦检仪就绪状态
OUT W15.01  ; 校准出错
LD TR0
AND=(300) D8501 D8620  ; 氦检校准暂存状态3-进行
AND=(300) D8502 D8621  ; 氦检校准暂存状态3-进行
AND=(300) D8503 D8622  ; 氦检校准暂存状态3-进行
OUT W15.02  ; 校准中
MOV(021) &4 D370  ; 氦检仪就绪状态
; rung 28
LD P_On
OUT TR0
LD W15.00  ; 校准完成
OR W15.01  ; 校准出错
ANDLD
TIMX(550) 0060 &50  ; 延时关校准
LD TR0
%AND 20.12  ; MES模式打开按钮
RSET W15.00  ; 校准完成

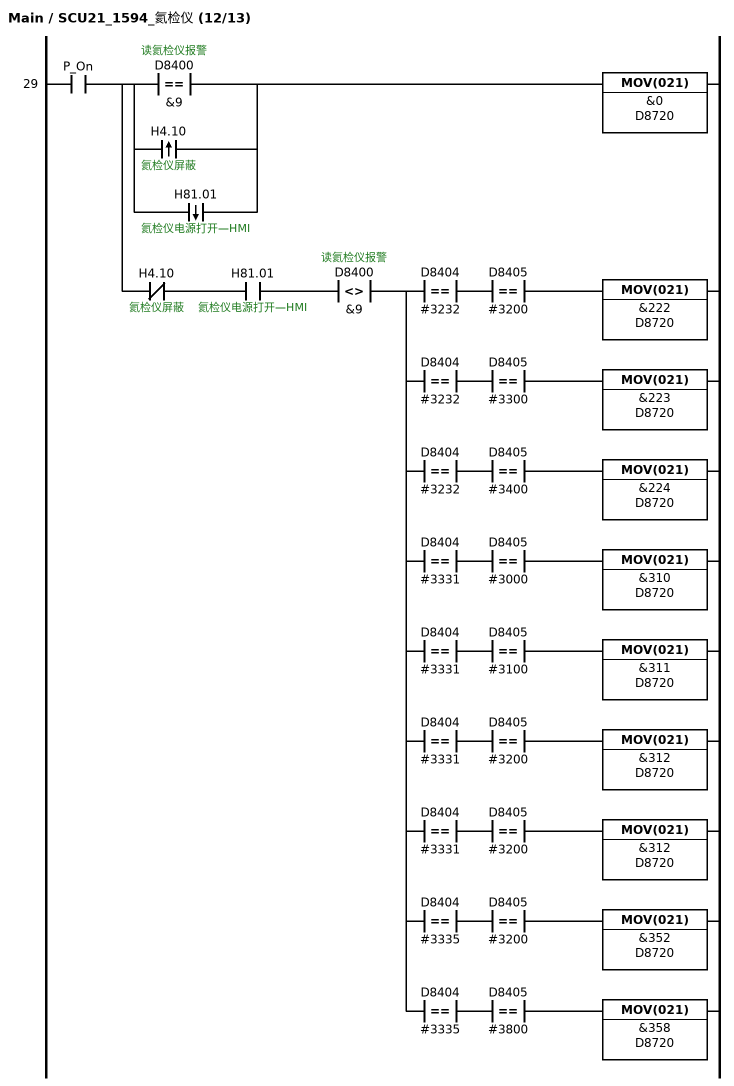
; rung 29
LD P_On
OUT TR0
LD=(300) D8400 &9  ; 读氦检仪报警
@OR H4.10  ; 氦检仪屏蔽
%OR H81.01  ; 氦检仪电源打开—HMI
ANDLD
MOV(021) &0 D8720
LD TR0
ANDNOT H4.10  ; 氦检仪屏蔽
AND H81.01  ; 氦检仪电源打开—HMI
AND<>(305) D8400 &9  ; 读氦检仪报警
OUT TR0
AND=(300) D8404 #3232
AND=(300) D8405 #3200
MOV(021) &222 D8720
LD TR0
AND=(300) D8404 #3232
AND=(300) D8405 #3300
MOV(021) &223 D8720
LD TR0
AND=(300) D8404 #3232
AND=(300) D8405 #3400
MOV(021) &224 D8720
LD TR0
AND=(300) D8404 #3331
AND=(300) D8405 #3000
MOV(021) &310 D8720
LD TR0
AND=(300) D8404 #3331
AND=(300) D8405 #3100
MOV(021) &311 D8720
LD TR0
AND=(300) D8404 #3331
AND=(300) D8405 #3200
MOV(021) &312 D8720
LD TR0
AND=(300) D8404 #3331
AND=(300) D8405 #3200
MOV(021) &312 D8720
LD TR0
AND=(300) D8404 #3335
AND=(300) D8405 #3200
MOV(021) &352 D8720
LD TR0
AND=(300) D8404 #3335
AND=(300) D8405 #3800
MOV(021) &358 D8720

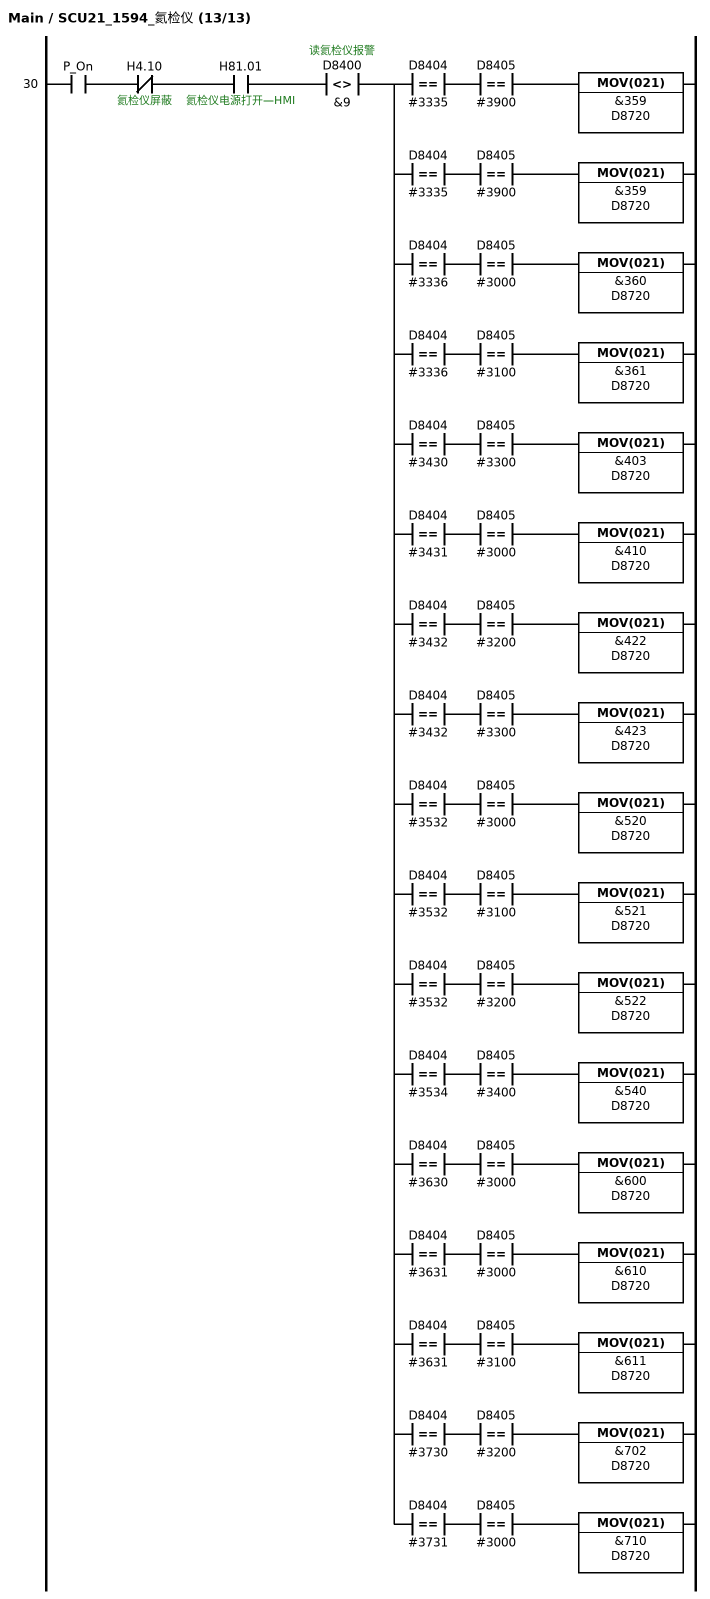
; rung 30
LD P_On
ANDNOT H4.10  ; 氦检仪屏蔽
AND H81.01  ; 氦检仪电源打开—HMI
AND<>(305) D8400 &9  ; 读氦检仪报警
OUT TR0
AND=(300) D8404 #3335
AND=(300) D8405 #3900
MOV(021) &359 D8720
LD TR0
AND=(300) D8404 #3335
AND=(300) D8405 #3900
MOV(021) &359 D8720
LD TR0
AND=(300) D8404 #3336
AND=(300) D8405 #3000
MOV(021) &360 D8720
LD TR0
AND=(300) D8404 #3336
AND=(300) D8405 #3100
MOV(021) &361 D8720
LD TR0
AND=(300) D8404 #3430
AND=(300) D8405 #3300
MOV(021) &403 D8720
LD TR0
AND=(300) D8404 #3431
AND=(300) D8405 #3000
MOV(021) &410 D8720
LD TR0
AND=(300) D8404 #3432
AND=(300) D8405 #3200
MOV(021) &422 D8720
LD TR0
AND=(300) D8404 #3432
AND=(300) D8405 #3300
MOV(021) &423 D8720
LD TR0
AND=(300) D8404 #3532
AND=(300) D8405 #3000
MOV(021) &520 D8720
LD TR0
AND=(300) D8404 #3532
AND=(300) D8405 #3100
MOV(021) &521 D8720
LD TR0
AND=(300) D8404 #3532
AND=(300) D8405 #3200
MOV(021) &522 D8720
LD TR0
AND=(300) D8404 #3534
AND=(300) D8405 #3400
MOV(021) &540 D8720
LD TR0
AND=(300) D8404 #3630
AND=(300) D8405 #3000
MOV(021) &600 D8720
LD TR0
AND=(300) D8404 #3631
AND=(300) D8405 #3000
MOV(021) &610 D8720
LD TR0
AND=(300) D8404 #3631
AND=(300) D8405 #3100
MOV(021) &611 D8720
LD TR0
AND=(300) D8404 #3730
AND=(300) D8405 #3200
MOV(021) &702 D8720
LD TR0
AND=(300) D8404 #3731
AND=(300) D8405 #3000
MOV(021) &710 D8720

### Section AD081_2020

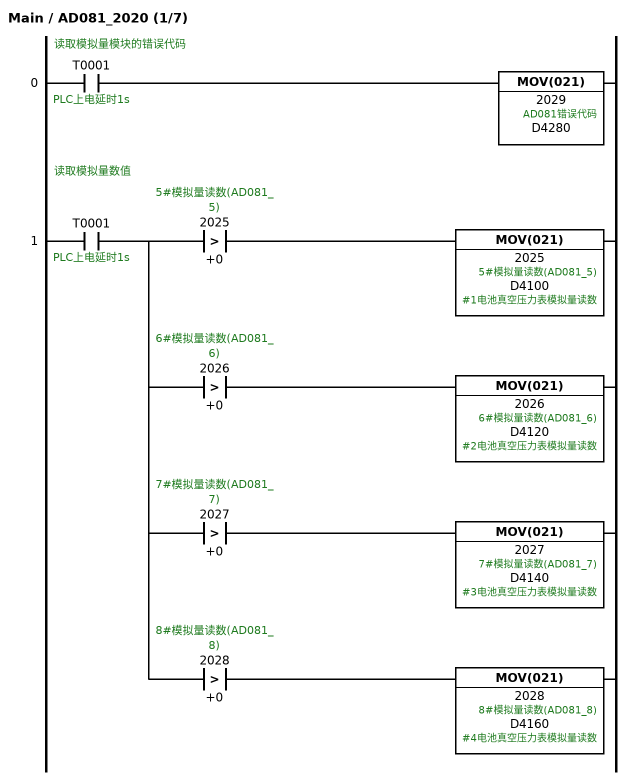
; rung 0: 读取模拟量模块的错误代码
LD T0001  ; PLC上电延时1s
MOV(021) 2029 D4280  ; AD081错误代码
; rung 1: 读取模拟量数值
LD T0001  ; PLC上电延时1s
OUT TR0
AND>S(322) 2025 +0  ; 5#模拟量读数(AD081_5)
MOV(021) 2025 D4100  ; 5#模拟量读数(AD081_5), #1电池真空压力表模拟量读数
LD TR0
AND>S(322) 2026 +0  ; 6#模拟量读数(AD081_6)
MOV(021) 2026 D4120  ; 6#模拟量读数(AD081_6), #2电池真空压力表模拟量读数
LD TR0
AND>S(322) 2027 +0  ; 7#模拟量读数(AD081_7)
MOV(021) 2027 D4140  ; 7#模拟量读数(AD081_7), #3电池真空压力表模拟量读数
LD TR0
AND>S(322) 2028 +0  ; 8#模拟量读数(AD081_8)
MOV(021) 2028 D4160  ; 8#模拟量读数(AD081_8), #4电池真空压力表模拟量读数

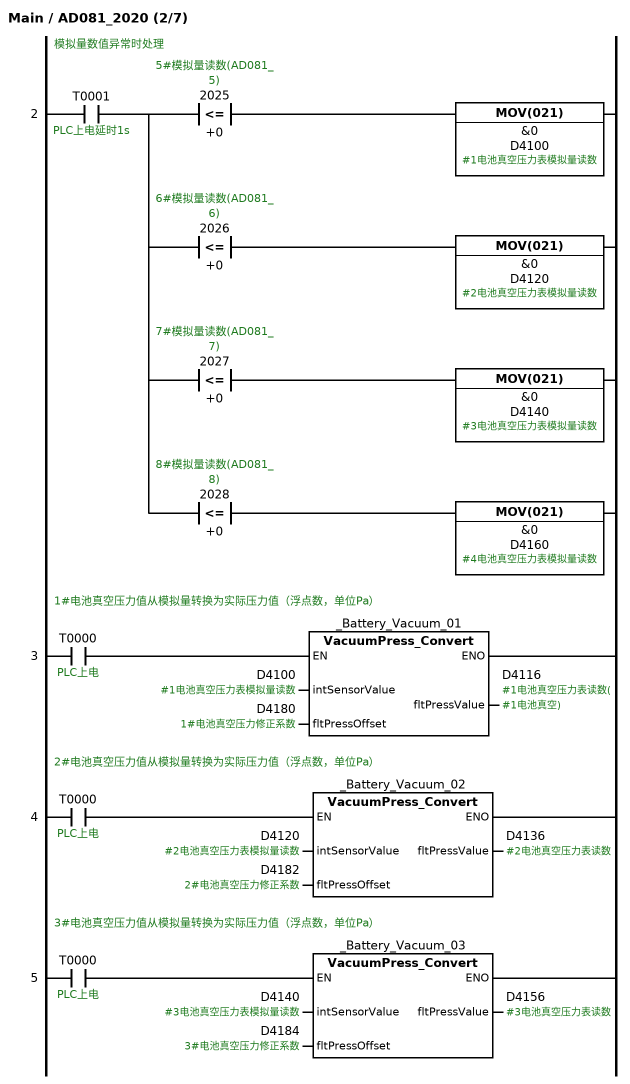
; rung 2: 模拟量数值异常时处理
LD T0001  ; PLC上电延时1s
OUT TR0
AND<=S(317) 2025 +0  ; 5#模拟量读数(AD081_5)
MOV(021) &0 D4100  ; #1电池真空压力表模拟量读数
LD TR0
AND<=S(317) 2026 +0  ; 6#模拟量读数(AD081_6)
MOV(021) &0 D4120  ; #2电池真空压力表模拟量读数
LD TR0
AND<=S(317) 2027 +0  ; 7#模拟量读数(AD081_7)
MOV(021) &0 D4140  ; #3电池真空压力表模拟量读数
LD TR0
AND<=S(317) 2028 +0  ; 8#模拟量读数(AD081_8)
MOV(021) &0 D4160  ; #4电池真空压力表模拟量读数
; rung 3: 1#电池真空压力值从模拟量转换为实际压力值（浮点数，单位Pa）
LD T0000  ; PLC上电
CALL _Battery_Vacuum_01 : VacuumPress_Convert (intSensorValue := D4100, fltPressOffset := D4180, fltPressValue => D4116)  ; #1电池真空压力表模拟量读数, 1#电池真空压力修正系数, #1电池真空压力表读数(#1电池真空)
; rung 4: 2#电池真空压力值从模拟量转换为实际压力值（浮点数，单位Pa）
LD T0000  ; PLC上电
CALL _Battery_Vacuum_02 : VacuumPress_Convert (intSensorValue := D4120, fltPressOffset := D4182, fltPressValue => D4136)  ; #2电池真空压力表模拟量读数, 2#电池真空压力修正系数, #2电池真空压力表读数
; rung 5: 3#电池真空压力值从模拟量转换为实际压力值（浮点数，单位Pa）
LD T0000  ; PLC上电
CALL _Battery_Vacuum_03 : VacuumPress_Convert (intSensorValue := D4140, fltPressOffset := D4184, fltPressValue => D4156)  ; #3电池真空压力表模拟量读数, 3#电池真空压力修正系数, #3电池真空压力表读数

